// TIA Portal project "ContadoresHMI2" (V16)

(* hardware
DEVICE "S71500/ET200MP station_1"  S7-1500 station
   slot 0: "Rail_0"  Rack  6ES7 590-1***0-0AA0
   slot 1: "PLC_1"  CPU 1516-3 PN/DP  6ES7 516-3AN00-0AB0  V1.8
      slot 3: "CPU display_1"  6ES7591-1BA00-0AA0
      slot 32768: "PROFINET interface_1"  X1
         slot 32769: "Port_1"  X1 P1
         slot 32770: "Port_2"  X1 P2
      slot 33024: "PROFINET interface_2"  X2
         slot 33025: "Port_1"  X2 P1
      slot 33280: "DP interface_1"  X3
DEVICE "HMI_1"  TP700 Comfort
   slot 0: "HMI_1"  TP700 Comfort  6AV2 124-0GC01-0AX0  16.0.0.0
   slot 1: "HMI_RT_1"  TP700 Comfort  6AV2 124-0GC01-0AX0  16.0.0.0
   slot 5: "HMI_1.IE_CP_1"  PROFINET Interface  16.0.0.0
      slot 1: "PROFINET Interface_1"  PROFINET Interface
         slot 1: "Port_1"  Port
         slot 2: "Port_2"  Port
   slot 7: "HMI_1.MPI/DP_CP_1"  MPI/DP Interface  16.0.0.0
*)

// ===== PLC "PLC_1"  CPU 1516-3 PN/DP =====

VAR_GLOBAL   // PLC tag table "Default tag table"
   "ReiniciarJuego" AT %M6.0 : Bool;
   "CodigoS0J1" AT %M6.1 : Bool;
   "CodigoS1J1" AT %M6.2 : Bool;
   "CodigoS2J1" AT %M6.3 : Bool;
   "CodigoS3J1" AT %M6.4 : Bool;
   "CodigoO0J1" AT %M6.5 : Bool;
   "CodigoO1J1" AT %M6.6 : Bool;
   "CodigoO2J1" AT %M6.7 : Bool;
   "CodigoO3J1" AT %M7.0 : Bool;
   "CodigoS0J2" AT %M7.1 : Bool;
   "CodigoS1J2" AT %M7.2 : Bool;
   "CodigoS2J2" AT %M7.3 : Bool;
   "CodigoS3J2" AT %M7.4 : Bool;
   "CodigoO0J2" AT %M7.5 : Bool;
   "CodigoO1J2" AT %M7.6 : Bool;
   "CodigoO2J2" AT %M7.7 : Bool;
   "CodigoO3J2" AT %M8.0 : Bool;
   "Intento0J1" AT %M8.1 : Bool;
   "Intento1J1" AT %M8.2 : Bool;
   "Intento2J1" AT %M8.3 : Bool;
   "Intento3J1" AT %M8.4 : Bool;
   "Intento0J2" AT %M8.5 : Bool;
   "Intento1J2" AT %M8.6 : Bool;
   "Intento2J2" AT %M8.7 : Bool;
   "Intento3J2" AT %M9.0 : Bool;
   "IntentoCompletoJ1" AT %MW2 : UInt;
   "IntentoCompletoJ2" AT %MW4 : UInt;
   "Timer" AT %M9.3 : Bool;
   "Repetido" AT %M9.4 : Bool;
   "Panel1CafeJ1" AT %M9.5 : Bool;
   "Panel1RosaJ1" AT %M9.6 : Bool;
   "Panel1MoradoJ1" AT %M9.7 : Bool;
   "Panel1RojoJ1" AT %M10.0 : Bool;
   "Panel1AzulJ1" AT %M10.1 : Bool;
   "Panel1VerdeJ1" AT %M10.2 : Bool;
   "Panel1AmarilloJ1" AT %M10.3 : Bool;
   "Panel2CafeJ1" AT %M10.4 : Bool;
   "Panel2RosaJ1" AT %M10.5 : Bool;
   "Panel2MoradoJ1" AT %M10.6 : Bool;
   "Panel2RojoJ1" AT %M10.7 : Bool;
   "Panel2AzulJ1" AT %M11.0 : Bool;
   "Panel2VerdeJ1" AT %M11.1 : Bool;
   "Panel2AmarilloJ1" AT %M11.2 : Bool;
   "Panel1CafeJ2" AT %M11.3 : Bool;
   "Panel1RosaJ2" AT %M11.4 : Bool;
   "Panel1MoradoJ2" AT %M11.5 : Bool;
   "Panel1RojoJ2" AT %M11.6 : Bool;
   "Panel1AzulJ2" AT %M11.7 : Bool;
   "Panel1VerdeJ2" AT %M12.0 : Bool;
   "Panel1AmarilloJ2" AT %M12.1 : Bool;
   "Panel2CafeJ2" AT %M12.2 : Bool;
   "Panel2RosaJ2" AT %M12.3 : Bool;
   "Panel2MoradoJ2" AT %M12.4 : Bool;
   "Panel2RojoJ2" AT %M12.5 : Bool;
   "Panel2AzulJ2" AT %M12.6 : Bool;
   "Panel2VerdeJ2" AT %M12.7 : Bool;
   "Panel2AmarilloJ2" AT %M13.0 : Bool;
   "Panel1J1Activado" AT %M13.1 : Bool;
   "Panel2J1Activado" AT %M13.2 : Bool;
   "Panel1J2Activado" AT %M13.3 : Bool;
   "Panel2J2Activado" AT %M13.4 : Bool;
   "ReinicioCorrecto" AT %M13.5 : Bool;
   "Bounce1" AT %M13.6 : Bool;
   "Bounce2" AT %M13.7 : Bool;
   "Bounce3" AT %M14.0 : Bool;
   "Bounce5" AT %M14.1 : Bool;
   "Bounce6" AT %M14.2 : Bool;
   "Bounce7" AT %M14.3 : Bool;
   "Bounce8" AT %M14.4 : Bool;
   "Bounce10" AT %M14.5 : Bool;
   "MensajeCorrecto" AT %M14.6 : Bool;
   "Bounce4" AT %M14.7 : Bool;
   "Bounce9" AT %M15.0 : Bool;
   "ReiniciarContadorJ1" AT %M15.1 : Bool;
   "ReiniciarContadorJ2" AT %M15.2 : Bool;
   "ChecarIntento1J1" AT %M15.3 : Bool;
   "ChecarIntento2J1" AT %M15.4 : Bool;
   "ChecarIntento3J1" AT %M15.5 : Bool;
   "ChecarIntento4J1" AT %M15.6 : Bool;
   "ChecarIntento1J2" AT %M15.7 : Bool;
   "ChecarIntento2J2" AT %M16.0 : Bool;
   "ChecarIntento3J2" AT %M16.1 : Bool;
   "ChecarIntento4J2" AT %M16.2 : Bool;
   "ContadorCorr" AT %MW17 : UInt;
   "ContadorSimi" AT %MW20 : UInt;
   "ContadorError" AT %MW22 : UInt;
   "ContadorCorrTemp" AT %MW24 : UInt;
   "ContadorSimiTemp" AT %MW26 : UInt;
   "ReiniciarChecarCorr" AT %M28.0 : Bool;
   "ReiniciarChecarSimi" AT %M28.1 : Bool;
   "ReiniciarChecarError" AT %M28.2 : Bool;
   "ChecarIntentoCorrecto" AT %M28.3 : Bool;
   "ChecarIntento1SJ1" AT %M28.4 : Bool;
   "ChecarIntento2SJ1" AT %M28.5 : Bool;
   "ChecarIntento3SJ1" AT %M28.6 : Bool;
   "ChecarIntento4SJ1" AT %M28.7 : Bool;
   "ChecarIntento1SJ2" AT %M29.0 : Bool;
   "ChecarIntento2SJ2" AT %M29.1 : Bool;
   "ChecarIntento3SJ2" AT %M29.2 : Bool;
   "ChecarIntento4SJ2" AT %M29.3 : Bool;
   "CorrectasSimilares" AT %M29.4 : Bool;
   "IntentoCompletoCORR" AT %MW31 : UInt;
   "ReiniciarCorrSimiDisp" AT %M34.0 : Bool;
   "CondicionGanasteJ1" AT %M34.1 : Bool;
   "CondicionPerdisteJ1" AT %M34.2 : Bool;
   "CondicionGanasteJ2" AT %M34.3 : Bool;
   "CondicionPerdisteJ2" AT %M34.4 : Bool;
END_VAR

DATA_BLOCK "Var"   // DB3
{ S7_Optimized_Access := 'TRUE' }
VERSION : 0.1
   VAR
      V1 : Array[0..10, 0..10] of Int;
      CodigoSJ1 : Array[0..3] of Int;
      CodigoOJ1 : Array[0..3] of Int;
      CodigoSJ2 : Array[0..3] of Int;
      CodigoOJ2 : Array[0..3] of Int;
      VectorPrincipalJ1 : Array[0..7, 0..3] of Int;
      VectorSecundarioJ1 : Array[0..7, 0..3] of Int;
      VectorPrincipalJ2 : Array[0..7, 0..3] of Int;
      VectorSecundarioJ2 : Array[0..7, 0..3] of Int;
      VectorMensajes : Array[0..10] of Int;
      VectorMensajesReset : Array[0..10] of Int;
      VectorMensajesJ2 : Array[0..10] of Int;
      VectorMensajesResetJ2 : Array[0..10] of Int;
      VectorCorrectas : Array[0..7, 0..3] of Int;
      VectorCorrectasReset : Array[0..7, 0..3] of Int;
      CodigoSimilaresJ1 : Array[0..3] of Int;
      CodigoSimilaresJ1Temp : Array[0..3] of Int;
   END_VAR
BEGIN
END_DATA_BLOCK

// folder: System blocks/Program resources

DATA_BLOCK "ContadorCorrectas"   // DB1
{ S7_Optimized_Access := 'TRUE' }
AUTHOR : Simatic
FAMILY : IEC
NAME : UCNTR
VERSION : 1.2
// stored: InstanceOfName IEC_UCOUNTER
"IEC_UCOUNTER"
BEGIN
END_DATA_BLOCK

DATA_BLOCK "IEC_Counter_0_DB_1"   // DB2
{ S7_Optimized_Access := 'TRUE' }
AUTHOR : Simatic
FAMILY : IEC
NAME : UCNTR
VERSION : 1.2
// stored: InstanceOfName IEC_UCOUNTER
"IEC_UCOUNTER"
BEGIN
END_DATA_BLOCK

DATA_BLOCK "IEC_Timer_1_DB"   // DB4
{ S7_Optimized_Access := 'TRUE' }
AUTHOR : Simatic
FAMILY : IEC
NAME : IEC_TMR
VERSION : 1.0
// stored: InstanceOfName IEC_TIMER
"IEC_TIMER"
BEGIN
END_DATA_BLOCK

DATA_BLOCK "IEC_Timer_0_DB_1"   // DB5
{ S7_Optimized_Access := 'TRUE' }
AUTHOR : Simatic
FAMILY : IEC
NAME : IEC_TMR
VERSION : 1.0
// stored: InstanceOfName IEC_TIMER
"IEC_TIMER"
BEGIN
END_DATA_BLOCK

DATA_BLOCK "IEC_Timer_2_DB"   // DB6
{ S7_Optimized_Access := 'TRUE' }
AUTHOR : Simatic
FAMILY : IEC
NAME : IEC_TMR
VERSION : 1.0
// stored: InstanceOfName IEC_TIMER
"IEC_TIMER"
BEGIN
END_DATA_BLOCK

DATA_BLOCK "IEC_Timer_3_DB"   // DB7
{ S7_Optimized_Access := 'TRUE' }
AUTHOR : Simatic
FAMILY : IEC
NAME : IEC_TMR
VERSION : 1.0
// stored: InstanceOfName IEC_TIMER
"IEC_TIMER"
BEGIN
END_DATA_BLOCK

DATA_BLOCK "IEC_Timer_4_DB"   // DB8
{ S7_Optimized_Access := 'TRUE' }
AUTHOR : Simatic
FAMILY : IEC
NAME : IEC_TMR
VERSION : 1.0
// stored: InstanceOfName IEC_TIMER
"IEC_TIMER"
BEGIN
END_DATA_BLOCK

DATA_BLOCK "IEC_Timer_5_DB"   // DB9
{ S7_Optimized_Access := 'TRUE' }
AUTHOR : Simatic
FAMILY : IEC
NAME : IEC_TMR
VERSION : 1.0
// stored: InstanceOfName IEC_TIMER
"IEC_TIMER"
BEGIN
END_DATA_BLOCK

DATA_BLOCK "ContadorSimilares"   // DB10
{ S7_Optimized_Access := 'TRUE' }
AUTHOR : Simatic
FAMILY : IEC
NAME : UCNTR
VERSION : 1.2
// stored: InstanceOfName IEC_UCOUNTER
"IEC_UCOUNTER"
BEGIN
END_DATA_BLOCK

// folder: (top level)

ORGANIZATION_BLOCK "Main"   // OB1, LAD, ProgramCycle
TITLE = "Main Program Sweep (Cycle)"
{ S7_Optimized_Access := 'TRUE' }
VERSION : 0.1
   VAR_INPUT
      Initial_Call : Bool;   // Initial call of this OB
      Remanence : Bool;   // =True, if remanent data are available
   END_VAR
   VAR_TEMP   // added for the SCL form of the ladder/FBD networks
      _w1 : Bool;
      _w2 : Bool;
      _w3 : Bool;
      _w4 : Bool;
      _w5 : Bool;
      _w6 : Bool;
      _w7 : Bool;
      _w8 : Bool;
      _w9 : Bool;
      _w10 : Bool;
      _w11 : Bool;
      _w12 : Bool;
      _w13 : Bool;
      _w14 : Bool;
      _w15 : Bool;
      _w16 : Bool;
      _w17 : Bool;
      _w18 : Bool;
      _w19 : Bool;
      _w20 : Bool;
      _w21 : Bool;
      _w22 : Bool;
      _w23 : Bool;
      _w24 : Bool;
      _w25 : Bool;
      _w26 : Bool;
      _w27 : Bool;
      _w28 : Bool;
      _w29 : Bool;
      _w30 : Bool;
      _w31 : Bool;
      _w32 : Bool;
      _w33 : Bool;
      _w34 : Bool;
      _w35 : Bool;
      _w36 : Bool;
      _w37 : Bool;
      _w38 : Bool;
      _w39 : Bool;
      _w40 : Bool;
      _w41 : Bool;
      _w42 : Bool;
      _w43 : Bool;
      _w44 : Bool;
      _w45 : Bool;
      _w46 : Bool;
      _w47 : Bool;
      _w48 : Bool;
      _w49 : Bool;
      _w50 : Bool;
      _w51 : Bool;
      _w52 : Bool;
      _w53 : Bool;
      _w54 : Bool;
      _w55 : Bool;
      _w56 : Bool;
      _w57 : Bool;
      _w58 : Bool;
      _w59 : Bool;
      _w60 : Bool;
      _w61 : Bool;
      _w62 : Bool;
      _w63 : Bool;
      _w64 : Bool;
      _w65 : Bool;
      _w66 : Bool;
      _w67 : Bool;
      _w68 : Bool;
      _w69 : Bool;
      _w70 : Bool;
      _w71 : Bool;
      _w72 : Bool;
      _w73 : Bool;
      _w74 : Bool;
      _w75 : Bool;
      _w76 : Bool;
      _w77 : Bool;
      _w78 : Bool;
      _w79 : Bool;
      _w80 : Bool;
      _w81 : Bool;
      _w82 : Bool;
      _w83 : Bool;
      _w84 : Bool;
      _w85 : Bool;
      _w86 : Bool;
      _w87 : Bool;
      _w88 : Bool;
   END_VAR
BEGIN

REGION Network 1: Reiniciar Juego
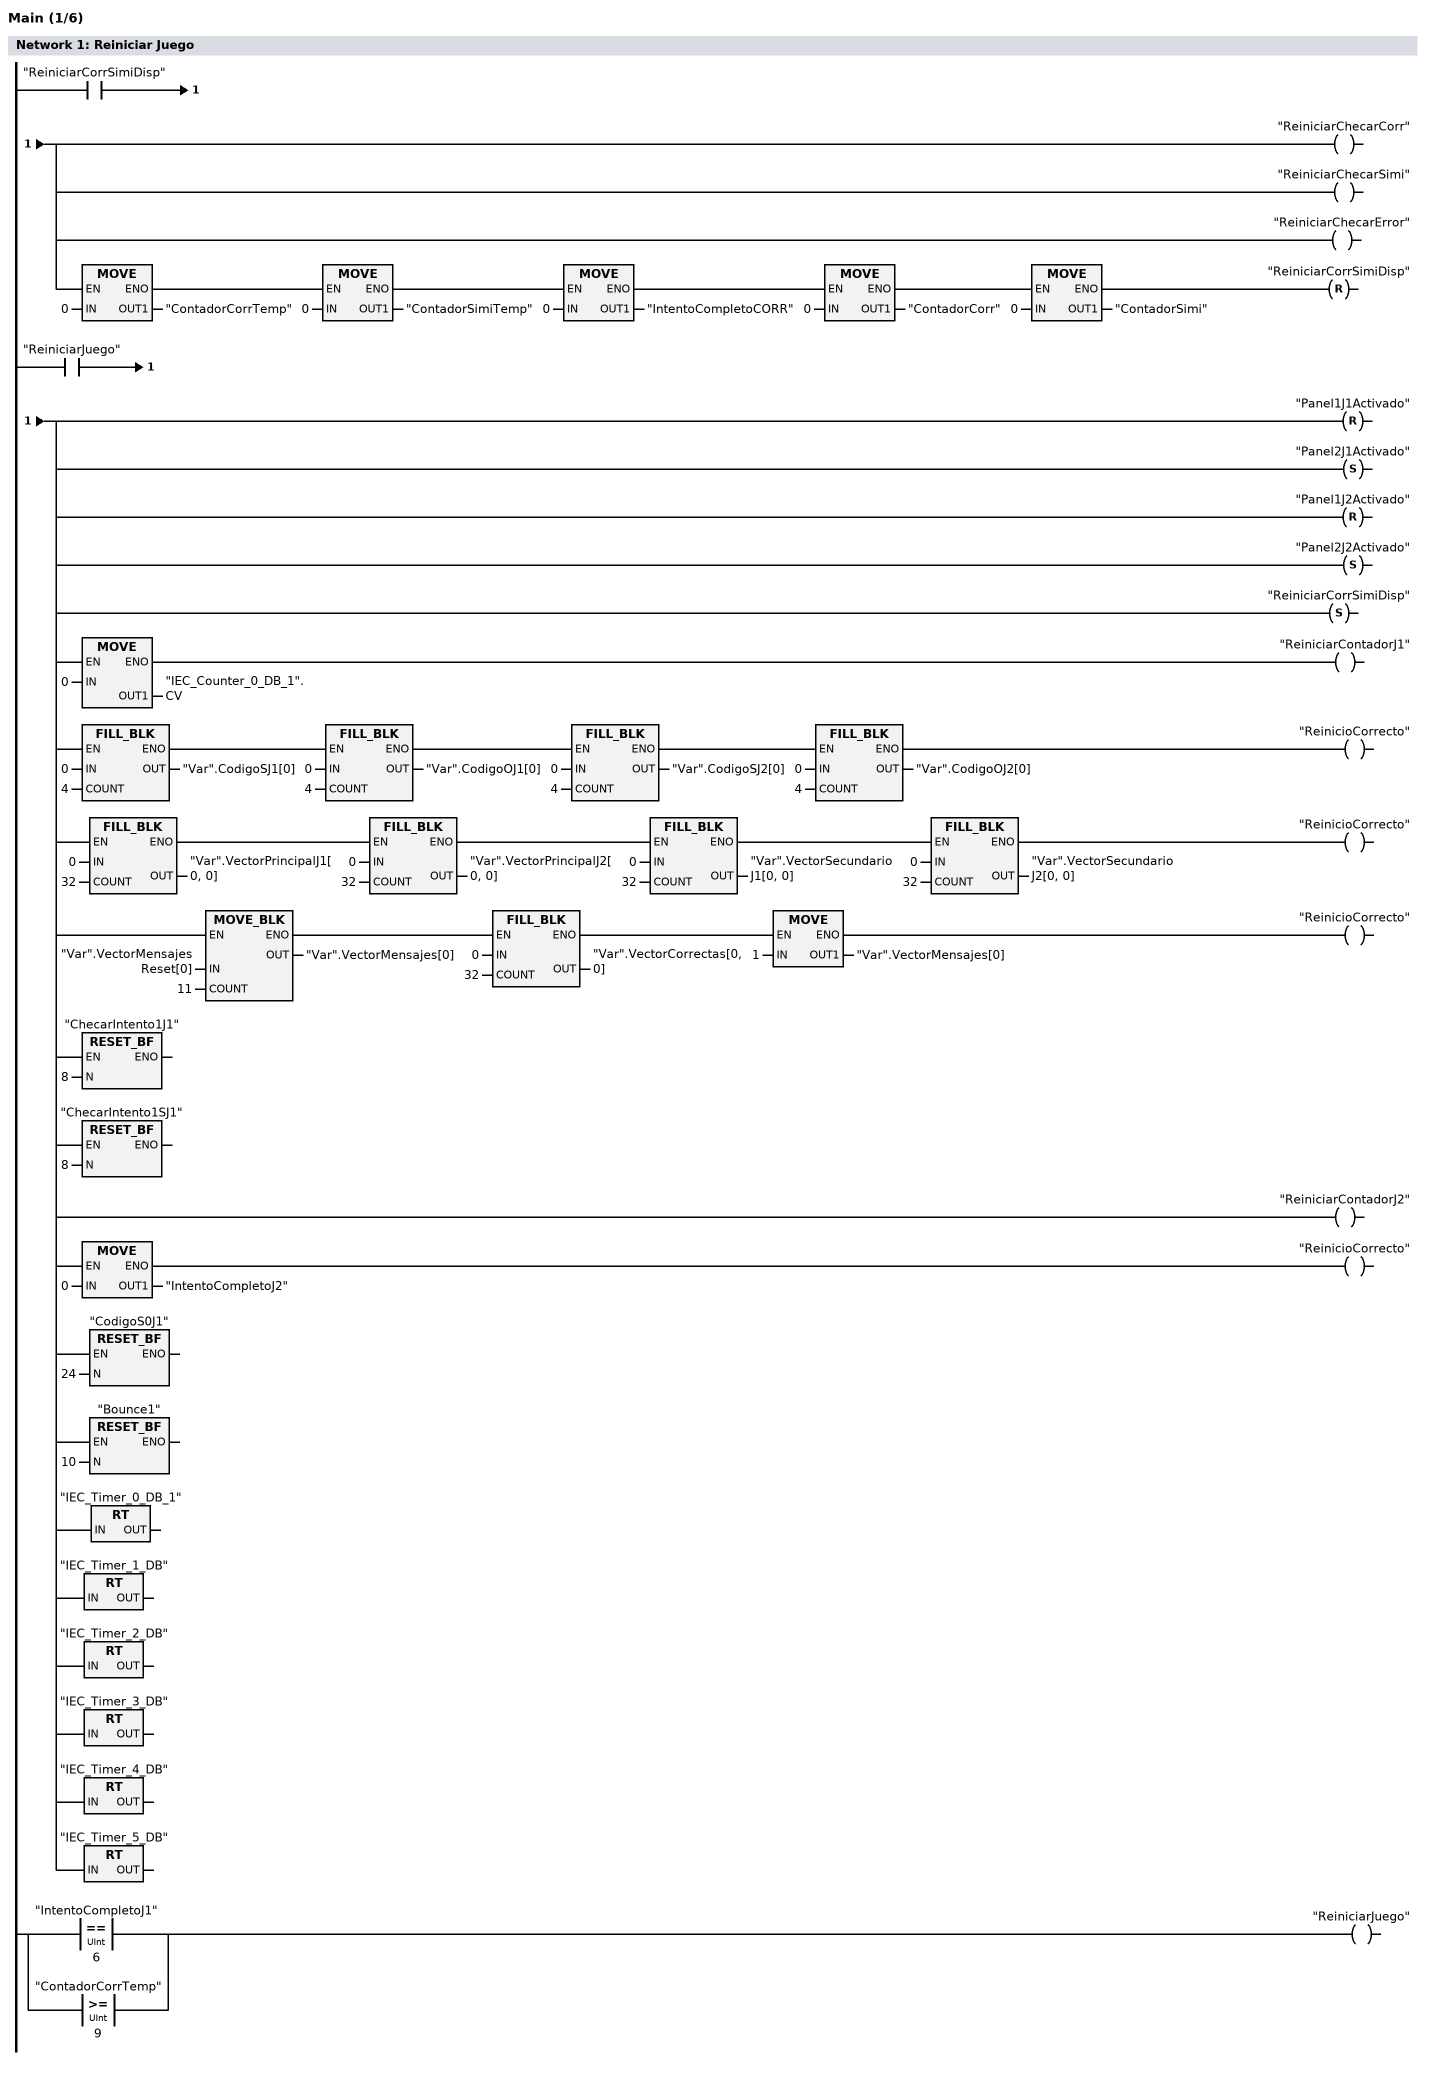
   // no SCL statement known for RBitfield: written as a call
   "ReiniciarChecarCorr" := "ReiniciarCorrSimiDisp";
   "ReiniciarChecarSimi" := "ReiniciarCorrSimiDisp";
   "ReiniciarChecarError" := "ReiniciarCorrSimiDisp";
   IF "ReiniciarCorrSimiDisp" THEN
       "ContadorCorrTemp" := 0;
       "ContadorSimiTemp" := 0;
       "IntentoCompletoCORR" := 0;
       "ContadorCorr" := 0;
       "ContadorSimi" := 0;
       "ReiniciarCorrSimiDisp" := FALSE;
   END_IF;
   IF "ReiniciarJuego" THEN
       "Panel1J1Activado" := FALSE;
       "Panel2J1Activado" := TRUE;
       "Panel1J2Activado" := FALSE;
       "Panel2J2Activado" := TRUE;
       "ReiniciarCorrSimiDisp" := TRUE;
       "IEC_Counter_0_DB_1".CV := 0;
   END_IF;
   "ReiniciarContadorJ1" := "ReiniciarJuego";
   #_w1 := "ReiniciarJuego";
   #_w2 := "ReiniciarJuego";
   IF #_w2 THEN
       FILL_BLK(IN := 0, COUNT := 4, OUT => "Var".CodigoSJ1[0]);
       FILL_BLK(IN := 0, COUNT := 4, OUT => "Var".CodigoOJ1[0]);
       FILL_BLK(IN := 0, COUNT := 4, OUT => "Var".CodigoSJ2[0]);
       FILL_BLK(IN := 0, COUNT := 4, OUT => "Var".CodigoOJ2[0]);
   END_IF;
   "ReinicioCorrecto" := #_w2;
   IF #_w1 THEN
       FILL_BLK(IN := 0, COUNT := 32, OUT => "Var".VectorPrincipalJ1[0, 0]);
       FILL_BLK(IN := 0, COUNT := 32, OUT => "Var".VectorPrincipalJ2[0, 0]);
       FILL_BLK(IN := 0, COUNT := 32, OUT => "Var".VectorSecundarioJ1[0, 0]);
       FILL_BLK(IN := 0, COUNT := 32, OUT => "Var".VectorSecundarioJ2[0, 0]);
   END_IF;
   "ReinicioCorrecto" := #_w1;
   IF #_w1 THEN
       MOVE_BLK(IN := "Var".VectorMensajesReset[0], COUNT := 11, OUT => "Var".VectorMensajes[0]);
       FILL_BLK(IN := 0, COUNT := 32, OUT => "Var".VectorCorrectas[0, 0]);
       "Var".VectorMensajes[0] := 1;
   END_IF;
   "ReinicioCorrecto" := #_w1;
   IF #_w1 THEN
       RESET_BF(operand := "ChecarIntento1J1", n := 8);
       RESET_BF(operand := "ChecarIntento1SJ1", n := 8);
   END_IF;
   "ReiniciarContadorJ2" := #_w1;
   IF #_w1 THEN "IntentoCompletoJ2" := 0; END_IF;
   "ReinicioCorrecto" := #_w1;
   IF #_w1 THEN
       RESET_BF(operand := "CodigoS0J1", n := 24);
       RESET_BF(operand := "Bounce1", n := 10);
       RESET_TIMER("IEC_Timer_0_DB_1");
       RESET_TIMER("IEC_Timer_1_DB");
       RESET_TIMER("IEC_Timer_2_DB");
       RESET_TIMER("IEC_Timer_3_DB");
       RESET_TIMER("IEC_Timer_4_DB");
       RESET_TIMER("IEC_Timer_5_DB");
   END_IF;
   "ReiniciarJuego" := ("IntentoCompletoJ1" = 6) OR ("ContadorCorrTemp" >= 9);
END_REGION

REGION Network 2: Seleccionar Codigo
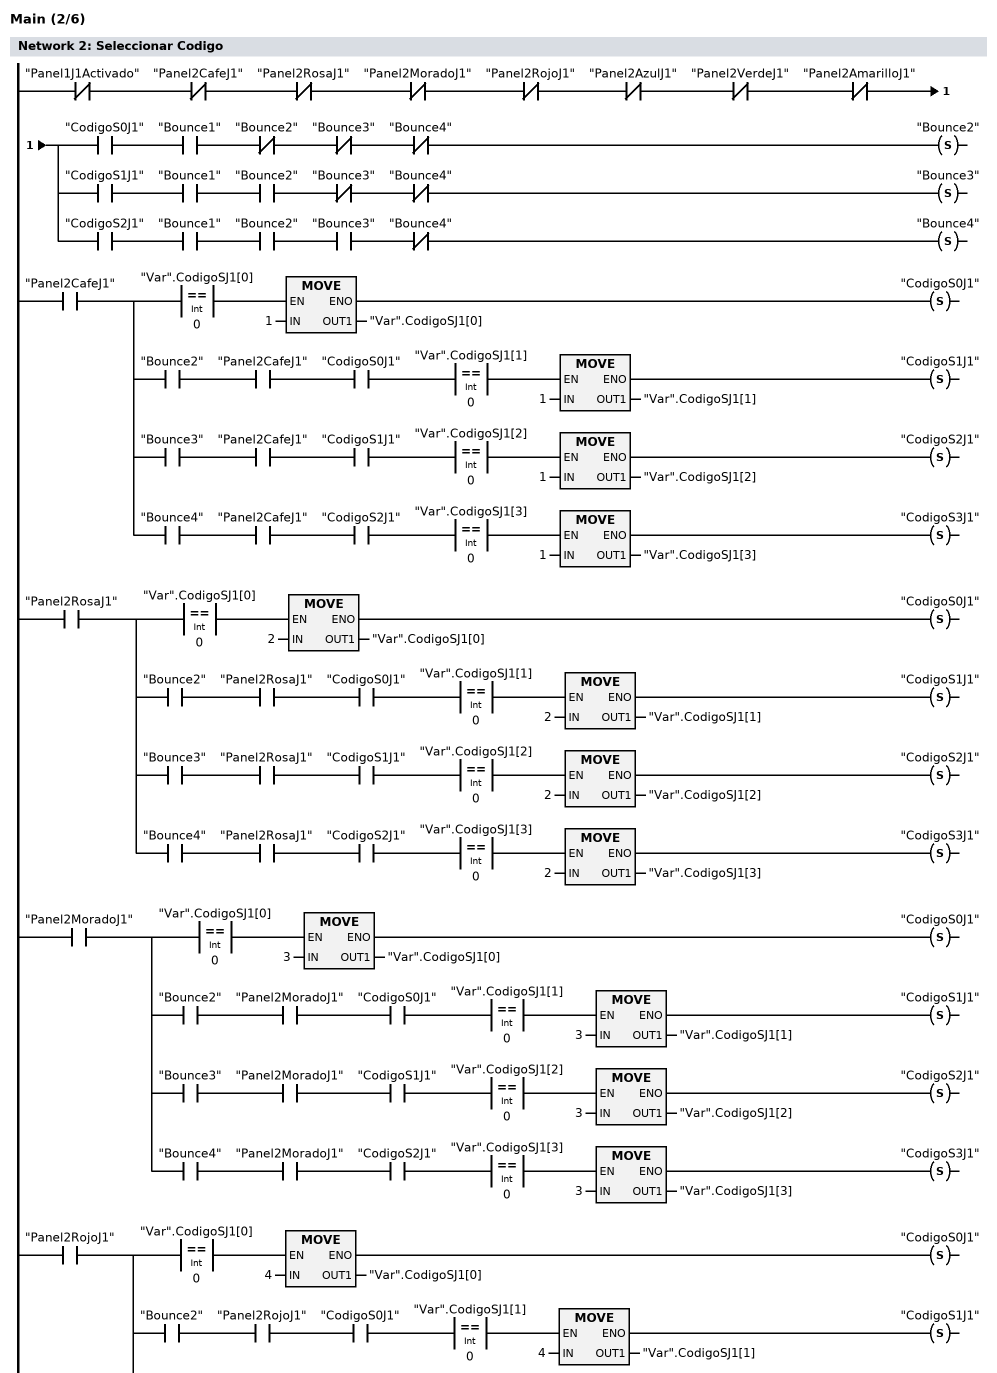
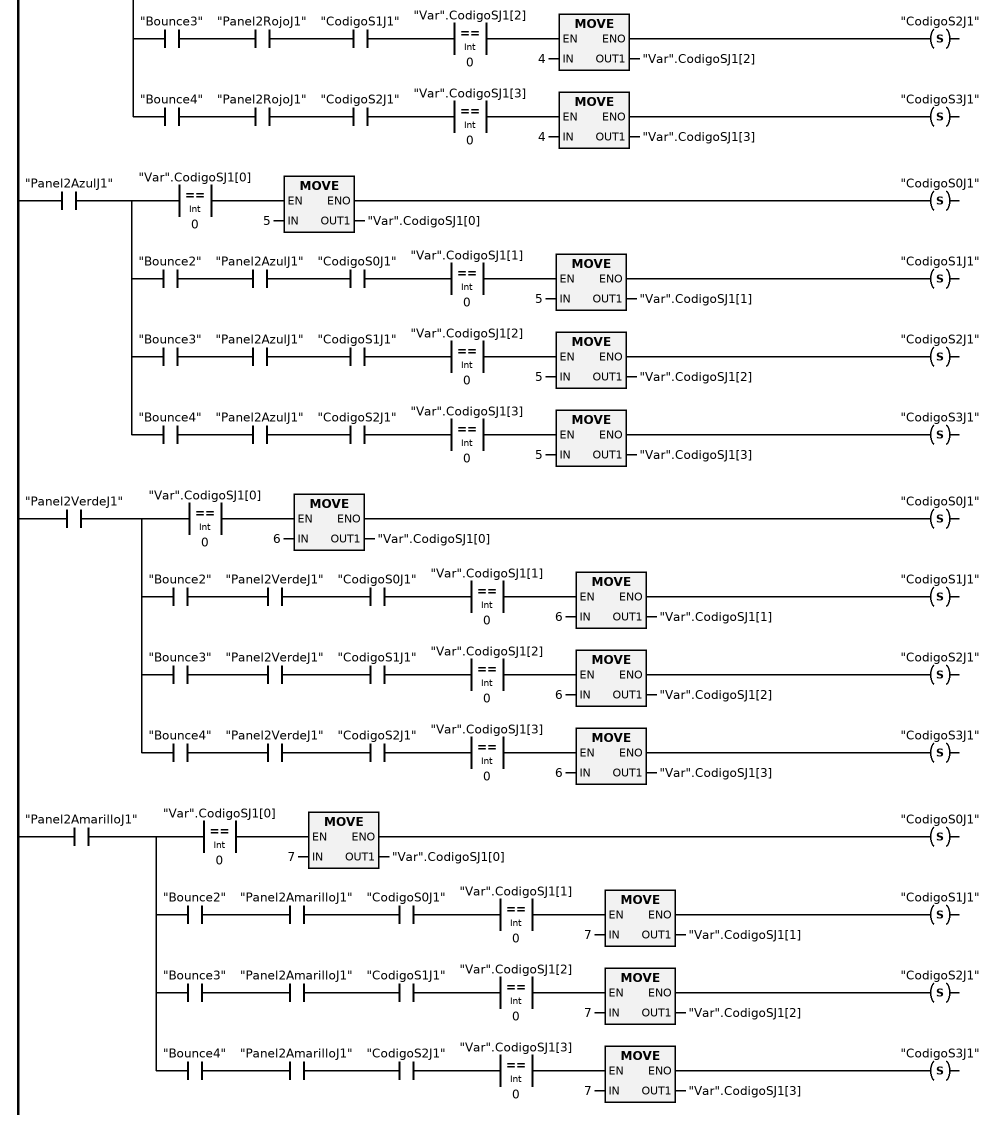
   RUNG wire#powerrail
      I_Contact( "Panel1J1Activado" )
      I_Contact( "Panel2CafeJ1" )
      I_Contact( "Panel2RosaJ1" )
      I_Contact( "Panel2MoradoJ1" )
      I_Contact( "Panel2RojoJ1" )
      I_Contact( "Panel2AzulJ1" )
      I_Contact( "Panel2VerdeJ1" )
      I_Contact( "Panel2AmarilloJ1" )
      wire#w1
      Contact( "CodigoS0J1" )
      Contact( "Bounce1" )
      I_Contact( "Bounce2" )
      I_Contact( "Bounce3" )
      I_Contact( "Bounce4" )
      S_Coil( "Bounce2" )
   END_RUNG
   RUNG wire#w1
      Contact( "CodigoS1J1" )
      Contact( "Bounce1" )
      Contact( "Bounce2" )
      I_Contact( "Bounce3" )
      I_Contact( "Bounce4" )
      S_Coil( "Bounce3" )
   END_RUNG
   RUNG wire#w1
      Contact( "CodigoS2J1" )
      Contact( "Bounce1" )
      Contact( "Bounce2" )
      Contact( "Bounce3" )
      I_Contact( "Bounce4" )
      S_Coil( "Bounce4" )
   END_RUNG
   RUNG wire#powerrail
      Contact( "Panel2CafeJ1" )
      wire#w2
      { S7_Templates := "SrcType := Int" } EQ_Contact(in1 := "Var".CodigoSJ1[0], in2 := 0)
      Move(in := 1, out1 => "Var".CodigoSJ1[0])
      S_Coil( "CodigoS0J1" )
   END_RUNG
   RUNG wire#w2
      Contact( "Bounce2" )
      Contact( "Panel2CafeJ1" )
      Contact( "CodigoS0J1" )
      { S7_Templates := "SrcType := Int" } EQ_Contact(in1 := "Var".CodigoSJ1[1], in2 := 0)
      Move(in := 1, out1 => "Var".CodigoSJ1[1])
      S_Coil( "CodigoS1J1" )
   END_RUNG
   RUNG wire#w2
      Contact( "Bounce3" )
      Contact( "Panel2CafeJ1" )
      Contact( "CodigoS1J1" )
      { S7_Templates := "SrcType := Int" } EQ_Contact(in1 := "Var".CodigoSJ1[2], in2 := 0)
      Move(in := 1, out1 => "Var".CodigoSJ1[2])
      S_Coil( "CodigoS2J1" )
   END_RUNG
   RUNG wire#w2
      Contact( "Bounce4" )
      Contact( "Panel2CafeJ1" )
      Contact( "CodigoS2J1" )
      { S7_Templates := "SrcType := Int" } EQ_Contact(in1 := "Var".CodigoSJ1[3], in2 := 0)
      Move(in := 1, out1 => "Var".CodigoSJ1[3])
      S_Coil( "CodigoS3J1" )
   END_RUNG
   RUNG wire#powerrail
      Contact( "Panel2RosaJ1" )
      wire#w3
      { S7_Templates := "SrcType := Int" } EQ_Contact(in1 := "Var".CodigoSJ1[0], in2 := 0)
      Move(in := 2, out1 => "Var".CodigoSJ1[0])
      S_Coil( "CodigoS0J1" )
   END_RUNG
   RUNG wire#w3
      Contact( "Bounce2" )
      Contact( "Panel2RosaJ1" )
      Contact( "CodigoS0J1" )
      { S7_Templates := "SrcType := Int" } EQ_Contact(in1 := "Var".CodigoSJ1[1], in2 := 0)
      Move(in := 2, out1 => "Var".CodigoSJ1[1])
      S_Coil( "CodigoS1J1" )
   END_RUNG
   RUNG wire#w3
      Contact( "Bounce3" )
      Contact( "Panel2RosaJ1" )
      Contact( "CodigoS1J1" )
      { S7_Templates := "SrcType := Int" } EQ_Contact(in1 := "Var".CodigoSJ1[2], in2 := 0)
      Move(in := 2, out1 => "Var".CodigoSJ1[2])
      S_Coil( "CodigoS2J1" )
   END_RUNG
   RUNG wire#w3
      Contact( "Bounce4" )
      Contact( "Panel2RosaJ1" )
      Contact( "CodigoS2J1" )
      { S7_Templates := "SrcType := Int" } EQ_Contact(in1 := "Var".CodigoSJ1[3], in2 := 0)
      Move(in := 2, out1 => "Var".CodigoSJ1[3])
      S_Coil( "CodigoS3J1" )
   END_RUNG
   RUNG wire#powerrail
      Contact( "Panel2MoradoJ1" )
      wire#w4
      { S7_Templates := "SrcType := Int" } EQ_Contact(in1 := "Var".CodigoSJ1[0], in2 := 0)
      Move(in := 3, out1 => "Var".CodigoSJ1[0])
      S_Coil( "CodigoS0J1" )
   END_RUNG
   RUNG wire#w4
      Contact( "Bounce2" )
      Contact( "Panel2MoradoJ1" )
      Contact( "CodigoS0J1" )
      { S7_Templates := "SrcType := Int" } EQ_Contact(in1 := "Var".CodigoSJ1[1], in2 := 0)
      Move(in := 3, out1 => "Var".CodigoSJ1[1])
      S_Coil( "CodigoS1J1" )
   END_RUNG
   RUNG wire#w4
      Contact( "Bounce3" )
      Contact( "Panel2MoradoJ1" )
      Contact( "CodigoS1J1" )
      { S7_Templates := "SrcType := Int" } EQ_Contact(in1 := "Var".CodigoSJ1[2], in2 := 0)
      Move(in := 3, out1 => "Var".CodigoSJ1[2])
      S_Coil( "CodigoS2J1" )
   END_RUNG
   RUNG wire#w4
      Contact( "Bounce4" )
      Contact( "Panel2MoradoJ1" )
      Contact( "CodigoS2J1" )
      { S7_Templates := "SrcType := Int" } EQ_Contact(in1 := "Var".CodigoSJ1[3], in2 := 0)
      Move(in := 3, out1 => "Var".CodigoSJ1[3])
      S_Coil( "CodigoS3J1" )
   END_RUNG
   RUNG wire#powerrail
      Contact( "Panel2RojoJ1" )
      wire#w5
      { S7_Templates := "SrcType := Int" } EQ_Contact(in1 := "Var".CodigoSJ1[0], in2 := 0)
      Move(in := 4, out1 => "Var".CodigoSJ1[0])
      S_Coil( "CodigoS0J1" )
   END_RUNG
   RUNG wire#w5
      Contact( "Bounce2" )
      Contact( "Panel2RojoJ1" )
      Contact( "CodigoS0J1" )
      { S7_Templates := "SrcType := Int" } EQ_Contact(in1 := "Var".CodigoSJ1[1], in2 := 0)
      Move(in := 4, out1 => "Var".CodigoSJ1[1])
      S_Coil( "CodigoS1J1" )
   END_RUNG
   RUNG wire#w5
      Contact( "Bounce3" )
      Contact( "Panel2RojoJ1" )
      Contact( "CodigoS1J1" )
      { S7_Templates := "SrcType := Int" } EQ_Contact(in1 := "Var".CodigoSJ1[2], in2 := 0)
      Move(in := 4, out1 => "Var".CodigoSJ1[2])
      S_Coil( "CodigoS2J1" )
   END_RUNG
   RUNG wire#w5
      Contact( "Bounce4" )
      Contact( "Panel2RojoJ1" )
      Contact( "CodigoS2J1" )
      { S7_Templates := "SrcType := Int" } EQ_Contact(in1 := "Var".CodigoSJ1[3], in2 := 0)
      Move(in := 4, out1 => "Var".CodigoSJ1[3])
      S_Coil( "CodigoS3J1" )
   END_RUNG
   RUNG wire#powerrail
      Contact( "Panel2AzulJ1" )
      wire#w6
      { S7_Templates := "SrcType := Int" } EQ_Contact(in1 := "Var".CodigoSJ1[0], in2 := 0)
      Move(in := 5, out1 => "Var".CodigoSJ1[0])
      S_Coil( "CodigoS0J1" )
   END_RUNG
   RUNG wire#w6
      Contact( "Bounce2" )
      Contact( "Panel2AzulJ1" )
      Contact( "CodigoS0J1" )
      { S7_Templates := "SrcType := Int" } EQ_Contact(in1 := "Var".CodigoSJ1[1], in2 := 0)
      Move(in := 5, out1 => "Var".CodigoSJ1[1])
      S_Coil( "CodigoS1J1" )
   END_RUNG
   RUNG wire#w6
      Contact( "Bounce3" )
      Contact( "Panel2AzulJ1" )
      Contact( "CodigoS1J1" )
      { S7_Templates := "SrcType := Int" } EQ_Contact(in1 := "Var".CodigoSJ1[2], in2 := 0)
      Move(in := 5, out1 => "Var".CodigoSJ1[2])
      S_Coil( "CodigoS2J1" )
   END_RUNG
   RUNG wire#w6
      Contact( "Bounce4" )
      Contact( "Panel2AzulJ1" )
      Contact( "CodigoS2J1" )
      { S7_Templates := "SrcType := Int" } EQ_Contact(in1 := "Var".CodigoSJ1[3], in2 := 0)
      Move(in := 5, out1 => "Var".CodigoSJ1[3])
      S_Coil( "CodigoS3J1" )
   END_RUNG
   RUNG wire#powerrail
      Contact( "Panel2VerdeJ1" )
      wire#w7
      { S7_Templates := "SrcType := Int" } EQ_Contact(in1 := "Var".CodigoSJ1[0], in2 := 0)
      Move(in := 6, out1 => "Var".CodigoSJ1[0])
      S_Coil( "CodigoS0J1" )
   END_RUNG
   RUNG wire#w7
      Contact( "Bounce2" )
      Contact( "Panel2VerdeJ1" )
      Contact( "CodigoS0J1" )
      { S7_Templates := "SrcType := Int" } EQ_Contact(in1 := "Var".CodigoSJ1[1], in2 := 0)
      Move(in := 6, out1 => "Var".CodigoSJ1[1])
      S_Coil( "CodigoS1J1" )
   END_RUNG
   RUNG wire#w7
      Contact( "Bounce3" )
      Contact( "Panel2VerdeJ1" )
      Contact( "CodigoS1J1" )
      { S7_Templates := "SrcType := Int" } EQ_Contact(in1 := "Var".CodigoSJ1[2], in2 := 0)
      Move(in := 6, out1 => "Var".CodigoSJ1[2])
      S_Coil( "CodigoS2J1" )
   END_RUNG
   RUNG wire#w7
      Contact( "Bounce4" )
      Contact( "Panel2VerdeJ1" )
      Contact( "CodigoS2J1" )
      { S7_Templates := "SrcType := Int" } EQ_Contact(in1 := "Var".CodigoSJ1[3], in2 := 0)
      Move(in := 6, out1 => "Var".CodigoSJ1[3])
      S_Coil( "CodigoS3J1" )
   END_RUNG
   RUNG wire#powerrail
      Contact( "Panel2AmarilloJ1" )
      wire#w8
      { S7_Templates := "SrcType := Int" } EQ_Contact(in1 := "Var".CodigoSJ1[0], in2 := 0)
      Move(in := 7, out1 => "Var".CodigoSJ1[0])
      S_Coil( "CodigoS0J1" )
   END_RUNG
   RUNG wire#w8
      Contact( "Bounce2" )
      Contact( "Panel2AmarilloJ1" )
      Contact( "CodigoS0J1" )
      { S7_Templates := "SrcType := Int" } EQ_Contact(in1 := "Var".CodigoSJ1[1], in2 := 0)
      Move(in := 7, out1 => "Var".CodigoSJ1[1])
      S_Coil( "CodigoS1J1" )
   END_RUNG
   RUNG wire#w8
      Contact( "Bounce3" )
      Contact( "Panel2AmarilloJ1" )
      Contact( "CodigoS1J1" )
      { S7_Templates := "SrcType := Int" } EQ_Contact(in1 := "Var".CodigoSJ1[2], in2 := 0)
      Move(in := 7, out1 => "Var".CodigoSJ1[2])
      S_Coil( "CodigoS2J1" )
   END_RUNG
   RUNG wire#w8
      Contact( "Bounce4" )
      Contact( "Panel2AmarilloJ1" )
      Contact( "CodigoS2J1" )
      { S7_Templates := "SrcType := Int" } EQ_Contact(in1 := "Var".CodigoSJ1[3], in2 := 0)
      Move(in := 7, out1 => "Var".CodigoSJ1[3])
      S_Coil( "CodigoS3J1" )
   END_RUNG
   // the same network as SCL:
   #_w1 := NOT "Panel1J1Activado" AND NOT "Panel2CafeJ1" AND NOT "Panel2RosaJ1" AND NOT "Panel2MoradoJ1" AND NOT "Panel2RojoJ1" AND NOT "Panel2AzulJ1" AND NOT "Panel2VerdeJ1" AND NOT "Panel2AmarilloJ1";
   IF #_w1 AND "CodigoS0J1" AND "Bounce1" AND NOT "Bounce2" AND NOT "Bounce3" AND NOT "Bounce4" THEN
       "Bounce2" := TRUE;
   END_IF;
   IF #_w1 AND "CodigoS1J1" AND "Bounce1" AND "Bounce2" AND NOT "Bounce3" AND NOT "Bounce4" THEN
       "Bounce3" := TRUE;
   END_IF;
   IF #_w1 AND "CodigoS2J1" AND "Bounce1" AND "Bounce2" AND "Bounce3" AND NOT "Bounce4" THEN
       "Bounce4" := TRUE;
   END_IF;
   #_w2 := "Panel2CafeJ1" AND ("Var".CodigoSJ1[0] = 0);
   IF #_w2 THEN
       "Var".CodigoSJ1[0] := 1;
       "CodigoS0J1" := TRUE;
   END_IF;
   #_w3 := "Panel2CafeJ1" AND "Bounce2" AND "Panel2CafeJ1" AND "CodigoS0J1" AND ("Var".CodigoSJ1[1] = 0);
   IF #_w3 THEN
       "Var".CodigoSJ1[1] := 1;
       "CodigoS1J1" := TRUE;
   END_IF;
   #_w4 := "Panel2CafeJ1" AND "Bounce3" AND "Panel2CafeJ1" AND "CodigoS1J1" AND ("Var".CodigoSJ1[2] = 0);
   IF #_w4 THEN
       "Var".CodigoSJ1[2] := 1;
       "CodigoS2J1" := TRUE;
   END_IF;
   #_w5 := "Panel2CafeJ1" AND "Bounce4" AND "Panel2CafeJ1" AND "CodigoS2J1" AND ("Var".CodigoSJ1[3] = 0);
   IF #_w5 THEN
       "Var".CodigoSJ1[3] := 1;
       "CodigoS3J1" := TRUE;
   END_IF;
   #_w6 := "Panel2RosaJ1" AND ("Var".CodigoSJ1[0] = 0);
   IF #_w6 THEN
       "Var".CodigoSJ1[0] := 2;
       "CodigoS0J1" := TRUE;
   END_IF;
   #_w7 := "Panel2RosaJ1" AND "Bounce2" AND "Panel2RosaJ1" AND "CodigoS0J1" AND ("Var".CodigoSJ1[1] = 0);
   IF #_w7 THEN
       "Var".CodigoSJ1[1] := 2;
       "CodigoS1J1" := TRUE;
   END_IF;
   #_w8 := "Panel2RosaJ1" AND "Bounce3" AND "Panel2RosaJ1" AND "CodigoS1J1" AND ("Var".CodigoSJ1[2] = 0);
   IF #_w8 THEN
       "Var".CodigoSJ1[2] := 2;
       "CodigoS2J1" := TRUE;
   END_IF;
   #_w9 := "Panel2RosaJ1" AND "Bounce4" AND "Panel2RosaJ1" AND "CodigoS2J1" AND ("Var".CodigoSJ1[3] = 0);
   IF #_w9 THEN
       "Var".CodigoSJ1[3] := 2;
       "CodigoS3J1" := TRUE;
   END_IF;
   #_w10 := "Panel2MoradoJ1" AND ("Var".CodigoSJ1[0] = 0);
   IF #_w10 THEN
       "Var".CodigoSJ1[0] := 3;
       "CodigoS0J1" := TRUE;
   END_IF;
   #_w11 := "Panel2MoradoJ1" AND "Bounce2" AND "Panel2MoradoJ1" AND "CodigoS0J1" AND ("Var".CodigoSJ1[1] = 0);
   IF #_w11 THEN
       "Var".CodigoSJ1[1] := 3;
       "CodigoS1J1" := TRUE;
   END_IF;
   #_w12 := "Panel2MoradoJ1" AND "Bounce3" AND "Panel2MoradoJ1" AND "CodigoS1J1" AND ("Var".CodigoSJ1[2] = 0);
   IF #_w12 THEN
       "Var".CodigoSJ1[2] := 3;
       "CodigoS2J1" := TRUE;
   END_IF;
   #_w13 := "Panel2MoradoJ1" AND "Bounce4" AND "Panel2MoradoJ1" AND "CodigoS2J1" AND ("Var".CodigoSJ1[3] = 0);
   IF #_w13 THEN
       "Var".CodigoSJ1[3] := 3;
       "CodigoS3J1" := TRUE;
   END_IF;
   #_w14 := "Panel2RojoJ1" AND ("Var".CodigoSJ1[0] = 0);
   IF #_w14 THEN
       "Var".CodigoSJ1[0] := 4;
       "CodigoS0J1" := TRUE;
   END_IF;
   #_w15 := "Panel2RojoJ1" AND "Bounce2" AND "Panel2RojoJ1" AND "CodigoS0J1" AND ("Var".CodigoSJ1[1] = 0);
   IF #_w15 THEN
       "Var".CodigoSJ1[1] := 4;
       "CodigoS1J1" := TRUE;
   END_IF;
   #_w16 := "Panel2RojoJ1" AND "Bounce3" AND "Panel2RojoJ1" AND "CodigoS1J1" AND ("Var".CodigoSJ1[2] = 0);
   IF #_w16 THEN
       "Var".CodigoSJ1[2] := 4;
       "CodigoS2J1" := TRUE;
   END_IF;
   #_w17 := "Panel2RojoJ1" AND "Bounce4" AND "Panel2RojoJ1" AND "CodigoS2J1" AND ("Var".CodigoSJ1[3] = 0);
   IF #_w17 THEN
       "Var".CodigoSJ1[3] := 4;
       "CodigoS3J1" := TRUE;
   END_IF;
   #_w18 := "Panel2AzulJ1" AND ("Var".CodigoSJ1[0] = 0);
   IF #_w18 THEN
       "Var".CodigoSJ1[0] := 5;
       "CodigoS0J1" := TRUE;
   END_IF;
   #_w19 := "Panel2AzulJ1" AND "Bounce2" AND "Panel2AzulJ1" AND "CodigoS0J1" AND ("Var".CodigoSJ1[1] = 0);
   IF #_w19 THEN
       "Var".CodigoSJ1[1] := 5;
       "CodigoS1J1" := TRUE;
   END_IF;
   #_w20 := "Panel2AzulJ1" AND "Bounce3" AND "Panel2AzulJ1" AND "CodigoS1J1" AND ("Var".CodigoSJ1[2] = 0);
   IF #_w20 THEN
       "Var".CodigoSJ1[2] := 5;
       "CodigoS2J1" := TRUE;
   END_IF;
   #_w21 := "Panel2AzulJ1" AND "Bounce4" AND "Panel2AzulJ1" AND "CodigoS2J1" AND ("Var".CodigoSJ1[3] = 0);
   IF #_w21 THEN
       "Var".CodigoSJ1[3] := 5;
       "CodigoS3J1" := TRUE;
   END_IF;
   #_w22 := "Panel2VerdeJ1" AND ("Var".CodigoSJ1[0] = 0);
   IF #_w22 THEN
       "Var".CodigoSJ1[0] := 6;
       "CodigoS0J1" := TRUE;
   END_IF;
   #_w23 := "Panel2VerdeJ1" AND "Bounce2" AND "Panel2VerdeJ1" AND "CodigoS0J1" AND ("Var".CodigoSJ1[1] = 0);
   IF #_w23 THEN
       "Var".CodigoSJ1[1] := 6;
       "CodigoS1J1" := TRUE;
   END_IF;
   #_w24 := "Panel2VerdeJ1" AND "Bounce3" AND "Panel2VerdeJ1" AND "CodigoS1J1" AND ("Var".CodigoSJ1[2] = 0);
   IF #_w24 THEN
       "Var".CodigoSJ1[2] := 6;
       "CodigoS2J1" := TRUE;
   END_IF;
   #_w25 := "Panel2VerdeJ1" AND "Bounce4" AND "Panel2VerdeJ1" AND "CodigoS2J1" AND ("Var".CodigoSJ1[3] = 0);
   IF #_w25 THEN
       "Var".CodigoSJ1[3] := 6;
       "CodigoS3J1" := TRUE;
   END_IF;
   #_w26 := "Panel2AmarilloJ1" AND ("Var".CodigoSJ1[0] = 0);
   IF #_w26 THEN
       "Var".CodigoSJ1[0] := 7;
       "CodigoS0J1" := TRUE;
   END_IF;
   #_w27 := "Panel2AmarilloJ1" AND "Bounce2" AND "Panel2AmarilloJ1" AND "CodigoS0J1" AND ("Var".CodigoSJ1[1] = 0);
   IF #_w27 THEN
       "Var".CodigoSJ1[1] := 7;
       "CodigoS1J1" := TRUE;
   END_IF;
   #_w28 := "Panel2AmarilloJ1" AND "Bounce3" AND "Panel2AmarilloJ1" AND "CodigoS1J1" AND ("Var".CodigoSJ1[2] = 0);
   IF #_w28 THEN
       "Var".CodigoSJ1[2] := 7;
       "CodigoS2J1" := TRUE;
   END_IF;
   #_w29 := "Panel2AmarilloJ1" AND "Bounce4" AND "Panel2AmarilloJ1" AND "CodigoS2J1" AND ("Var".CodigoSJ1[3] = 0);
   IF #_w29 THEN
       "Var".CodigoSJ1[3] := 7;
       "CodigoS3J1" := TRUE;
   END_IF;
END_REGION

REGION Network 3: Clave Secreta
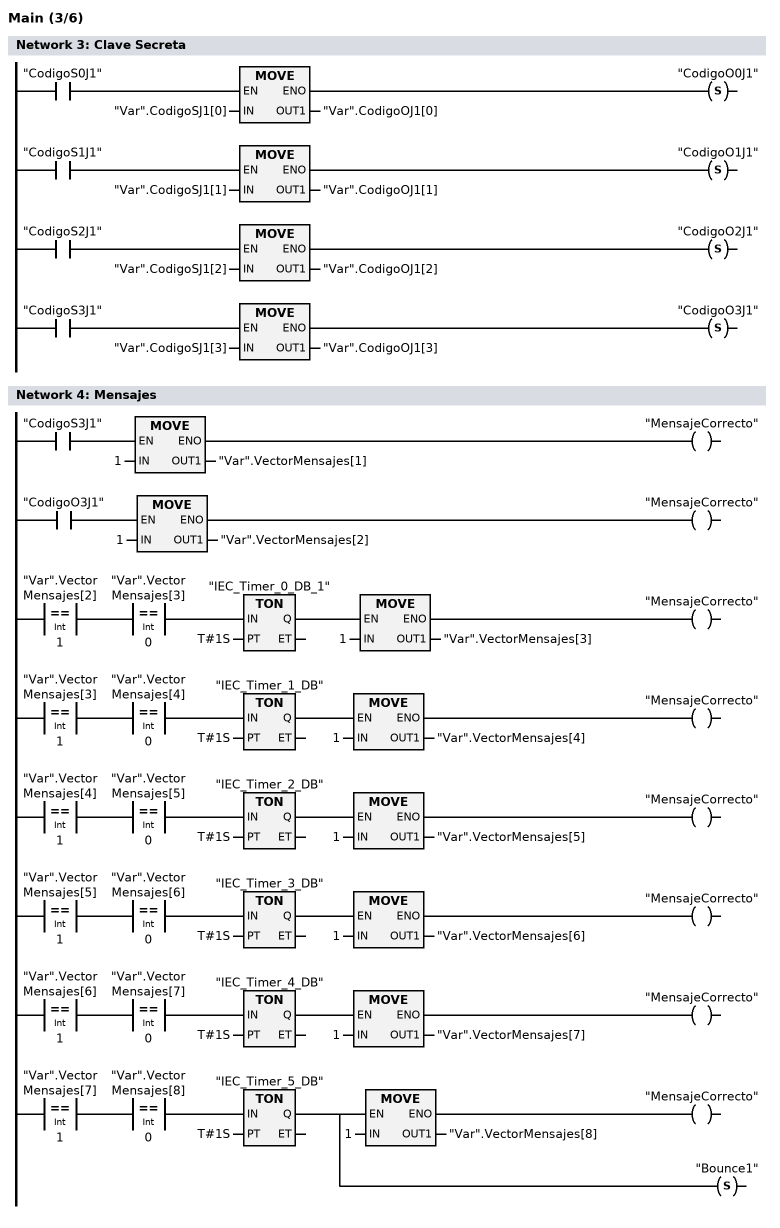
   RUNG wire#powerrail
      Contact( "CodigoS0J1" )
      Move(in := "Var".CodigoSJ1[0], out1 => "Var".CodigoOJ1[0])
      S_Coil( "CodigoO0J1" )
   END_RUNG
   RUNG wire#powerrail
      Contact( "CodigoS1J1" )
      Move(in := "Var".CodigoSJ1[1], out1 => "Var".CodigoOJ1[1])
      S_Coil( "CodigoO1J1" )
   END_RUNG
   RUNG wire#powerrail
      Contact( "CodigoS2J1" )
      Move(in := "Var".CodigoSJ1[2], out1 => "Var".CodigoOJ1[2])
      S_Coil( "CodigoO2J1" )
   END_RUNG
   RUNG wire#powerrail
      Contact( "CodigoS3J1" )
      Move(in := "Var".CodigoSJ1[3], out1 => "Var".CodigoOJ1[3])
      S_Coil( "CodigoO3J1" )
   END_RUNG
   // the same network as SCL:
   IF "CodigoS0J1" THEN
       "Var".CodigoOJ1[0] := "Var".CodigoSJ1[0];
       "CodigoO0J1" := TRUE;
   END_IF;
   IF "CodigoS1J1" THEN
       "Var".CodigoOJ1[1] := "Var".CodigoSJ1[1];
       "CodigoO1J1" := TRUE;
   END_IF;
   IF "CodigoS2J1" THEN
       "Var".CodigoOJ1[2] := "Var".CodigoSJ1[2];
       "CodigoO2J1" := TRUE;
   END_IF;
   IF "CodigoS3J1" THEN
       "Var".CodigoOJ1[3] := "Var".CodigoSJ1[3];
       "CodigoO3J1" := TRUE;
   END_IF;
END_REGION

REGION Network 4: Mensajes
   IF "CodigoS3J1" THEN "Var".VectorMensajes[1] := 1; END_IF;
   "MensajeCorrecto" := "CodigoS3J1";
   IF "CodigoO3J1" THEN "Var".VectorMensajes[2] := 1; END_IF;
   "MensajeCorrecto" := "CodigoO3J1";
   "IEC_Timer_0_DB_1".TON(IN := ("Var".VectorMensajes[2] = 1) AND ("Var".VectorMensajes[3] = 0), PT := T#1S);
   IF "IEC_Timer_0_DB_1".Q THEN "Var".VectorMensajes[3] := 1; END_IF;
   "MensajeCorrecto" := "IEC_Timer_0_DB_1".Q;
   "IEC_Timer_1_DB".TON(IN := ("Var".VectorMensajes[3] = 1) AND ("Var".VectorMensajes[4] = 0), PT := T#1S);
   IF "IEC_Timer_1_DB".Q THEN "Var".VectorMensajes[4] := 1; END_IF;
   "MensajeCorrecto" := "IEC_Timer_1_DB".Q;
   "IEC_Timer_2_DB".TON(IN := ("Var".VectorMensajes[4] = 1) AND ("Var".VectorMensajes[5] = 0), PT := T#1S);
   IF "IEC_Timer_2_DB".Q THEN "Var".VectorMensajes[5] := 1; END_IF;
   "MensajeCorrecto" := "IEC_Timer_2_DB".Q;
   "IEC_Timer_3_DB".TON(IN := ("Var".VectorMensajes[5] = 1) AND ("Var".VectorMensajes[6] = 0), PT := T#1S);
   IF "IEC_Timer_3_DB".Q THEN "Var".VectorMensajes[6] := 1; END_IF;
   "MensajeCorrecto" := "IEC_Timer_3_DB".Q;
   "IEC_Timer_4_DB".TON(IN := ("Var".VectorMensajes[6] = 1) AND ("Var".VectorMensajes[7] = 0), PT := T#1S);
   IF "IEC_Timer_4_DB".Q THEN "Var".VectorMensajes[7] := 1; END_IF;
   "MensajeCorrecto" := "IEC_Timer_4_DB".Q;
   "IEC_Timer_5_DB".TON(IN := ("Var".VectorMensajes[7] = 1) AND ("Var".VectorMensajes[8] = 0), PT := T#1S);
   IF "IEC_Timer_5_DB".Q THEN "Var".VectorMensajes[8] := 1; END_IF;
   "MensajeCorrecto" := "IEC_Timer_5_DB".Q;
   IF "IEC_Timer_5_DB".Q THEN "Bounce1" := TRUE; END_IF;
END_REGION

REGION Network 5: ActivarOtroPanel
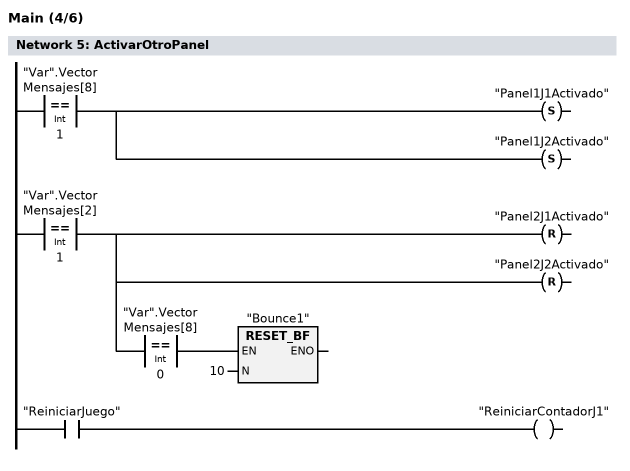
   // no SCL statement known for RBitfield: written as a call
   IF "Var".VectorMensajes[8] = 1 THEN
       "Panel1J1Activado" := TRUE;
       "Panel1J2Activado" := TRUE;
   END_IF;
   #_w1 := "Var".VectorMensajes[2] = 1;
   IF #_w1 THEN
       "Panel2J1Activado" := FALSE;
       "Panel2J2Activado" := FALSE;
   END_IF;
   IF #_w1 AND ("Var".VectorMensajes[8] = 0) THEN RESET_BF(operand := "Bounce1", n := 10); END_IF;
   "ReiniciarContadorJ1" := "ReiniciarJuego";
END_REGION

REGION Network 6: Seleccionar Intentos
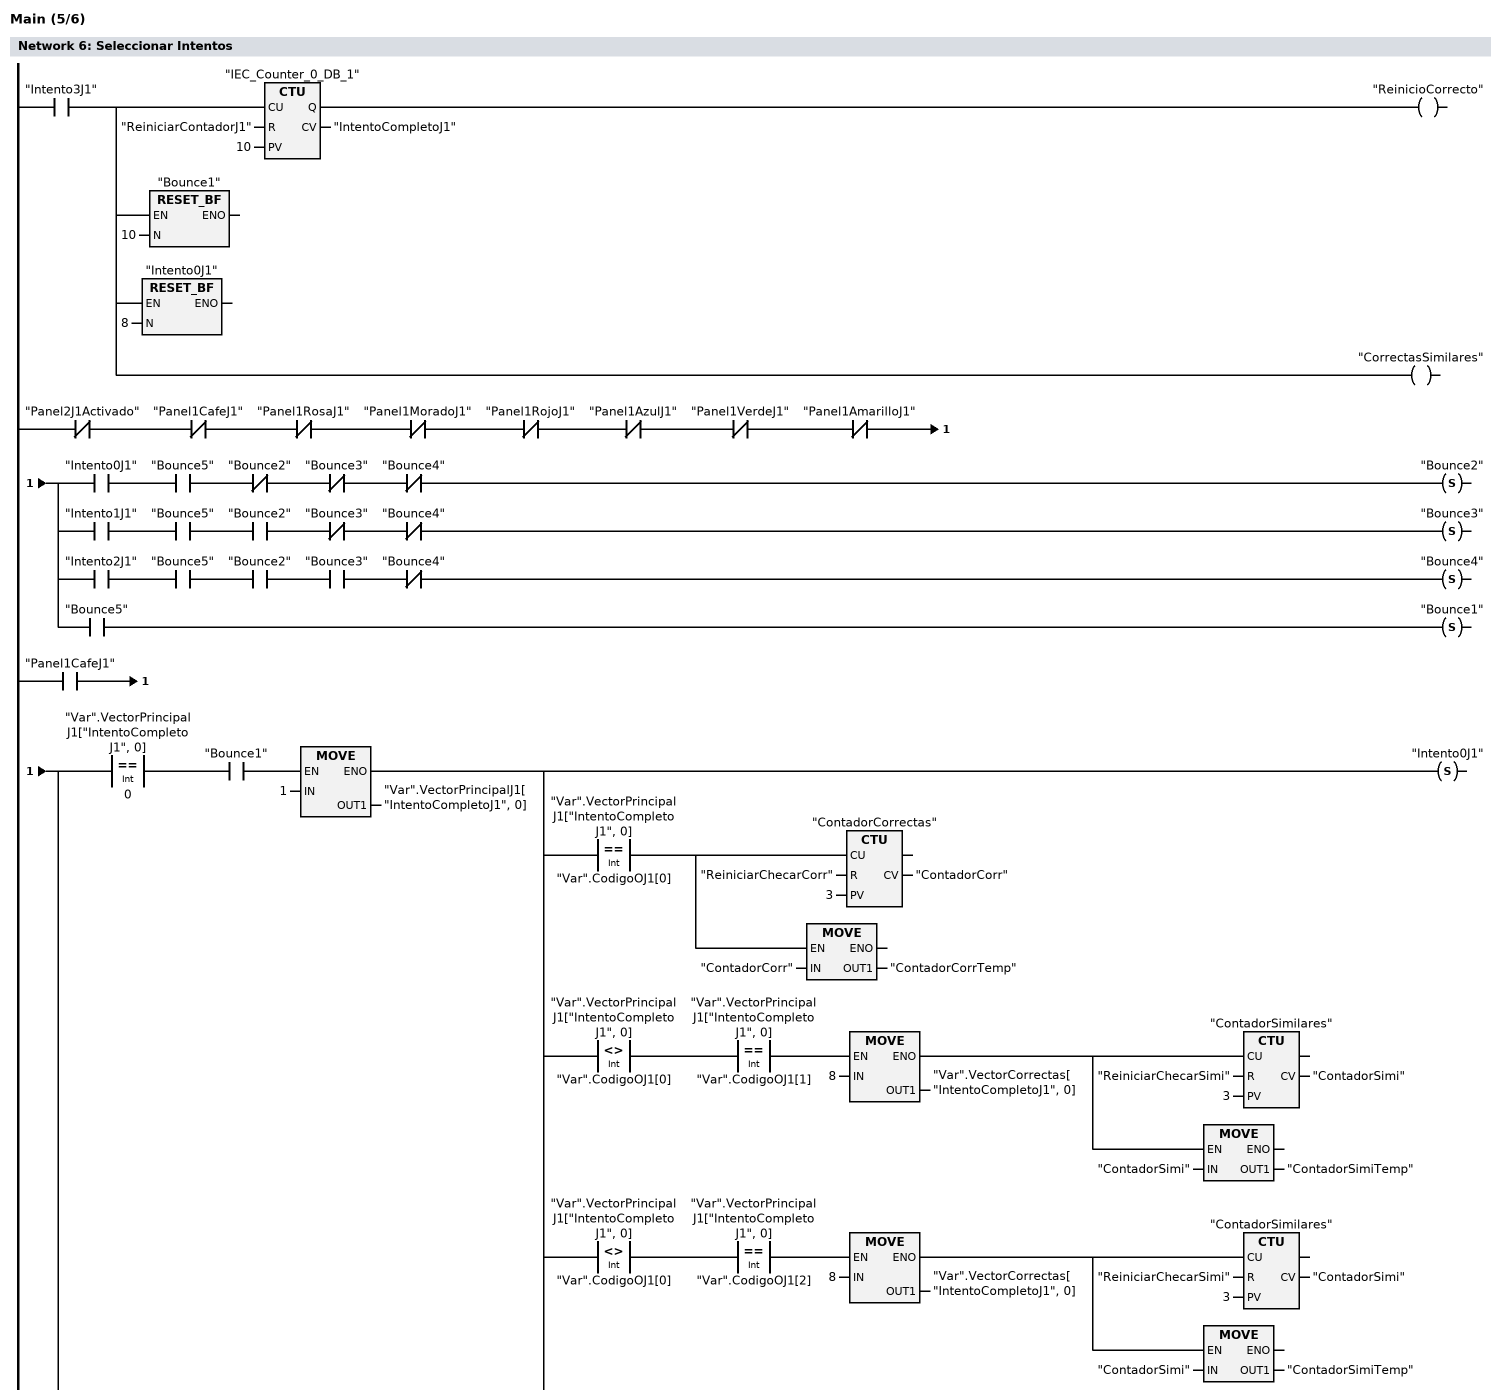
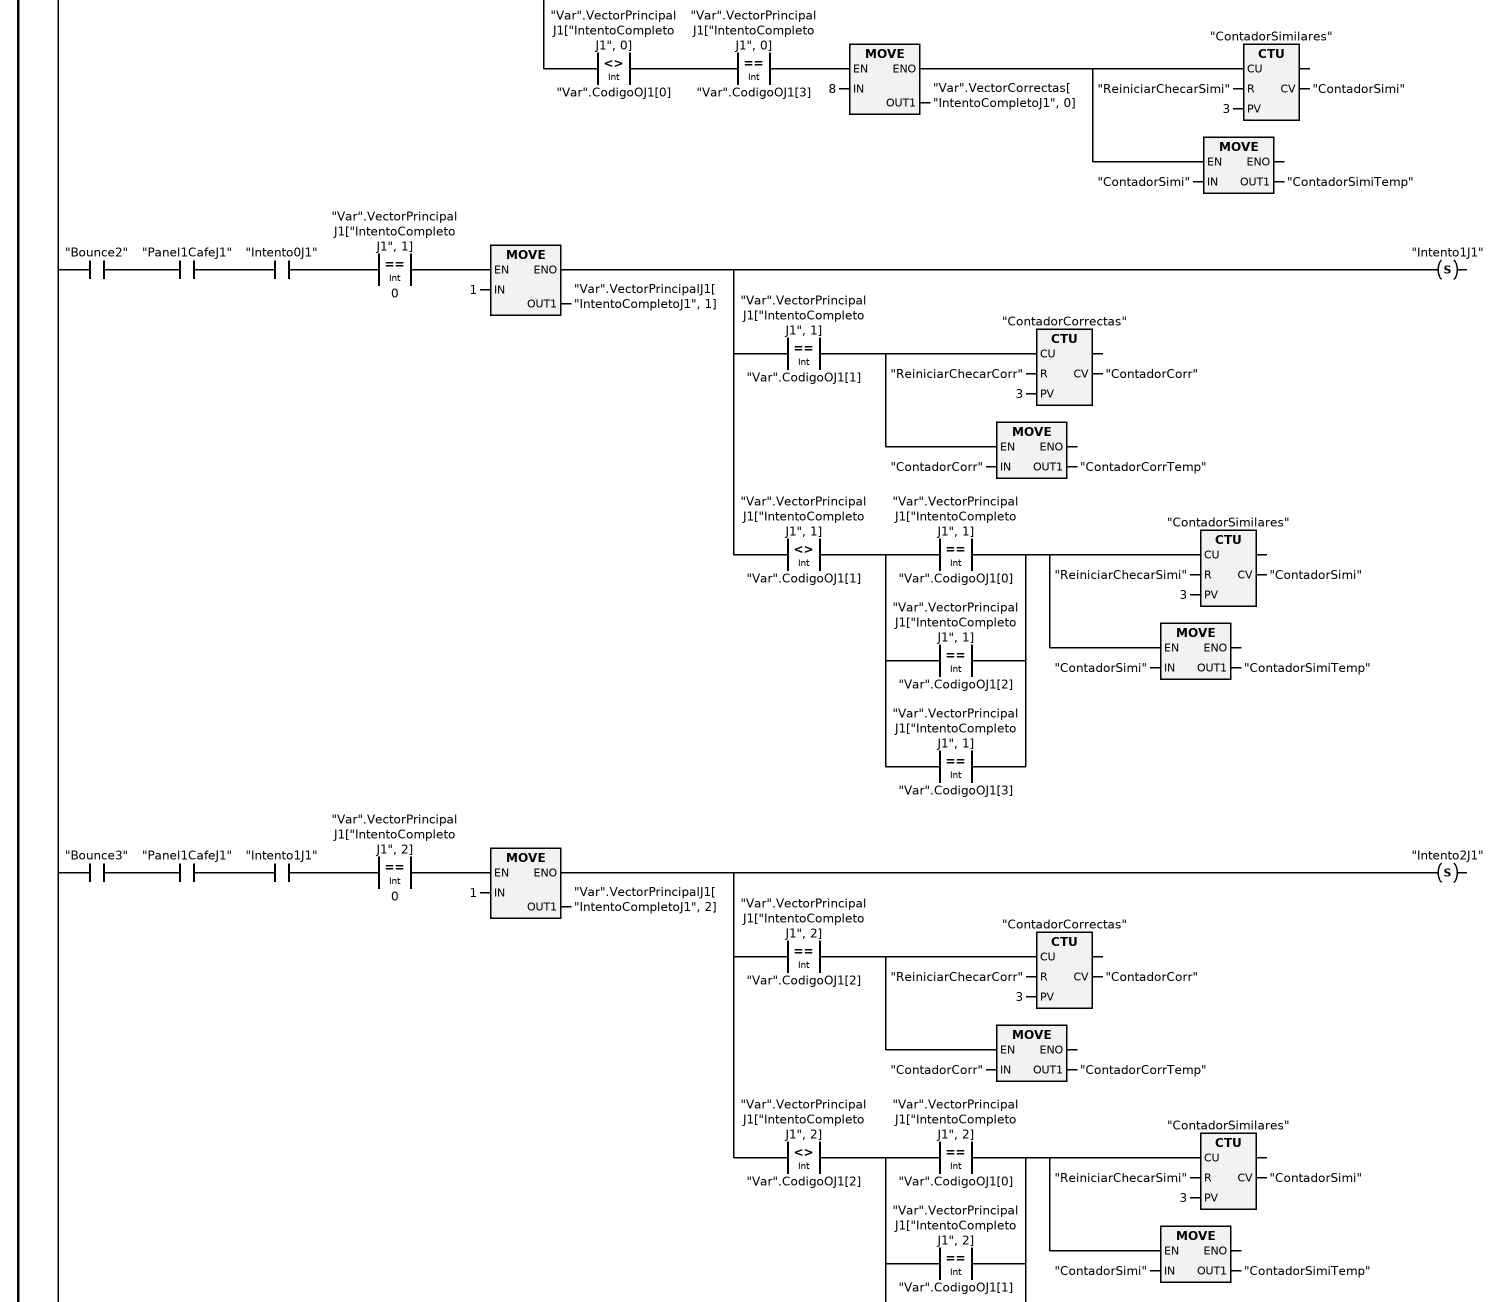
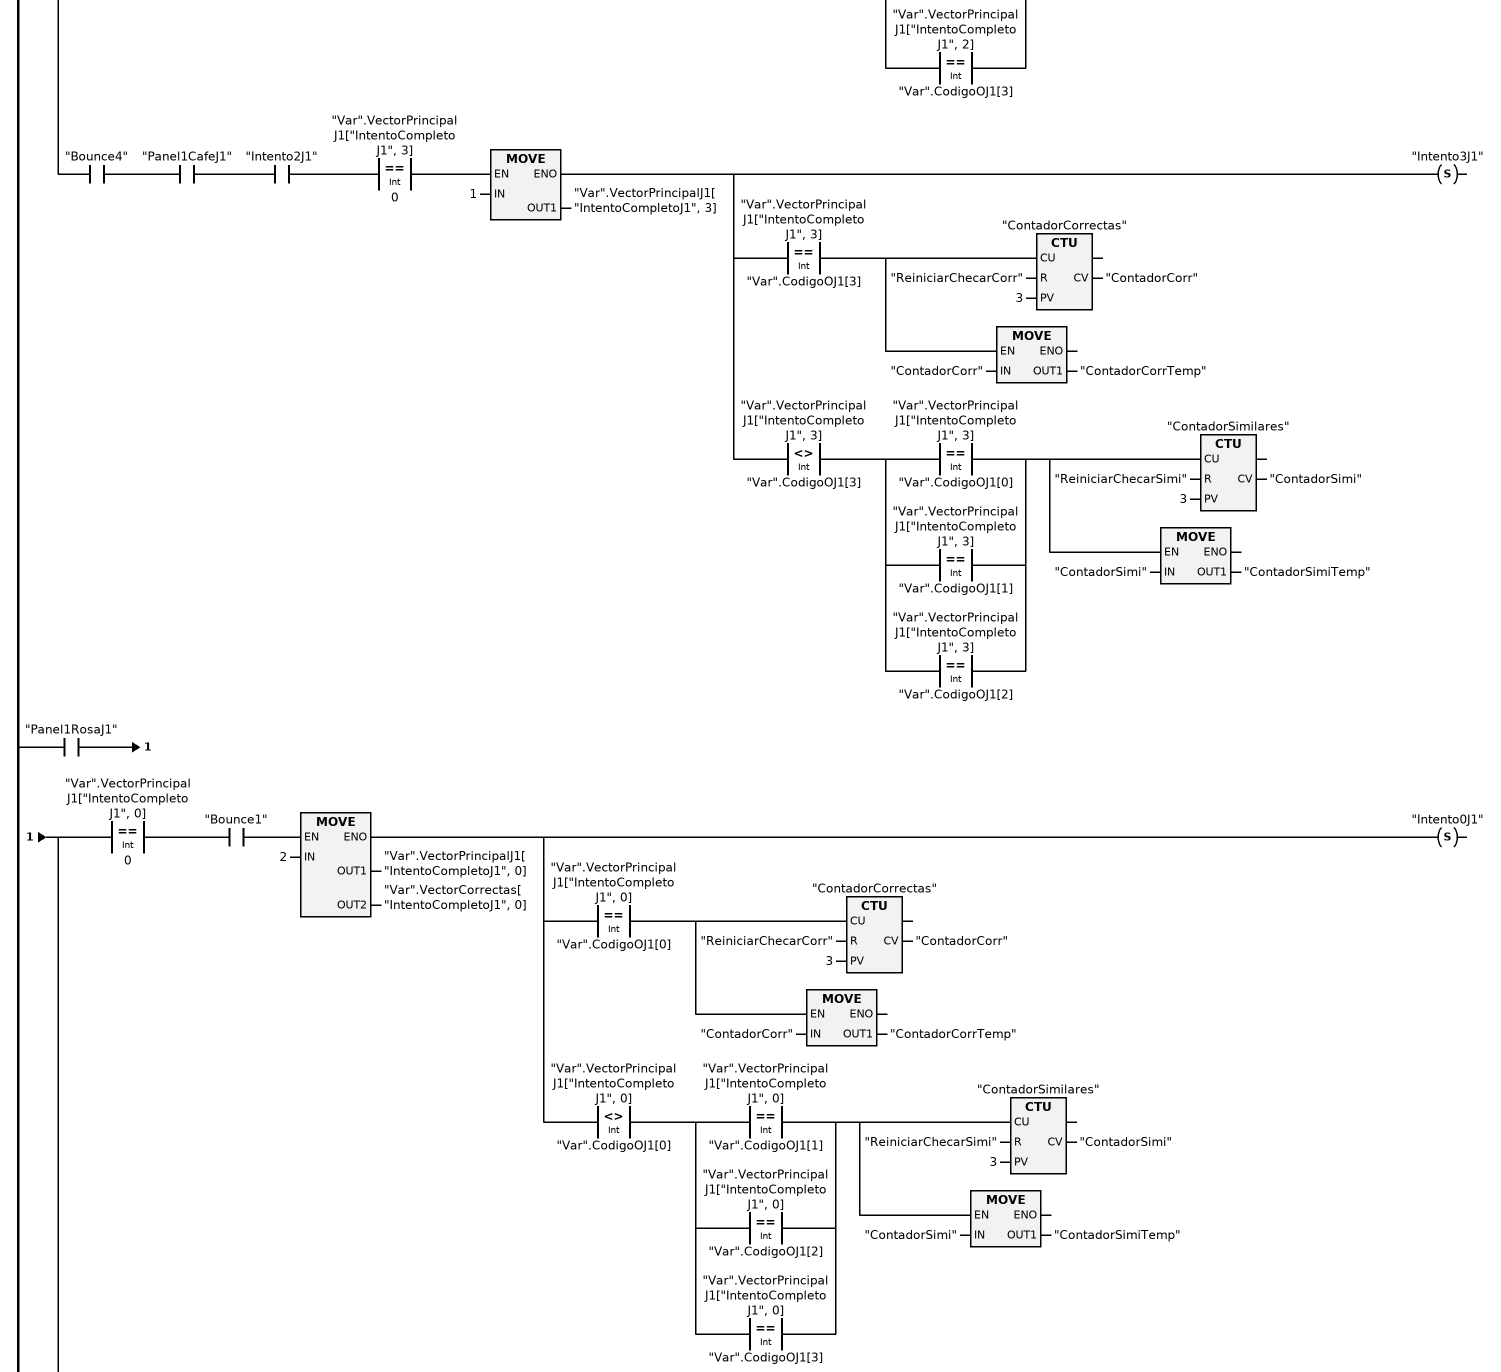
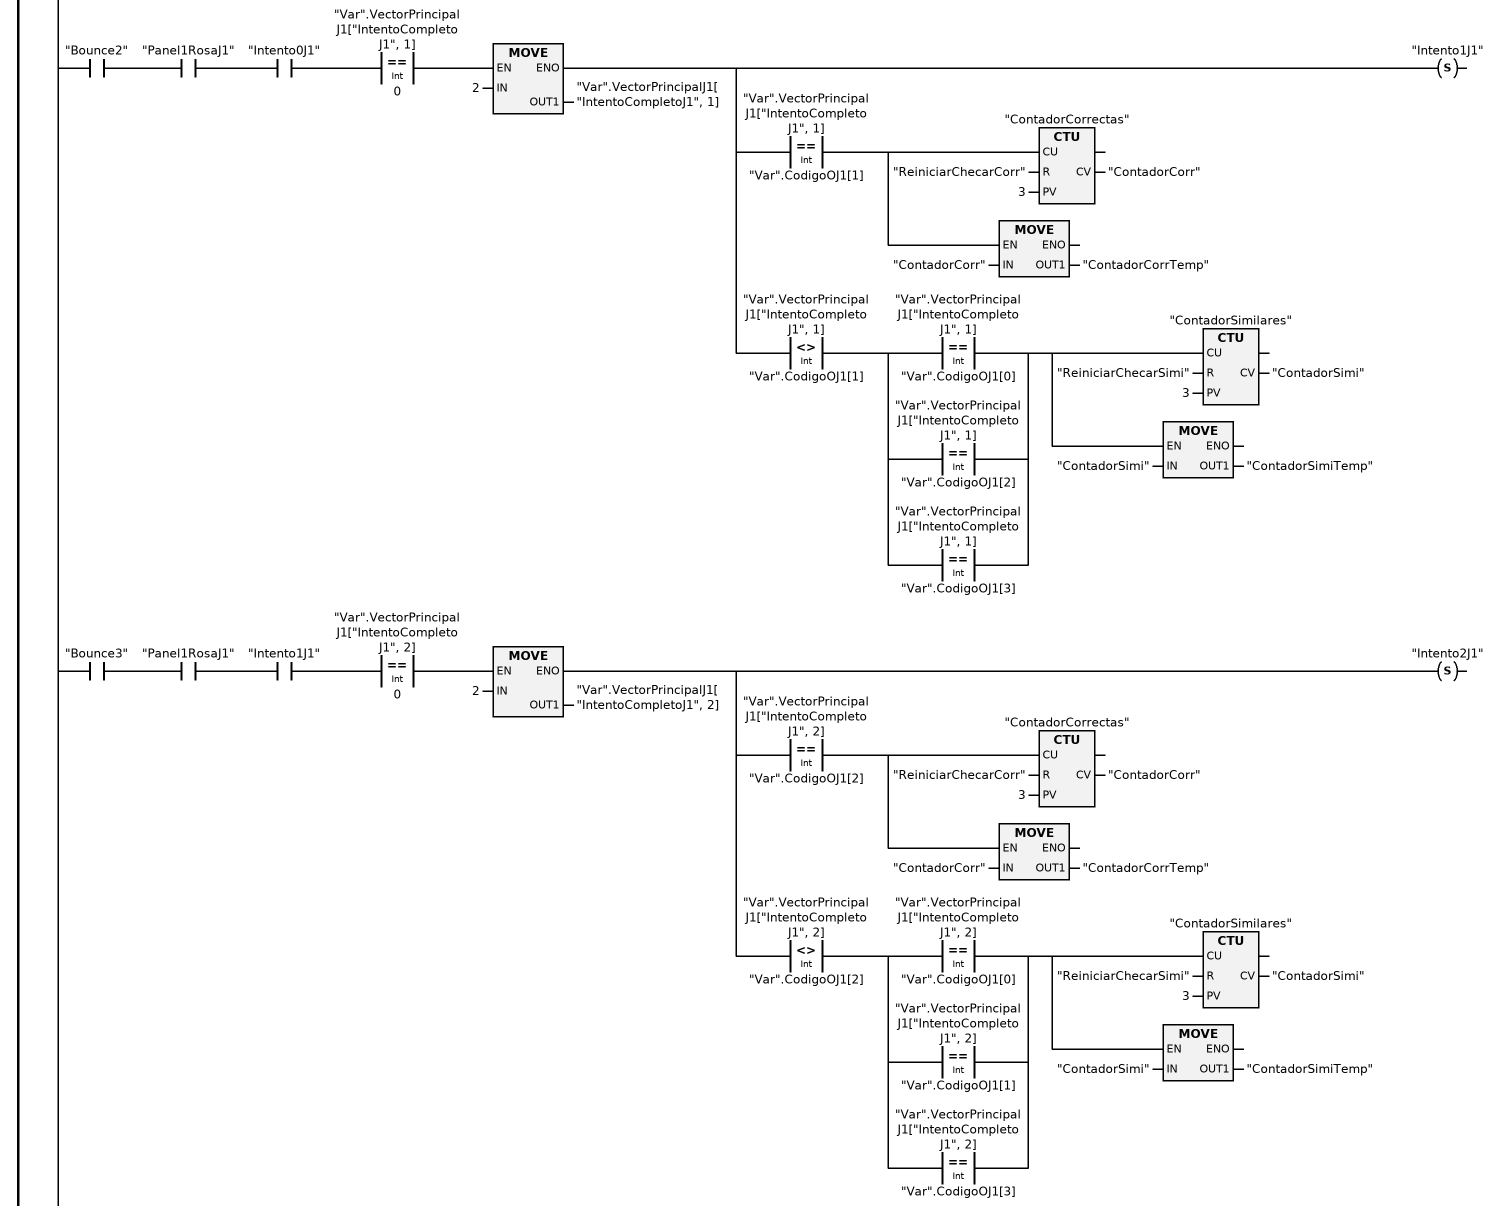
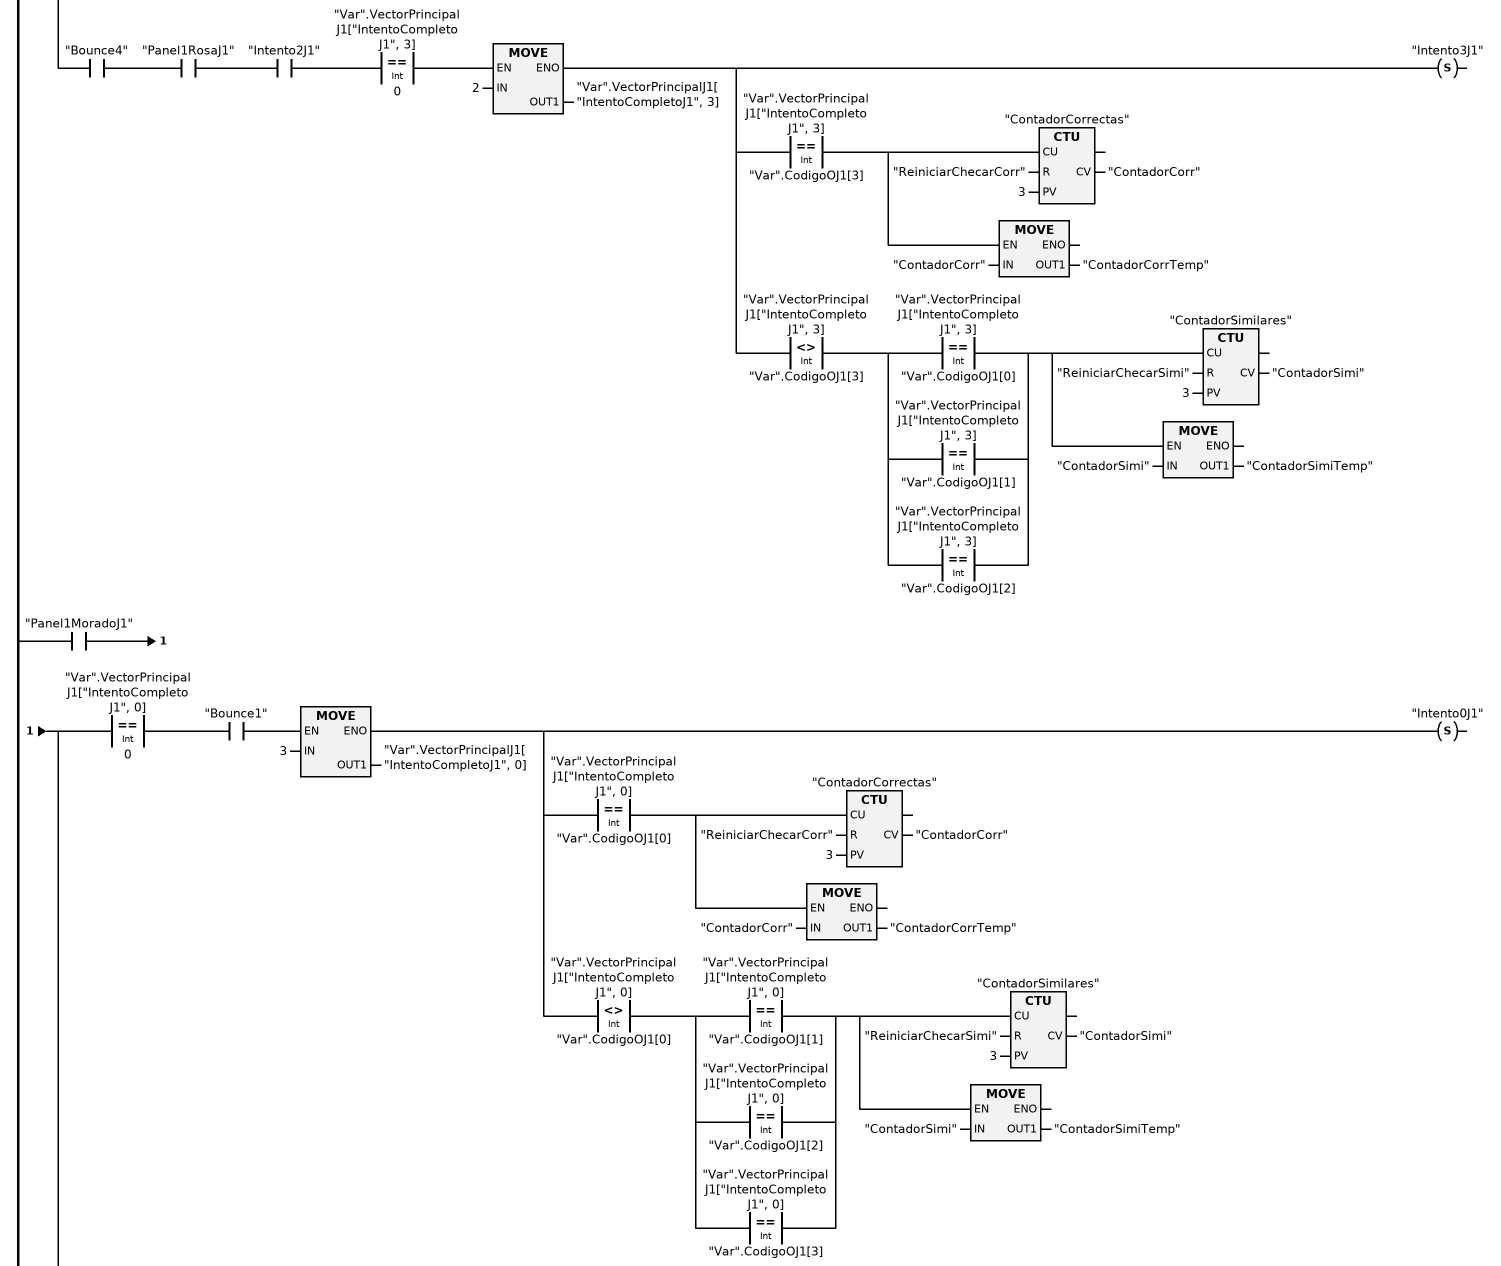
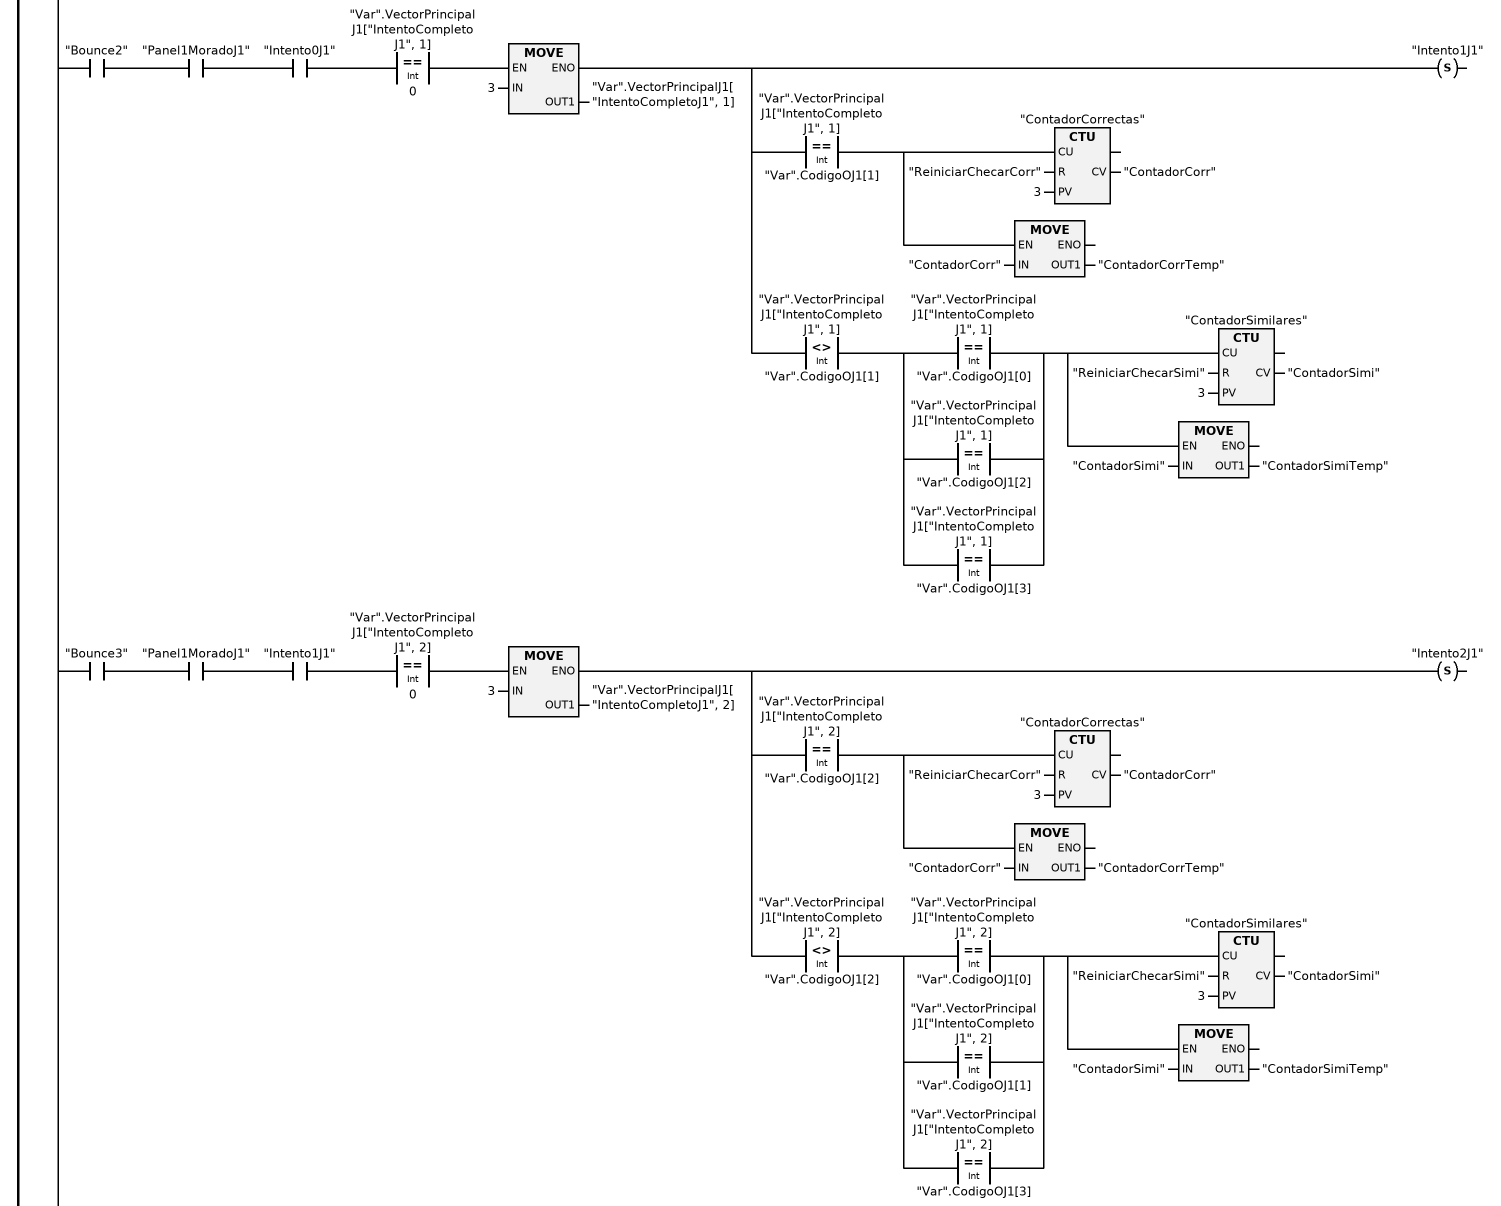
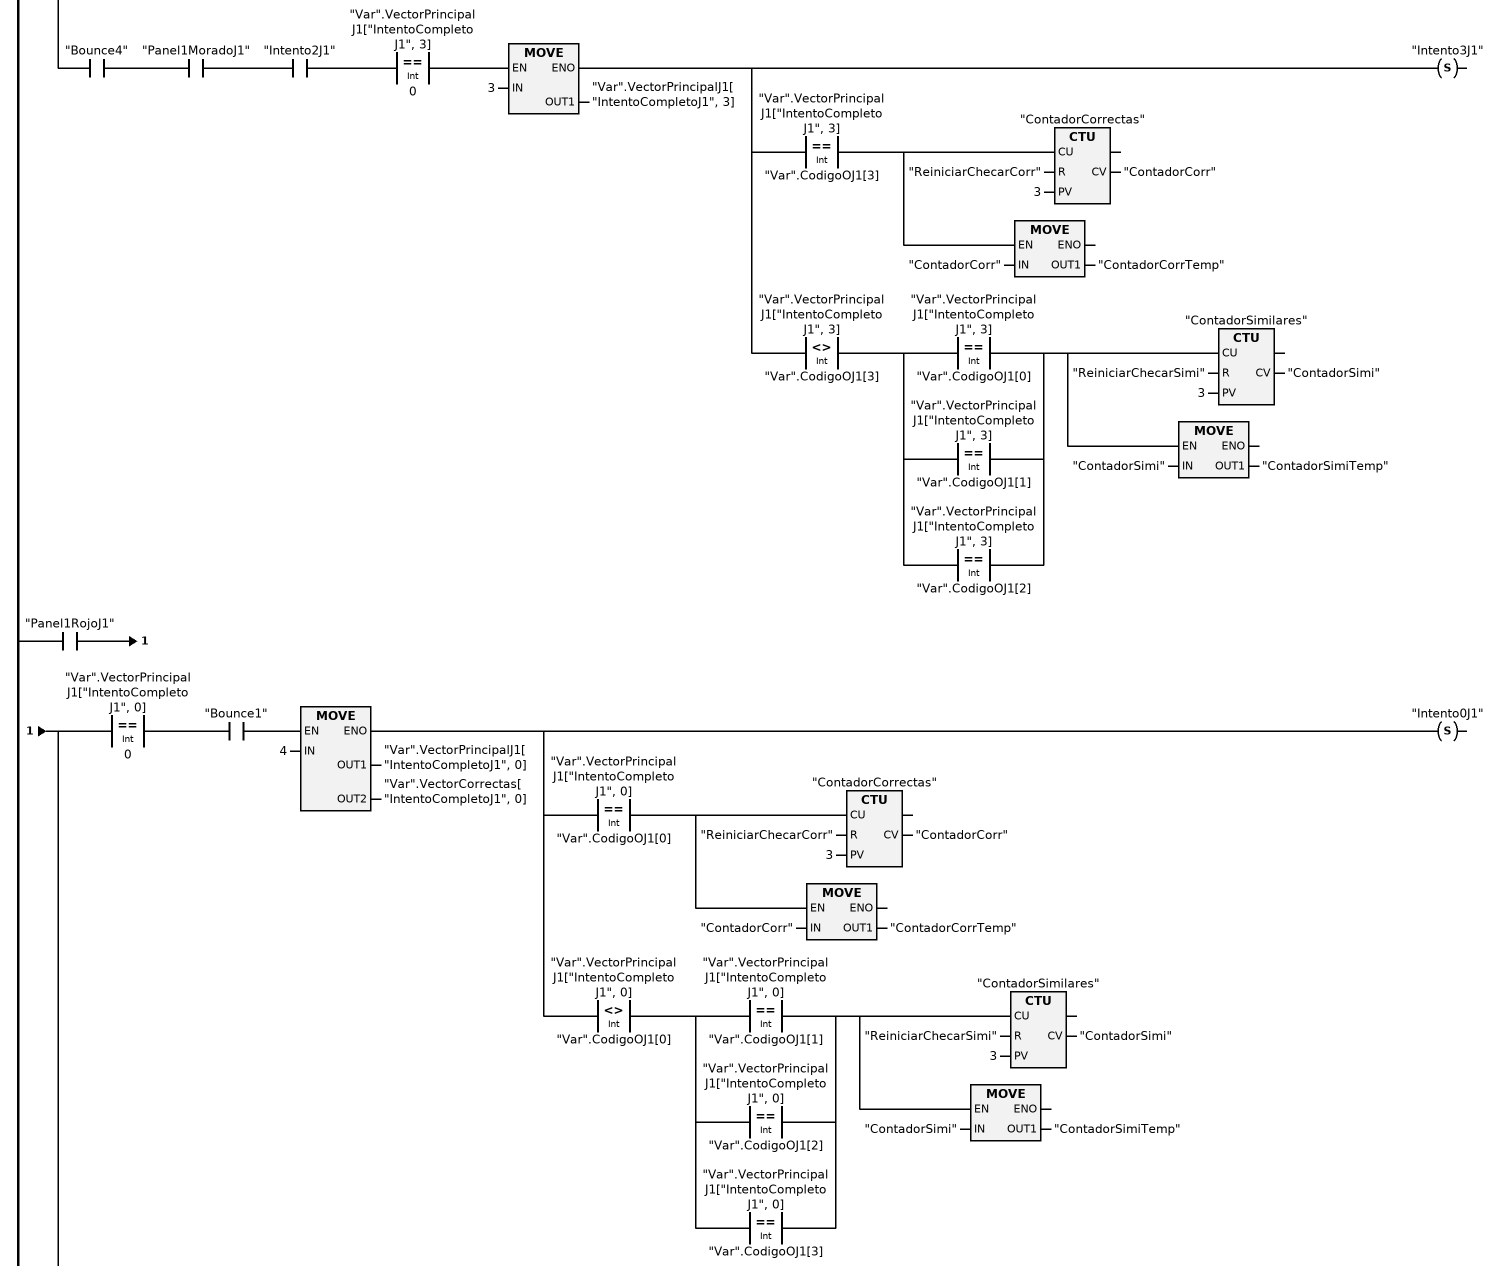
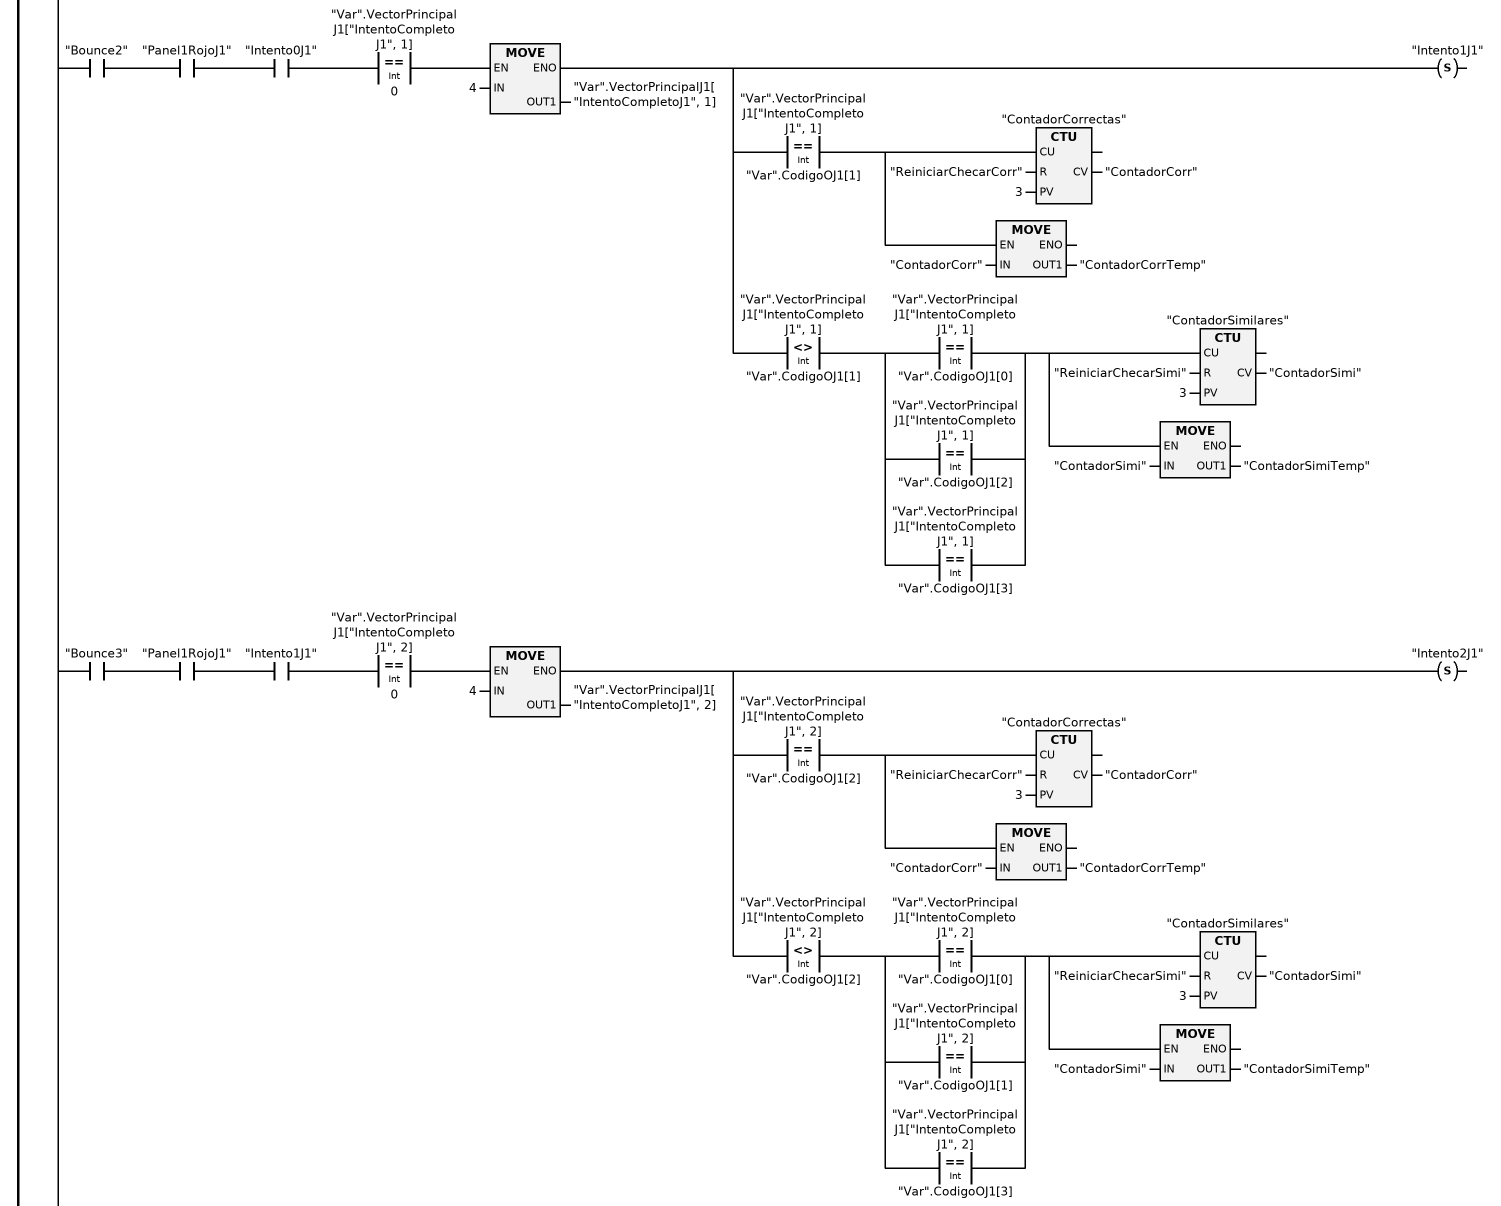
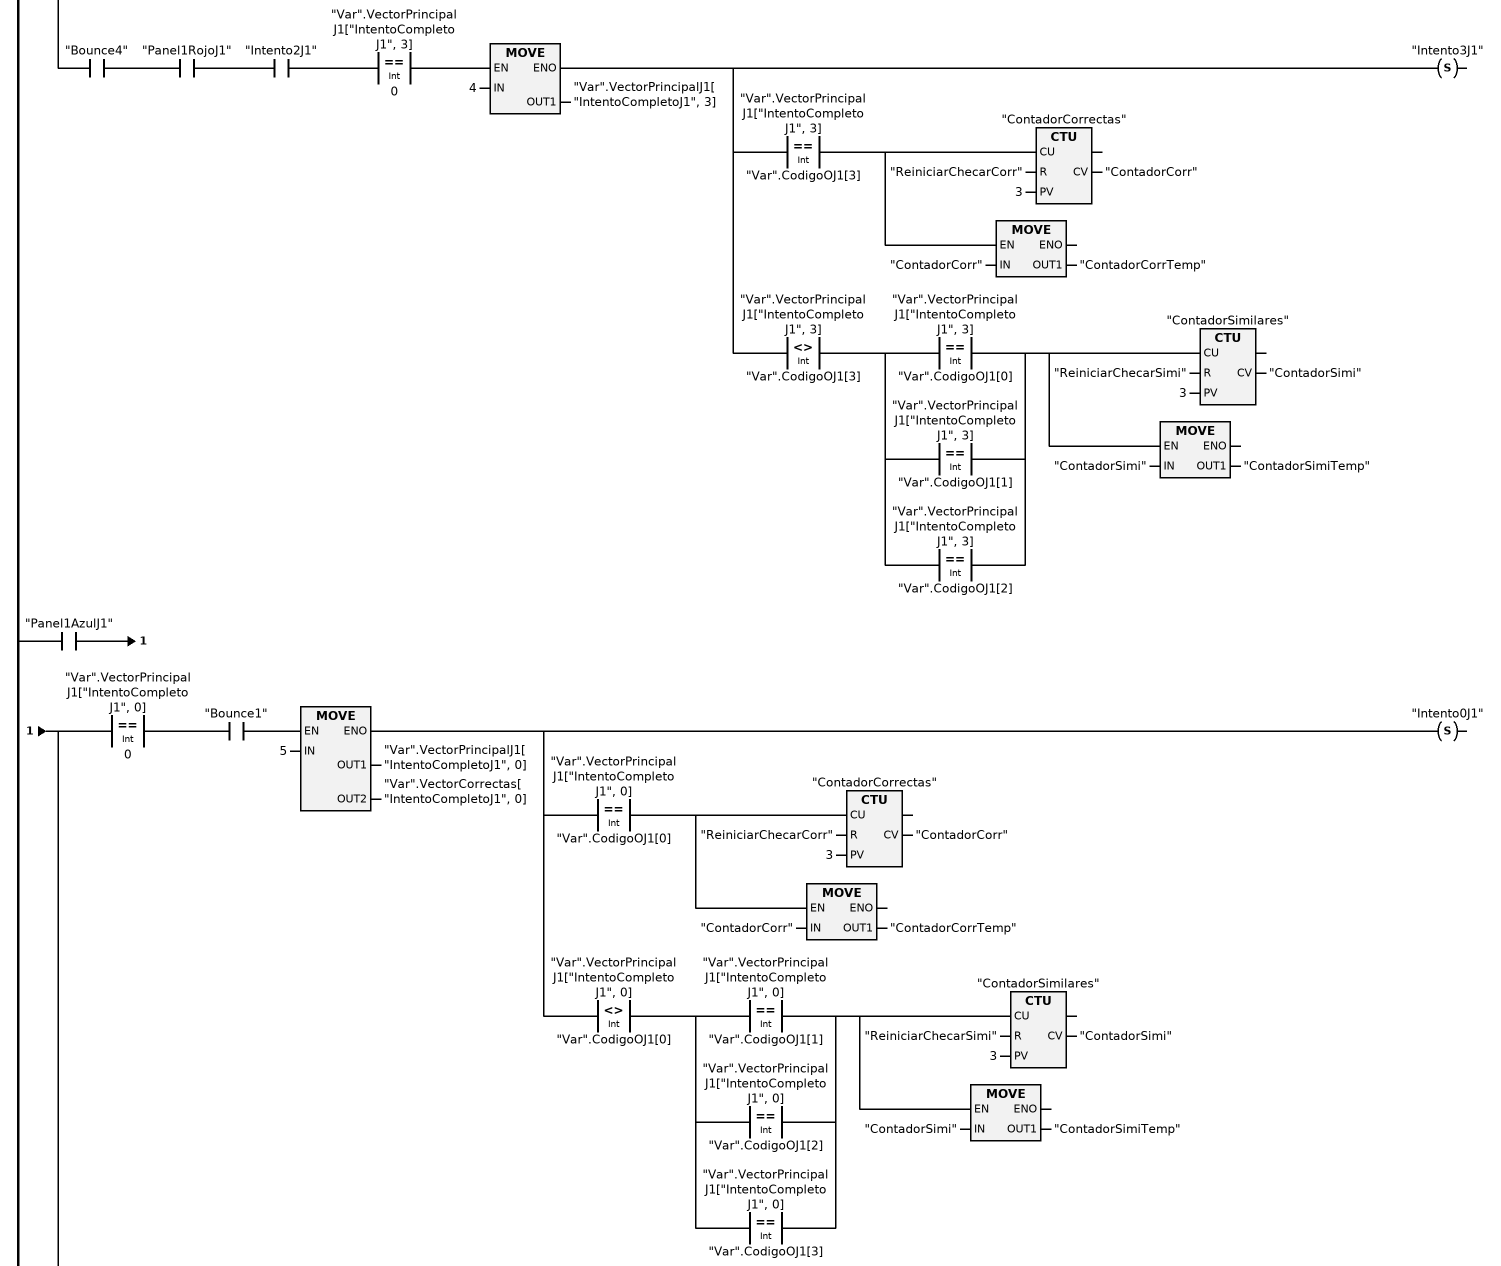
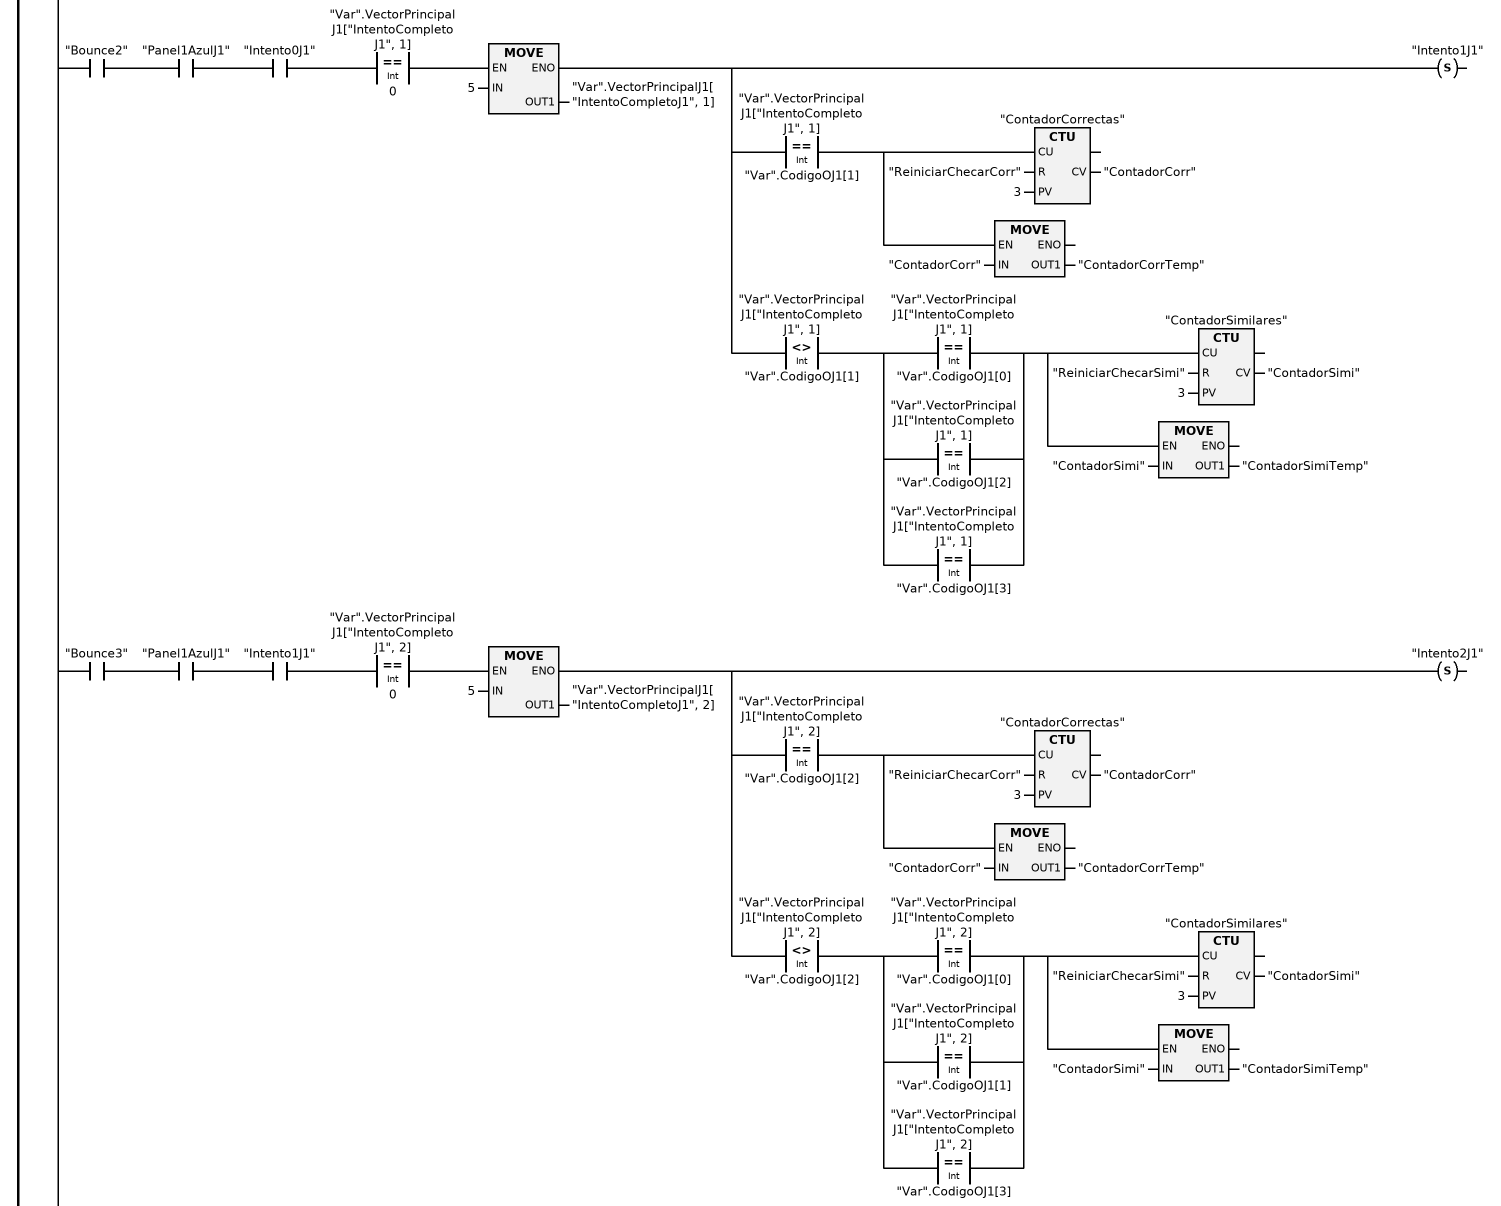
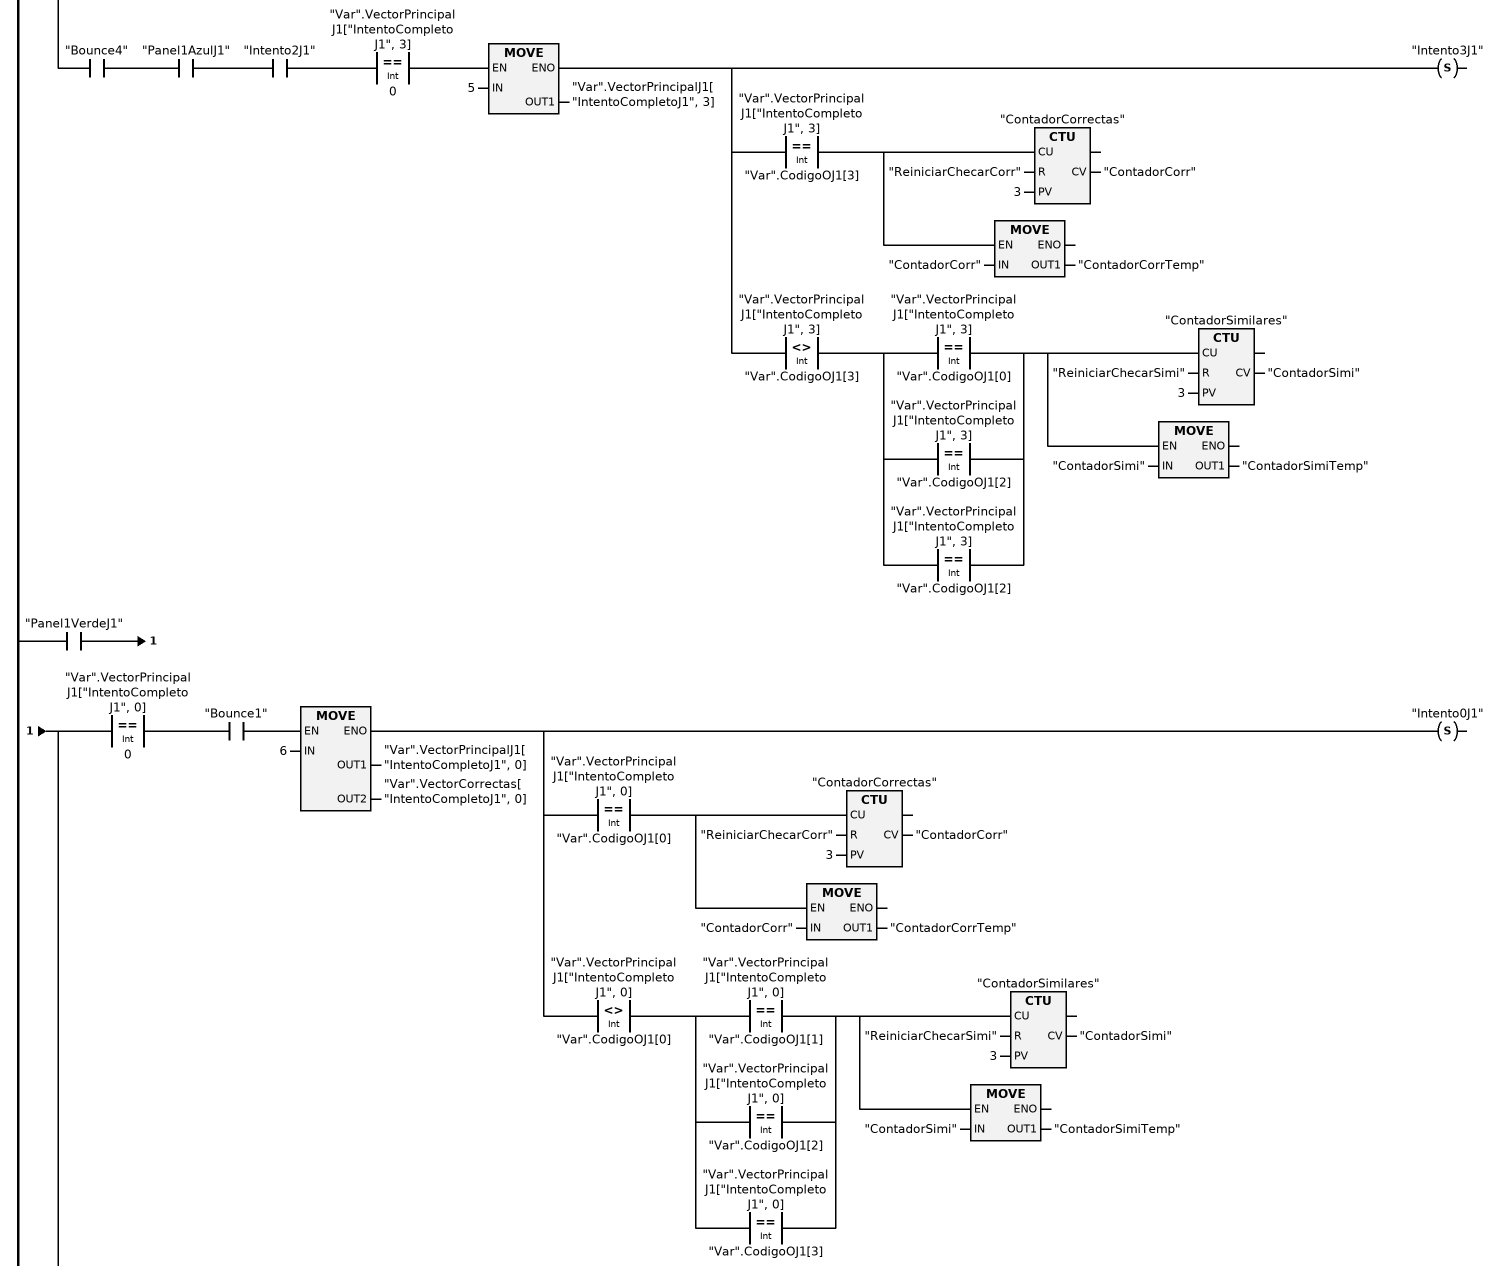
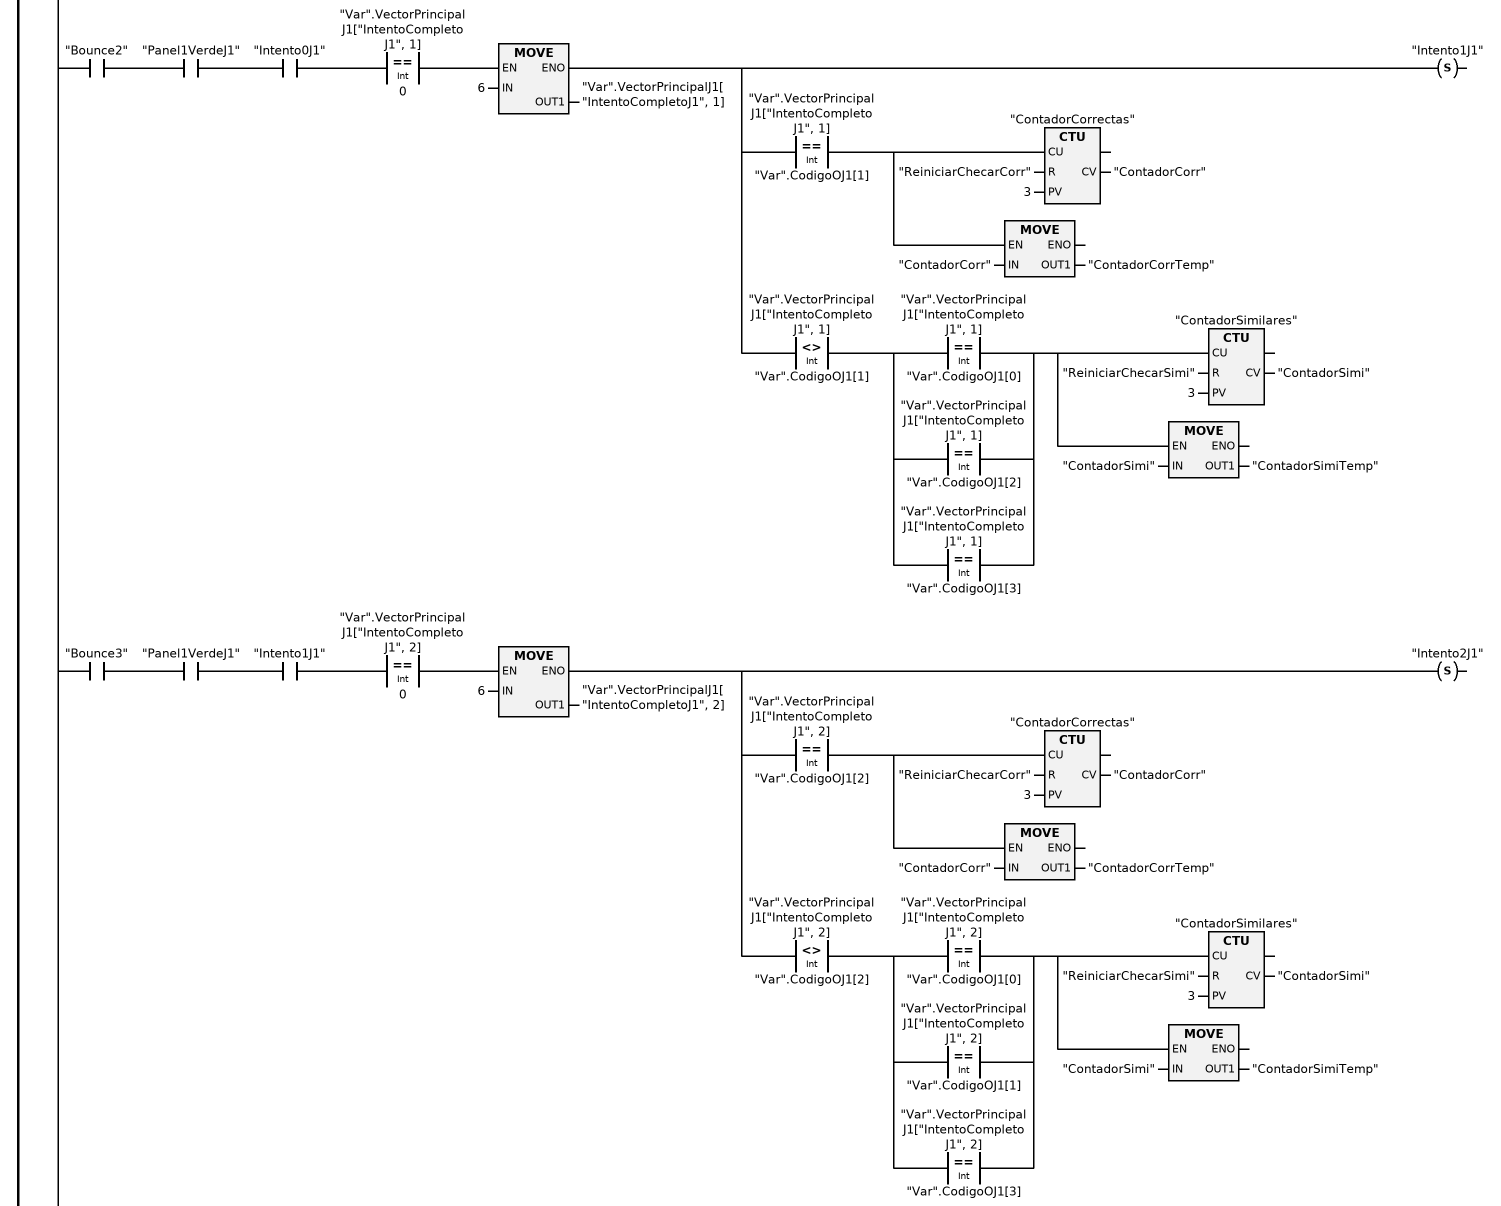
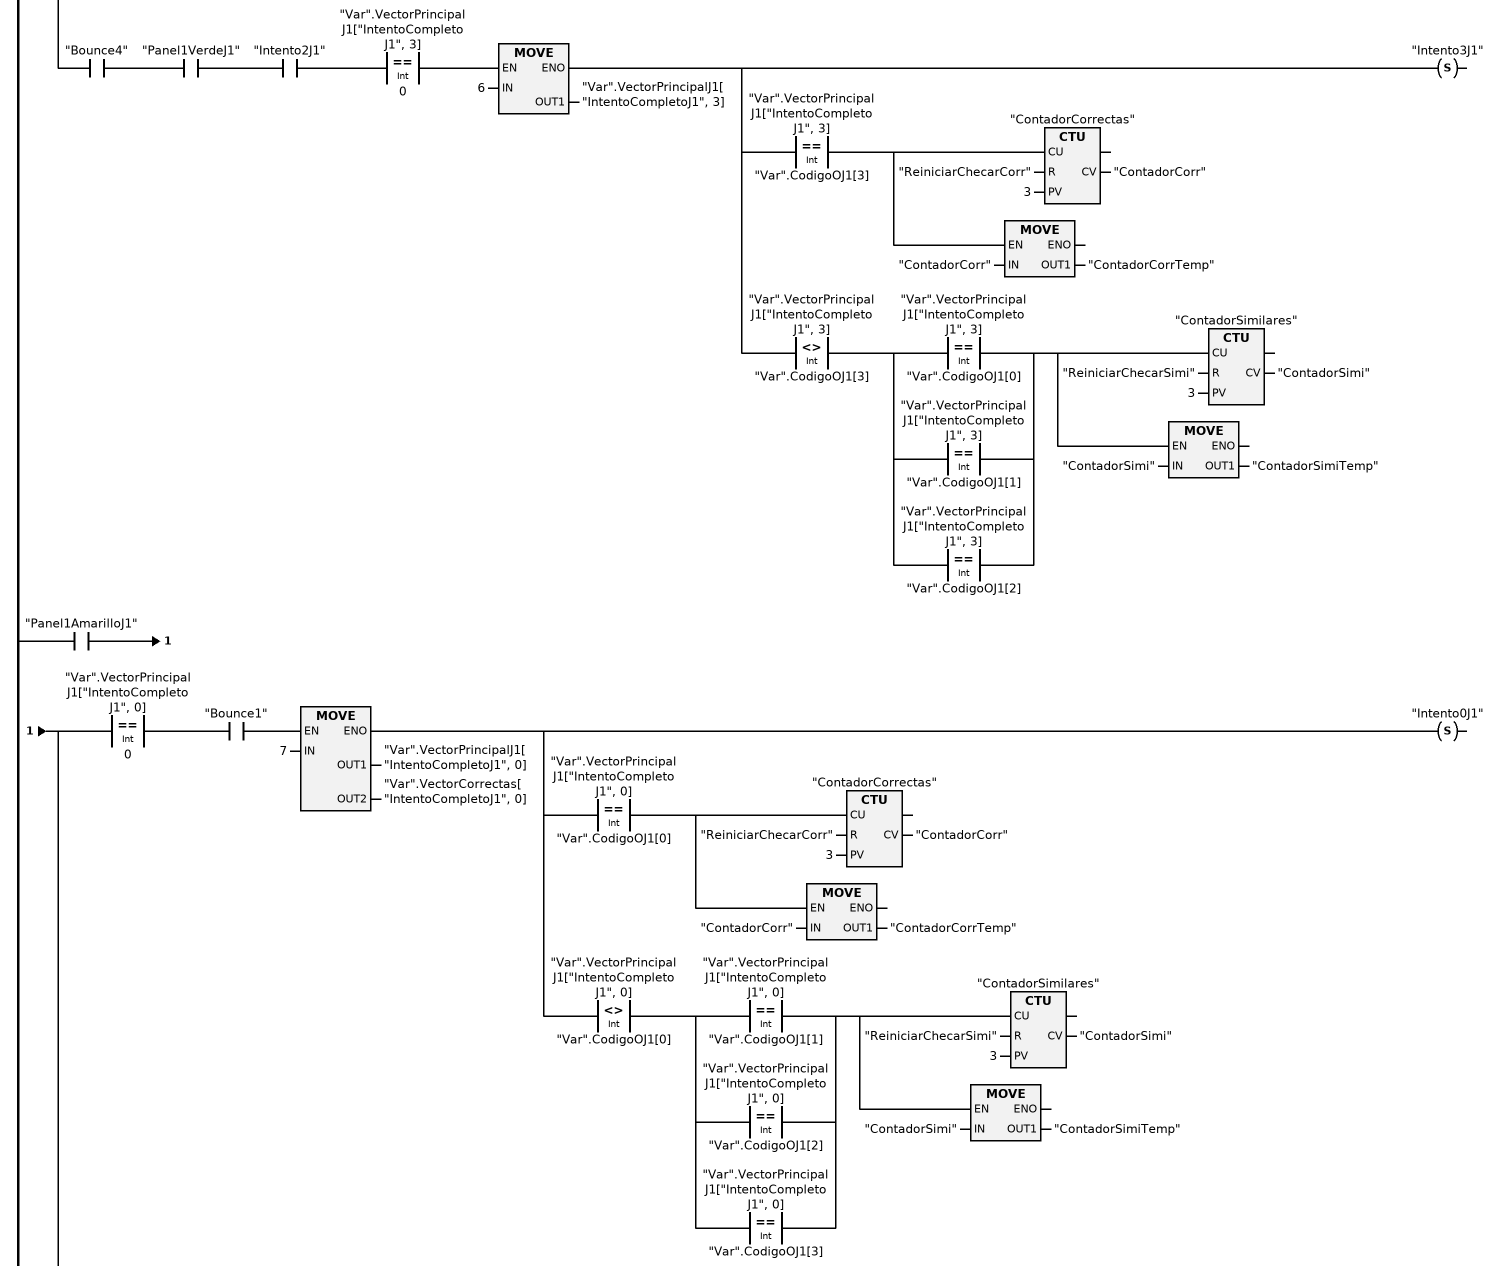
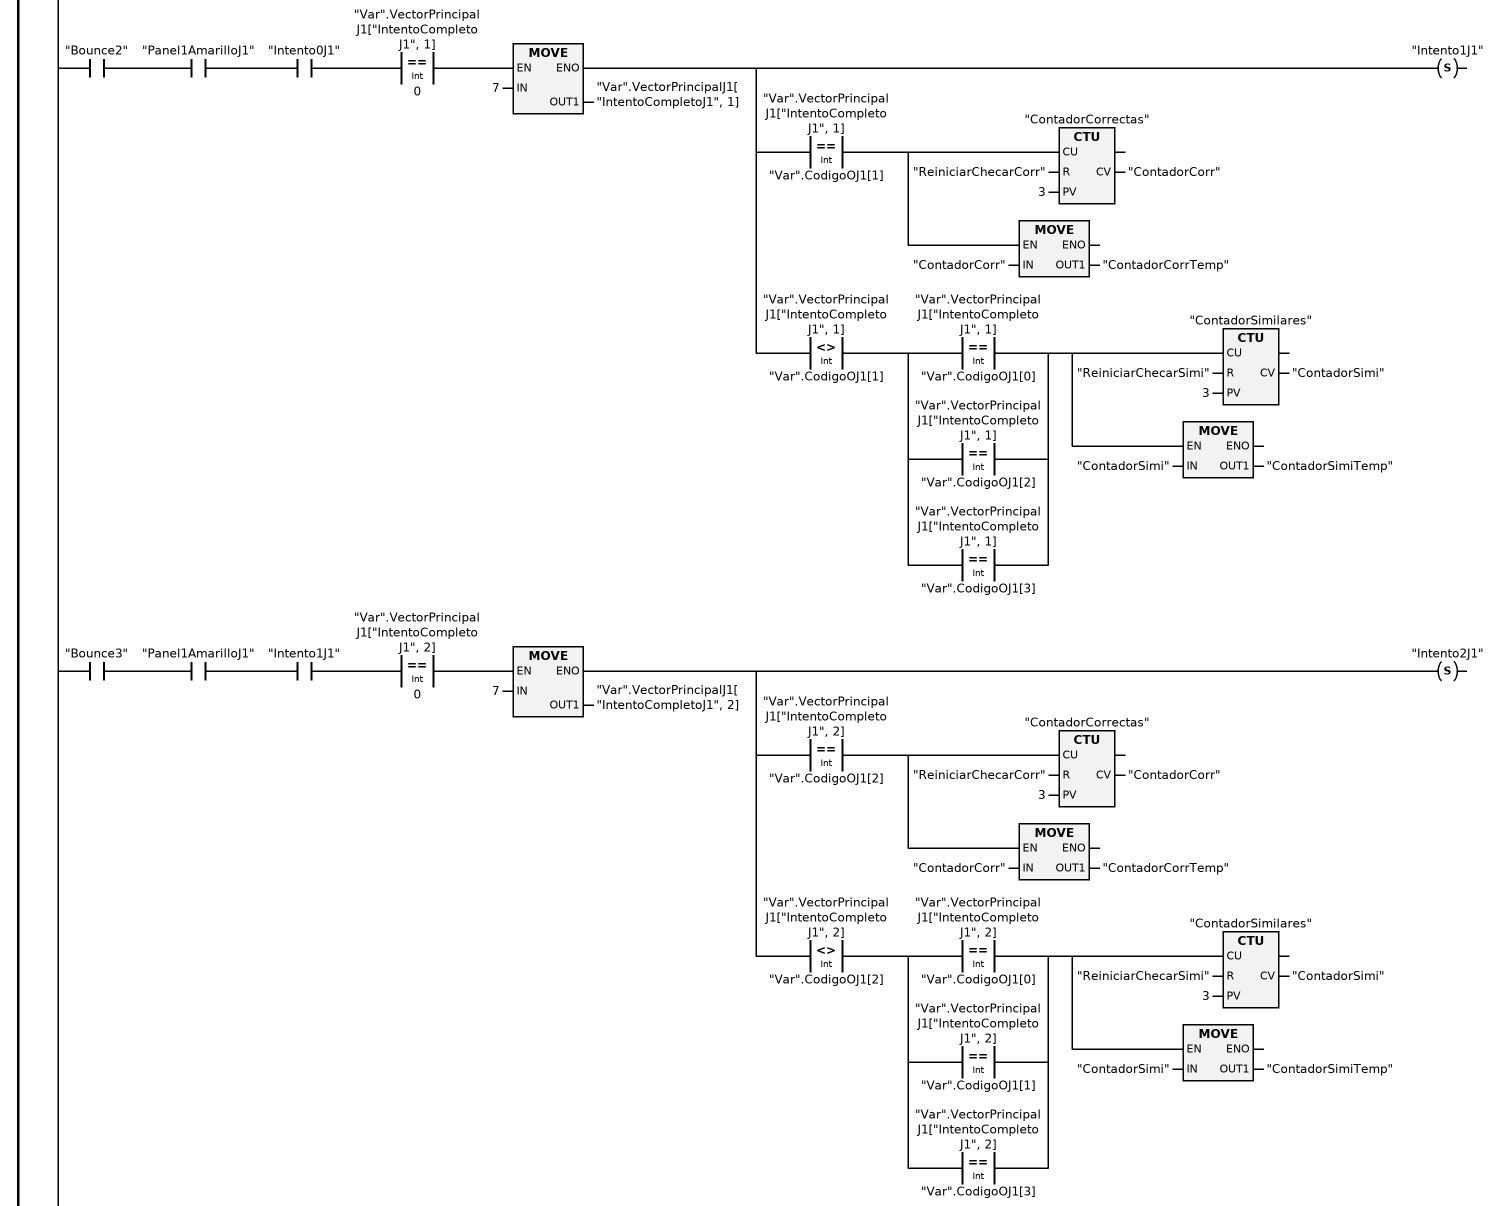
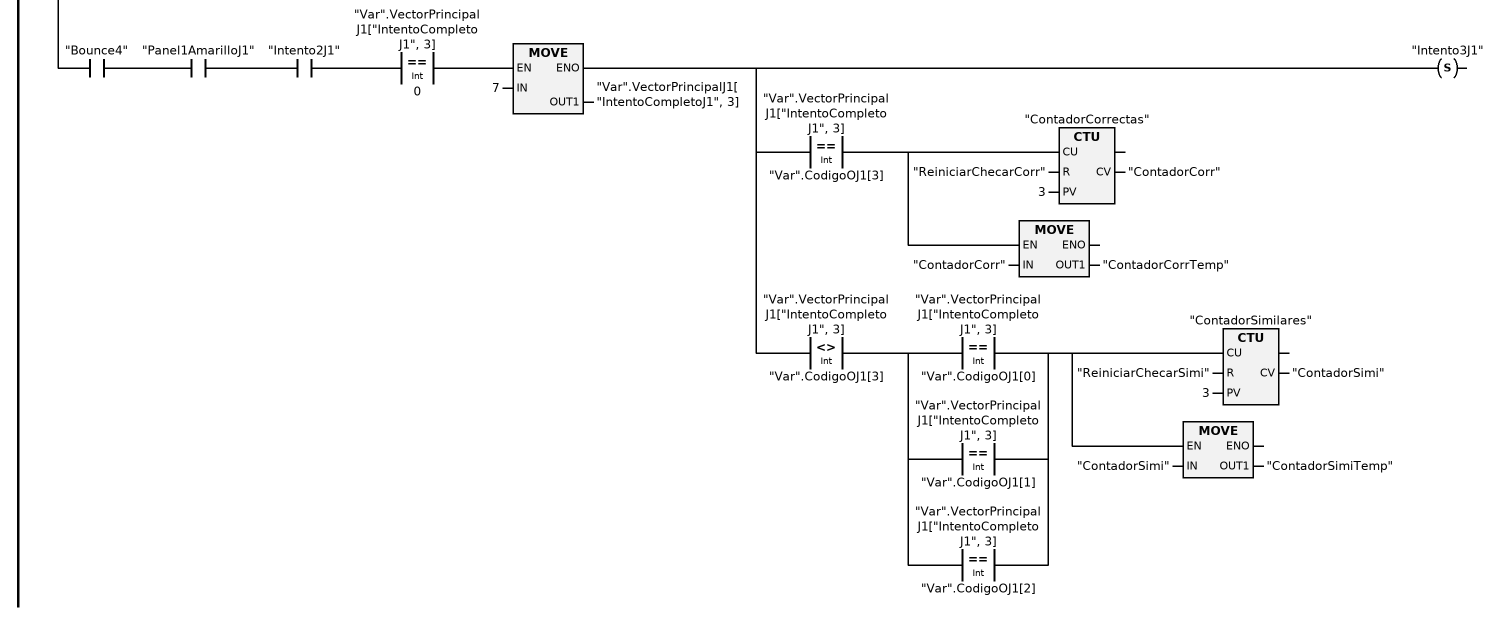
   // no SCL statement known for RBitfield: written as a call
   "IEC_Counter_0_DB_1".CTU(CU := "Intento3J1", R := "ReiniciarContadorJ1", PV := 10, CV => "IntentoCompletoJ1");
   "ReinicioCorrecto" := "IEC_Counter_0_DB_1".Q;
   #_w1 := "Intento3J1";
   IF #_w1 THEN
       RESET_BF(operand := "Bounce1", n := 10);
       RESET_BF(operand := "Intento0J1", n := 8);
   END_IF;
   "CorrectasSimilares" := #_w1;
   #_w2 := NOT "Panel2J1Activado" AND NOT "Panel1CafeJ1" AND NOT "Panel1RosaJ1" AND NOT "Panel1MoradoJ1" AND NOT "Panel1RojoJ1" AND NOT "Panel1AzulJ1" AND NOT "Panel1VerdeJ1" AND NOT "Panel1AmarilloJ1";
   IF #_w2 AND "Intento0J1" AND "Bounce5" AND NOT "Bounce2" AND NOT "Bounce3" AND NOT "Bounce4" THEN
       "Bounce2" := TRUE;
   END_IF;
   IF #_w2 AND "Intento1J1" AND "Bounce5" AND "Bounce2" AND NOT "Bounce3" AND NOT "Bounce4" THEN
       "Bounce3" := TRUE;
   END_IF;
   IF #_w2 AND "Intento2J1" AND "Bounce5" AND "Bounce2" AND "Bounce3" AND NOT "Bounce4" THEN
       "Bounce4" := TRUE;
   END_IF;
   IF #_w2 AND "Bounce5" THEN "Bounce1" := TRUE; END_IF;
   #_w3 := "Panel1CafeJ1" AND ("Var".VectorPrincipalJ1["IntentoCompletoJ1", 0] = 0) AND "Bounce1";
   IF #_w3 THEN
       "Var".VectorPrincipalJ1["IntentoCompletoJ1", 0] := 1;
       "Intento0J1" := TRUE;
   END_IF;
   #_w4 := #_w3 AND ("Var".VectorPrincipalJ1["IntentoCompletoJ1", 0] = "Var".CodigoOJ1[0]);
   "ContadorCorrectas".CTU(CU := #_w4, R := "ReiniciarChecarCorr", PV := 3, CV => "ContadorCorr");
   IF #_w4 THEN "ContadorCorrTemp" := "ContadorCorr"; END_IF;
   #_w5 := #_w3 AND ("Var".VectorPrincipalJ1["IntentoCompletoJ1", 0] <> "Var".CodigoOJ1[0]) AND ("Var".VectorPrincipalJ1["IntentoCompletoJ1", 0] = "Var".CodigoOJ1[1]);
   IF #_w5 THEN "Var".VectorCorrectas["IntentoCompletoJ1", 0] := 8; END_IF;
   "ContadorSimilares".CTU(CU := #_w5, R := "ReiniciarChecarSimi", PV := 3, CV => "ContadorSimi");
   IF #_w5 THEN "ContadorSimiTemp" := "ContadorSimi"; END_IF;
   #_w6 := #_w3 AND ("Var".VectorPrincipalJ1["IntentoCompletoJ1", 0] <> "Var".CodigoOJ1[0]) AND ("Var".VectorPrincipalJ1["IntentoCompletoJ1", 0] = "Var".CodigoOJ1[2]);
   IF #_w6 THEN "Var".VectorCorrectas["IntentoCompletoJ1", 0] := 8; END_IF;
   "ContadorSimilares".CTU(CU := #_w6, R := "ReiniciarChecarSimi", PV := 3, CV => "ContadorSimi");
   IF #_w6 THEN "ContadorSimiTemp" := "ContadorSimi"; END_IF;
   #_w7 := #_w3 AND ("Var".VectorPrincipalJ1["IntentoCompletoJ1", 0] <> "Var".CodigoOJ1[0]) AND ("Var".VectorPrincipalJ1["IntentoCompletoJ1", 0] = "Var".CodigoOJ1[3]);
   IF #_w7 THEN "Var".VectorCorrectas["IntentoCompletoJ1", 0] := 8; END_IF;
   "ContadorSimilares".CTU(CU := #_w7, R := "ReiniciarChecarSimi", PV := 3, CV => "ContadorSimi");
   IF #_w7 THEN "ContadorSimiTemp" := "ContadorSimi"; END_IF;
   #_w8 := "Panel1CafeJ1" AND "Bounce2" AND "Panel1CafeJ1" AND "Intento0J1" AND ("Var".VectorPrincipalJ1["IntentoCompletoJ1", 1] = 0);
   IF #_w8 THEN
       "Var".VectorPrincipalJ1["IntentoCompletoJ1", 1] := 1;
       "Intento1J1" := TRUE;
   END_IF;
   #_w9 := #_w8 AND ("Var".VectorPrincipalJ1["IntentoCompletoJ1", 1] = "Var".CodigoOJ1[1]);
   "ContadorCorrectas".CTU(CU := #_w9, R := "ReiniciarChecarCorr", PV := 3, CV => "ContadorCorr");
   IF #_w9 THEN "ContadorCorrTemp" := "ContadorCorr"; END_IF;
   #_w10 := #_w8 AND ("Var".VectorPrincipalJ1["IntentoCompletoJ1", 1] <> "Var".CodigoOJ1[1]) AND (("Var".VectorPrincipalJ1["IntentoCompletoJ1", 1] = "Var".CodigoOJ1[0]) OR ("Var".VectorPrincipalJ1["IntentoCompletoJ1", 1] = "Var".CodigoOJ1[2]) OR ("Var".VectorPrincipalJ1["IntentoCompletoJ1", 1] = "Var".CodigoOJ1[3]));
   "ContadorSimilares".CTU(CU := #_w10, R := "ReiniciarChecarSimi", PV := 3, CV => "ContadorSimi");
   IF #_w10 THEN "ContadorSimiTemp" := "ContadorSimi"; END_IF;
   #_w11 := "Panel1CafeJ1" AND "Bounce3" AND "Panel1CafeJ1" AND "Intento1J1" AND ("Var".VectorPrincipalJ1["IntentoCompletoJ1", 2] = 0);
   IF #_w11 THEN
       "Var".VectorPrincipalJ1["IntentoCompletoJ1", 2] := 1;
       "Intento2J1" := TRUE;
   END_IF;
   #_w12 := #_w11 AND ("Var".VectorPrincipalJ1["IntentoCompletoJ1", 2] = "Var".CodigoOJ1[2]);
   "ContadorCorrectas".CTU(CU := #_w12, R := "ReiniciarChecarCorr", PV := 3, CV => "ContadorCorr");
   IF #_w12 THEN "ContadorCorrTemp" := "ContadorCorr"; END_IF;
   #_w13 := #_w11 AND ("Var".VectorPrincipalJ1["IntentoCompletoJ1", 2] <> "Var".CodigoOJ1[2]) AND (("Var".VectorPrincipalJ1["IntentoCompletoJ1", 2] = "Var".CodigoOJ1[0]) OR ("Var".VectorPrincipalJ1["IntentoCompletoJ1", 2] = "Var".CodigoOJ1[1]) OR ("Var".VectorPrincipalJ1["IntentoCompletoJ1", 2] = "Var".CodigoOJ1[3]));
   "ContadorSimilares".CTU(CU := #_w13, R := "ReiniciarChecarSimi", PV := 3, CV => "ContadorSimi");
   IF #_w13 THEN "ContadorSimiTemp" := "ContadorSimi"; END_IF;
   #_w14 := "Panel1CafeJ1" AND "Bounce4" AND "Panel1CafeJ1" AND "Intento2J1" AND ("Var".VectorPrincipalJ1["IntentoCompletoJ1", 3] = 0);
   IF #_w14 THEN
       "Var".VectorPrincipalJ1["IntentoCompletoJ1", 3] := 1;
       "Intento3J1" := TRUE;
   END_IF;
   #_w15 := #_w14 AND ("Var".VectorPrincipalJ1["IntentoCompletoJ1", 3] = "Var".CodigoOJ1[3]);
   "ContadorCorrectas".CTU(CU := #_w15, R := "ReiniciarChecarCorr", PV := 3, CV => "ContadorCorr");
   IF #_w15 THEN "ContadorCorrTemp" := "ContadorCorr"; END_IF;
   #_w16 := #_w14 AND ("Var".VectorPrincipalJ1["IntentoCompletoJ1", 3] <> "Var".CodigoOJ1[3]) AND (("Var".VectorPrincipalJ1["IntentoCompletoJ1", 3] = "Var".CodigoOJ1[0]) OR ("Var".VectorPrincipalJ1["IntentoCompletoJ1", 3] = "Var".CodigoOJ1[1]) OR ("Var".VectorPrincipalJ1["IntentoCompletoJ1", 3] = "Var".CodigoOJ1[2]));
   "ContadorSimilares".CTU(CU := #_w16, R := "ReiniciarChecarSimi", PV := 3, CV => "ContadorSimi");
   IF #_w16 THEN "ContadorSimiTemp" := "ContadorSimi"; END_IF;
   #_w17 := "Panel1RosaJ1" AND ("Var".VectorPrincipalJ1["IntentoCompletoJ1", 0] = 0) AND "Bounce1";
   IF #_w17 THEN
       "Var".VectorPrincipalJ1["IntentoCompletoJ1", 0] := 2;
       "Var".VectorCorrectas["IntentoCompletoJ1", 0] := 2;
       "Intento0J1" := TRUE;
   END_IF;
   #_w18 := #_w17 AND ("Var".VectorPrincipalJ1["IntentoCompletoJ1", 0] = "Var".CodigoOJ1[0]);
   "ContadorCorrectas".CTU(CU := #_w18, R := "ReiniciarChecarCorr", PV := 3, CV => "ContadorCorr");
   IF #_w18 THEN "ContadorCorrTemp" := "ContadorCorr"; END_IF;
   #_w19 := #_w17 AND ("Var".VectorPrincipalJ1["IntentoCompletoJ1", 0] <> "Var".CodigoOJ1[0]) AND (("Var".VectorPrincipalJ1["IntentoCompletoJ1", 0] = "Var".CodigoOJ1[1]) OR ("Var".VectorPrincipalJ1["IntentoCompletoJ1", 0] = "Var".CodigoOJ1[2]) OR ("Var".VectorPrincipalJ1["IntentoCompletoJ1", 0] = "Var".CodigoOJ1[3]));
   "ContadorSimilares".CTU(CU := #_w19, R := "ReiniciarChecarSimi", PV := 3, CV => "ContadorSimi");
   IF #_w19 THEN "ContadorSimiTemp" := "ContadorSimi"; END_IF;
   #_w20 := "Panel1RosaJ1" AND "Bounce2" AND "Panel1RosaJ1" AND "Intento0J1" AND ("Var".VectorPrincipalJ1["IntentoCompletoJ1", 1] = 0);
   IF #_w20 THEN
       "Var".VectorPrincipalJ1["IntentoCompletoJ1", 1] := 2;
       "Intento1J1" := TRUE;
   END_IF;
   #_w21 := #_w20 AND ("Var".VectorPrincipalJ1["IntentoCompletoJ1", 1] = "Var".CodigoOJ1[1]);
   "ContadorCorrectas".CTU(CU := #_w21, R := "ReiniciarChecarCorr", PV := 3, CV => "ContadorCorr");
   IF #_w21 THEN "ContadorCorrTemp" := "ContadorCorr"; END_IF;
   #_w22 := #_w20 AND ("Var".VectorPrincipalJ1["IntentoCompletoJ1", 1] <> "Var".CodigoOJ1[1]) AND (("Var".VectorPrincipalJ1["IntentoCompletoJ1", 1] = "Var".CodigoOJ1[0]) OR ("Var".VectorPrincipalJ1["IntentoCompletoJ1", 1] = "Var".CodigoOJ1[2]) OR ("Var".VectorPrincipalJ1["IntentoCompletoJ1", 1] = "Var".CodigoOJ1[3]));
   "ContadorSimilares".CTU(CU := #_w22, R := "ReiniciarChecarSimi", PV := 3, CV => "ContadorSimi");
   IF #_w22 THEN "ContadorSimiTemp" := "ContadorSimi"; END_IF;
   #_w23 := "Panel1RosaJ1" AND "Bounce3" AND "Panel1RosaJ1" AND "Intento1J1" AND ("Var".VectorPrincipalJ1["IntentoCompletoJ1", 2] = 0);
   IF #_w23 THEN
       "Var".VectorPrincipalJ1["IntentoCompletoJ1", 2] := 2;
       "Intento2J1" := TRUE;
   END_IF;
   #_w24 := #_w23 AND ("Var".VectorPrincipalJ1["IntentoCompletoJ1", 2] = "Var".CodigoOJ1[2]);
   "ContadorCorrectas".CTU(CU := #_w24, R := "ReiniciarChecarCorr", PV := 3, CV => "ContadorCorr");
   IF #_w24 THEN "ContadorCorrTemp" := "ContadorCorr"; END_IF;
   #_w25 := #_w23 AND ("Var".VectorPrincipalJ1["IntentoCompletoJ1", 2] <> "Var".CodigoOJ1[2]) AND (("Var".VectorPrincipalJ1["IntentoCompletoJ1", 2] = "Var".CodigoOJ1[0]) OR ("Var".VectorPrincipalJ1["IntentoCompletoJ1", 2] = "Var".CodigoOJ1[1]) OR ("Var".VectorPrincipalJ1["IntentoCompletoJ1", 2] = "Var".CodigoOJ1[3]));
   "ContadorSimilares".CTU(CU := #_w25, R := "ReiniciarChecarSimi", PV := 3, CV => "ContadorSimi");
   IF #_w25 THEN "ContadorSimiTemp" := "ContadorSimi"; END_IF;
   #_w26 := "Panel1RosaJ1" AND "Bounce4" AND "Panel1RosaJ1" AND "Intento2J1" AND ("Var".VectorPrincipalJ1["IntentoCompletoJ1", 3] = 0);
   IF #_w26 THEN
       "Var".VectorPrincipalJ1["IntentoCompletoJ1", 3] := 2;
       "Intento3J1" := TRUE;
   END_IF;
   #_w27 := #_w26 AND ("Var".VectorPrincipalJ1["IntentoCompletoJ1", 3] = "Var".CodigoOJ1[3]);
   "ContadorCorrectas".CTU(CU := #_w27, R := "ReiniciarChecarCorr", PV := 3, CV => "ContadorCorr");
   IF #_w27 THEN "ContadorCorrTemp" := "ContadorCorr"; END_IF;
   #_w28 := #_w26 AND ("Var".VectorPrincipalJ1["IntentoCompletoJ1", 3] <> "Var".CodigoOJ1[3]) AND (("Var".VectorPrincipalJ1["IntentoCompletoJ1", 3] = "Var".CodigoOJ1[0]) OR ("Var".VectorPrincipalJ1["IntentoCompletoJ1", 3] = "Var".CodigoOJ1[1]) OR ("Var".VectorPrincipalJ1["IntentoCompletoJ1", 3] = "Var".CodigoOJ1[2]));
   "ContadorSimilares".CTU(CU := #_w28, R := "ReiniciarChecarSimi", PV := 3, CV => "ContadorSimi");
   IF #_w28 THEN "ContadorSimiTemp" := "ContadorSimi"; END_IF;
   #_w29 := "Panel1MoradoJ1" AND ("Var".VectorPrincipalJ1["IntentoCompletoJ1", 0] = 0) AND "Bounce1";
   IF #_w29 THEN
       "Var".VectorPrincipalJ1["IntentoCompletoJ1", 0] := 3;
       "Intento0J1" := TRUE;
   END_IF;
   #_w30 := #_w29 AND ("Var".VectorPrincipalJ1["IntentoCompletoJ1", 0] = "Var".CodigoOJ1[0]);
   "ContadorCorrectas".CTU(CU := #_w30, R := "ReiniciarChecarCorr", PV := 3, CV => "ContadorCorr");
   IF #_w30 THEN "ContadorCorrTemp" := "ContadorCorr"; END_IF;
   #_w31 := #_w29 AND ("Var".VectorPrincipalJ1["IntentoCompletoJ1", 0] <> "Var".CodigoOJ1[0]) AND (("Var".VectorPrincipalJ1["IntentoCompletoJ1", 0] = "Var".CodigoOJ1[1]) OR ("Var".VectorPrincipalJ1["IntentoCompletoJ1", 0] = "Var".CodigoOJ1[2]) OR ("Var".VectorPrincipalJ1["IntentoCompletoJ1", 0] = "Var".CodigoOJ1[3]));
   "ContadorSimilares".CTU(CU := #_w31, R := "ReiniciarChecarSimi", PV := 3, CV => "ContadorSimi");
   IF #_w31 THEN "ContadorSimiTemp" := "ContadorSimi"; END_IF;
   #_w32 := "Panel1MoradoJ1" AND "Bounce2" AND "Panel1MoradoJ1" AND "Intento0J1" AND ("Var".VectorPrincipalJ1["IntentoCompletoJ1", 1] = 0);
   IF #_w32 THEN
       "Var".VectorPrincipalJ1["IntentoCompletoJ1", 1] := 3;
       "Intento1J1" := TRUE;
   END_IF;
   #_w33 := #_w32 AND ("Var".VectorPrincipalJ1["IntentoCompletoJ1", 1] = "Var".CodigoOJ1[1]);
   "ContadorCorrectas".CTU(CU := #_w33, R := "ReiniciarChecarCorr", PV := 3, CV => "ContadorCorr");
   IF #_w33 THEN "ContadorCorrTemp" := "ContadorCorr"; END_IF;
   #_w34 := #_w32 AND ("Var".VectorPrincipalJ1["IntentoCompletoJ1", 1] <> "Var".CodigoOJ1[1]) AND (("Var".VectorPrincipalJ1["IntentoCompletoJ1", 1] = "Var".CodigoOJ1[0]) OR ("Var".VectorPrincipalJ1["IntentoCompletoJ1", 1] = "Var".CodigoOJ1[2]) OR ("Var".VectorPrincipalJ1["IntentoCompletoJ1", 1] = "Var".CodigoOJ1[3]));
   "ContadorSimilares".CTU(CU := #_w34, R := "ReiniciarChecarSimi", PV := 3, CV => "ContadorSimi");
   IF #_w34 THEN "ContadorSimiTemp" := "ContadorSimi"; END_IF;
   #_w35 := "Panel1MoradoJ1" AND "Bounce3" AND "Panel1MoradoJ1" AND "Intento1J1" AND ("Var".VectorPrincipalJ1["IntentoCompletoJ1", 2] = 0);
   IF #_w35 THEN
       "Var".VectorPrincipalJ1["IntentoCompletoJ1", 2] := 3;
       "Intento2J1" := TRUE;
   END_IF;
   #_w36 := #_w35 AND ("Var".VectorPrincipalJ1["IntentoCompletoJ1", 2] = "Var".CodigoOJ1[2]);
   "ContadorCorrectas".CTU(CU := #_w36, R := "ReiniciarChecarCorr", PV := 3, CV => "ContadorCorr");
   IF #_w36 THEN "ContadorCorrTemp" := "ContadorCorr"; END_IF;
   #_w37 := #_w35 AND ("Var".VectorPrincipalJ1["IntentoCompletoJ1", 2] <> "Var".CodigoOJ1[2]) AND (("Var".VectorPrincipalJ1["IntentoCompletoJ1", 2] = "Var".CodigoOJ1[0]) OR ("Var".VectorPrincipalJ1["IntentoCompletoJ1", 2] = "Var".CodigoOJ1[1]) OR ("Var".VectorPrincipalJ1["IntentoCompletoJ1", 2] = "Var".CodigoOJ1[3]));
   "ContadorSimilares".CTU(CU := #_w37, R := "ReiniciarChecarSimi", PV := 3, CV => "ContadorSimi");
   IF #_w37 THEN "ContadorSimiTemp" := "ContadorSimi"; END_IF;
   #_w38 := "Panel1MoradoJ1" AND "Bounce4" AND "Panel1MoradoJ1" AND "Intento2J1" AND ("Var".VectorPrincipalJ1["IntentoCompletoJ1", 3] = 0);
   IF #_w38 THEN
       "Var".VectorPrincipalJ1["IntentoCompletoJ1", 3] := 3;
       "Intento3J1" := TRUE;
   END_IF;
   #_w39 := #_w38 AND ("Var".VectorPrincipalJ1["IntentoCompletoJ1", 3] = "Var".CodigoOJ1[3]);
   "ContadorCorrectas".CTU(CU := #_w39, R := "ReiniciarChecarCorr", PV := 3, CV => "ContadorCorr");
   IF #_w39 THEN "ContadorCorrTemp" := "ContadorCorr"; END_IF;
   #_w40 := #_w38 AND ("Var".VectorPrincipalJ1["IntentoCompletoJ1", 3] <> "Var".CodigoOJ1[3]) AND (("Var".VectorPrincipalJ1["IntentoCompletoJ1", 3] = "Var".CodigoOJ1[0]) OR ("Var".VectorPrincipalJ1["IntentoCompletoJ1", 3] = "Var".CodigoOJ1[1]) OR ("Var".VectorPrincipalJ1["IntentoCompletoJ1", 3] = "Var".CodigoOJ1[2]));
   "ContadorSimilares".CTU(CU := #_w40, R := "ReiniciarChecarSimi", PV := 3, CV => "ContadorSimi");
   IF #_w40 THEN "ContadorSimiTemp" := "ContadorSimi"; END_IF;
   #_w41 := "Panel1RojoJ1" AND ("Var".VectorPrincipalJ1["IntentoCompletoJ1", 0] = 0) AND "Bounce1";
   IF #_w41 THEN
       "Var".VectorPrincipalJ1["IntentoCompletoJ1", 0] := 4;
       "Var".VectorCorrectas["IntentoCompletoJ1", 0] := 4;
       "Intento0J1" := TRUE;
   END_IF;
   #_w42 := #_w41 AND ("Var".VectorPrincipalJ1["IntentoCompletoJ1", 0] = "Var".CodigoOJ1[0]);
   "ContadorCorrectas".CTU(CU := #_w42, R := "ReiniciarChecarCorr", PV := 3, CV => "ContadorCorr");
   IF #_w42 THEN "ContadorCorrTemp" := "ContadorCorr"; END_IF;
   #_w43 := #_w41 AND ("Var".VectorPrincipalJ1["IntentoCompletoJ1", 0] <> "Var".CodigoOJ1[0]) AND (("Var".VectorPrincipalJ1["IntentoCompletoJ1", 0] = "Var".CodigoOJ1[1]) OR ("Var".VectorPrincipalJ1["IntentoCompletoJ1", 0] = "Var".CodigoOJ1[2]) OR ("Var".VectorPrincipalJ1["IntentoCompletoJ1", 0] = "Var".CodigoOJ1[3]));
   "ContadorSimilares".CTU(CU := #_w43, R := "ReiniciarChecarSimi", PV := 3, CV => "ContadorSimi");
   IF #_w43 THEN "ContadorSimiTemp" := "ContadorSimi"; END_IF;
   #_w44 := "Panel1RojoJ1" AND "Bounce2" AND "Panel1RojoJ1" AND "Intento0J1" AND ("Var".VectorPrincipalJ1["IntentoCompletoJ1", 1] = 0);
   IF #_w44 THEN
       "Var".VectorPrincipalJ1["IntentoCompletoJ1", 1] := 4;
       "Intento1J1" := TRUE;
   END_IF;
   #_w45 := #_w44 AND ("Var".VectorPrincipalJ1["IntentoCompletoJ1", 1] = "Var".CodigoOJ1[1]);
   "ContadorCorrectas".CTU(CU := #_w45, R := "ReiniciarChecarCorr", PV := 3, CV => "ContadorCorr");
   IF #_w45 THEN "ContadorCorrTemp" := "ContadorCorr"; END_IF;
   #_w46 := #_w44 AND ("Var".VectorPrincipalJ1["IntentoCompletoJ1", 1] <> "Var".CodigoOJ1[1]) AND (("Var".VectorPrincipalJ1["IntentoCompletoJ1", 1] = "Var".CodigoOJ1[0]) OR ("Var".VectorPrincipalJ1["IntentoCompletoJ1", 1] = "Var".CodigoOJ1[2]) OR ("Var".VectorPrincipalJ1["IntentoCompletoJ1", 1] = "Var".CodigoOJ1[3]));
   "ContadorSimilares".CTU(CU := #_w46, R := "ReiniciarChecarSimi", PV := 3, CV => "ContadorSimi");
   IF #_w46 THEN "ContadorSimiTemp" := "ContadorSimi"; END_IF;
   #_w47 := "Panel1RojoJ1" AND "Bounce3" AND "Panel1RojoJ1" AND "Intento1J1" AND ("Var".VectorPrincipalJ1["IntentoCompletoJ1", 2] = 0);
   IF #_w47 THEN
       "Var".VectorPrincipalJ1["IntentoCompletoJ1", 2] := 4;
       "Intento2J1" := TRUE;
   END_IF;
   #_w48 := #_w47 AND ("Var".VectorPrincipalJ1["IntentoCompletoJ1", 2] = "Var".CodigoOJ1[2]);
   "ContadorCorrectas".CTU(CU := #_w48, R := "ReiniciarChecarCorr", PV := 3, CV => "ContadorCorr");
   IF #_w48 THEN "ContadorCorrTemp" := "ContadorCorr"; END_IF;
   #_w49 := #_w47 AND ("Var".VectorPrincipalJ1["IntentoCompletoJ1", 2] <> "Var".CodigoOJ1[2]) AND (("Var".VectorPrincipalJ1["IntentoCompletoJ1", 2] = "Var".CodigoOJ1[0]) OR ("Var".VectorPrincipalJ1["IntentoCompletoJ1", 2] = "Var".CodigoOJ1[1]) OR ("Var".VectorPrincipalJ1["IntentoCompletoJ1", 2] = "Var".CodigoOJ1[3]));
   "ContadorSimilares".CTU(CU := #_w49, R := "ReiniciarChecarSimi", PV := 3, CV => "ContadorSimi");
   IF #_w49 THEN "ContadorSimiTemp" := "ContadorSimi"; END_IF;
   #_w50 := "Panel1RojoJ1" AND "Bounce4" AND "Panel1RojoJ1" AND "Intento2J1" AND ("Var".VectorPrincipalJ1["IntentoCompletoJ1", 3] = 0);
   IF #_w50 THEN
       "Var".VectorPrincipalJ1["IntentoCompletoJ1", 3] := 4;
       "Intento3J1" := TRUE;
   END_IF;
   #_w51 := #_w50 AND ("Var".VectorPrincipalJ1["IntentoCompletoJ1", 3] = "Var".CodigoOJ1[3]);
   "ContadorCorrectas".CTU(CU := #_w51, R := "ReiniciarChecarCorr", PV := 3, CV => "ContadorCorr");
   IF #_w51 THEN "ContadorCorrTemp" := "ContadorCorr"; END_IF;
   #_w52 := #_w50 AND ("Var".VectorPrincipalJ1["IntentoCompletoJ1", 3] <> "Var".CodigoOJ1[3]) AND (("Var".VectorPrincipalJ1["IntentoCompletoJ1", 3] = "Var".CodigoOJ1[0]) OR ("Var".VectorPrincipalJ1["IntentoCompletoJ1", 3] = "Var".CodigoOJ1[1]) OR ("Var".VectorPrincipalJ1["IntentoCompletoJ1", 3] = "Var".CodigoOJ1[2]));
   "ContadorSimilares".CTU(CU := #_w52, R := "ReiniciarChecarSimi", PV := 3, CV => "ContadorSimi");
   IF #_w52 THEN "ContadorSimiTemp" := "ContadorSimi"; END_IF;
   #_w53 := "Panel1AzulJ1" AND ("Var".VectorPrincipalJ1["IntentoCompletoJ1", 0] = 0) AND "Bounce1";
   IF #_w53 THEN
       "Var".VectorPrincipalJ1["IntentoCompletoJ1", 0] := 5;
       "Var".VectorCorrectas["IntentoCompletoJ1", 0] := 5;
       "Intento0J1" := TRUE;
   END_IF;
   #_w54 := #_w53 AND ("Var".VectorPrincipalJ1["IntentoCompletoJ1", 0] = "Var".CodigoOJ1[0]);
   "ContadorCorrectas".CTU(CU := #_w54, R := "ReiniciarChecarCorr", PV := 3, CV => "ContadorCorr");
   IF #_w54 THEN "ContadorCorrTemp" := "ContadorCorr"; END_IF;
   #_w55 := #_w53 AND ("Var".VectorPrincipalJ1["IntentoCompletoJ1", 0] <> "Var".CodigoOJ1[0]) AND (("Var".VectorPrincipalJ1["IntentoCompletoJ1", 0] = "Var".CodigoOJ1[1]) OR ("Var".VectorPrincipalJ1["IntentoCompletoJ1", 0] = "Var".CodigoOJ1[2]) OR ("Var".VectorPrincipalJ1["IntentoCompletoJ1", 0] = "Var".CodigoOJ1[3]));
   "ContadorSimilares".CTU(CU := #_w55, R := "ReiniciarChecarSimi", PV := 3, CV => "ContadorSimi");
   IF #_w55 THEN "ContadorSimiTemp" := "ContadorSimi"; END_IF;
   #_w56 := "Panel1AzulJ1" AND "Bounce2" AND "Panel1AzulJ1" AND "Intento0J1" AND ("Var".VectorPrincipalJ1["IntentoCompletoJ1", 1] = 0);
   IF #_w56 THEN
       "Var".VectorPrincipalJ1["IntentoCompletoJ1", 1] := 5;
       "Intento1J1" := TRUE;
   END_IF;
   #_w57 := #_w56 AND ("Var".VectorPrincipalJ1["IntentoCompletoJ1", 1] = "Var".CodigoOJ1[1]);
   "ContadorCorrectas".CTU(CU := #_w57, R := "ReiniciarChecarCorr", PV := 3, CV => "ContadorCorr");
   IF #_w57 THEN "ContadorCorrTemp" := "ContadorCorr"; END_IF;
   #_w58 := #_w56 AND ("Var".VectorPrincipalJ1["IntentoCompletoJ1", 1] <> "Var".CodigoOJ1[1]) AND (("Var".VectorPrincipalJ1["IntentoCompletoJ1", 1] = "Var".CodigoOJ1[0]) OR ("Var".VectorPrincipalJ1["IntentoCompletoJ1", 1] = "Var".CodigoOJ1[2]) OR ("Var".VectorPrincipalJ1["IntentoCompletoJ1", 1] = "Var".CodigoOJ1[3]));
   "ContadorSimilares".CTU(CU := #_w58, R := "ReiniciarChecarSimi", PV := 3, CV => "ContadorSimi");
   IF #_w58 THEN "ContadorSimiTemp" := "ContadorSimi"; END_IF;
   #_w59 := "Panel1AzulJ1" AND "Bounce3" AND "Panel1AzulJ1" AND "Intento1J1" AND ("Var".VectorPrincipalJ1["IntentoCompletoJ1", 2] = 0);
   IF #_w59 THEN
       "Var".VectorPrincipalJ1["IntentoCompletoJ1", 2] := 5;
       "Intento2J1" := TRUE;
   END_IF;
   #_w60 := #_w59 AND ("Var".VectorPrincipalJ1["IntentoCompletoJ1", 2] = "Var".CodigoOJ1[2]);
   "ContadorCorrectas".CTU(CU := #_w60, R := "ReiniciarChecarCorr", PV := 3, CV => "ContadorCorr");
   IF #_w60 THEN "ContadorCorrTemp" := "ContadorCorr"; END_IF;
   #_w61 := #_w59 AND ("Var".VectorPrincipalJ1["IntentoCompletoJ1", 2] <> "Var".CodigoOJ1[2]) AND (("Var".VectorPrincipalJ1["IntentoCompletoJ1", 2] = "Var".CodigoOJ1[0]) OR ("Var".VectorPrincipalJ1["IntentoCompletoJ1", 2] = "Var".CodigoOJ1[1]) OR ("Var".VectorPrincipalJ1["IntentoCompletoJ1", 2] = "Var".CodigoOJ1[3]));
   "ContadorSimilares".CTU(CU := #_w61, R := "ReiniciarChecarSimi", PV := 3, CV => "ContadorSimi");
   IF #_w61 THEN "ContadorSimiTemp" := "ContadorSimi"; END_IF;
   #_w62 := "Panel1AzulJ1" AND "Bounce4" AND "Panel1AzulJ1" AND "Intento2J1" AND ("Var".VectorPrincipalJ1["IntentoCompletoJ1", 3] = 0);
   IF #_w62 THEN
       "Var".VectorPrincipalJ1["IntentoCompletoJ1", 3] := 5;
       "Intento3J1" := TRUE;
   END_IF;
   #_w63 := #_w62 AND ("Var".VectorPrincipalJ1["IntentoCompletoJ1", 3] = "Var".CodigoOJ1[3]);
   "ContadorCorrectas".CTU(CU := #_w63, R := "ReiniciarChecarCorr", PV := 3, CV => "ContadorCorr");
   IF #_w63 THEN "ContadorCorrTemp" := "ContadorCorr"; END_IF;
   #_w64 := #_w62 AND ("Var".VectorPrincipalJ1["IntentoCompletoJ1", 3] <> "Var".CodigoOJ1[3]) AND (("Var".VectorPrincipalJ1["IntentoCompletoJ1", 3] = "Var".CodigoOJ1[0]) OR ("Var".VectorPrincipalJ1["IntentoCompletoJ1", 3] = "Var".CodigoOJ1[2]) OR ("Var".VectorPrincipalJ1["IntentoCompletoJ1", 3] = "Var".CodigoOJ1[2]));
   "ContadorSimilares".CTU(CU := #_w64, R := "ReiniciarChecarSimi", PV := 3, CV => "ContadorSimi");
   IF #_w64 THEN "ContadorSimiTemp" := "ContadorSimi"; END_IF;
   #_w65 := "Panel1VerdeJ1" AND ("Var".VectorPrincipalJ1["IntentoCompletoJ1", 0] = 0) AND "Bounce1";
   IF #_w65 THEN
       "Var".VectorPrincipalJ1["IntentoCompletoJ1", 0] := 6;
       "Var".VectorCorrectas["IntentoCompletoJ1", 0] := 6;
       "Intento0J1" := TRUE;
   END_IF;
   #_w66 := #_w65 AND ("Var".VectorPrincipalJ1["IntentoCompletoJ1", 0] = "Var".CodigoOJ1[0]);
   "ContadorCorrectas".CTU(CU := #_w66, R := "ReiniciarChecarCorr", PV := 3, CV => "ContadorCorr");
   IF #_w66 THEN "ContadorCorrTemp" := "ContadorCorr"; END_IF;
   #_w67 := #_w65 AND ("Var".VectorPrincipalJ1["IntentoCompletoJ1", 0] <> "Var".CodigoOJ1[0]) AND (("Var".VectorPrincipalJ1["IntentoCompletoJ1", 0] = "Var".CodigoOJ1[1]) OR ("Var".VectorPrincipalJ1["IntentoCompletoJ1", 0] = "Var".CodigoOJ1[2]) OR ("Var".VectorPrincipalJ1["IntentoCompletoJ1", 0] = "Var".CodigoOJ1[3]));
   "ContadorSimilares".CTU(CU := #_w67, R := "ReiniciarChecarSimi", PV := 3, CV => "ContadorSimi");
   IF #_w67 THEN "ContadorSimiTemp" := "ContadorSimi"; END_IF;
   #_w68 := "Panel1VerdeJ1" AND "Bounce2" AND "Panel1VerdeJ1" AND "Intento0J1" AND ("Var".VectorPrincipalJ1["IntentoCompletoJ1", 1] = 0);
   IF #_w68 THEN
       "Var".VectorPrincipalJ1["IntentoCompletoJ1", 1] := 6;
       "Intento1J1" := TRUE;
   END_IF;
   #_w69 := #_w68 AND ("Var".VectorPrincipalJ1["IntentoCompletoJ1", 1] = "Var".CodigoOJ1[1]);
   "ContadorCorrectas".CTU(CU := #_w69, R := "ReiniciarChecarCorr", PV := 3, CV => "ContadorCorr");
   IF #_w69 THEN "ContadorCorrTemp" := "ContadorCorr"; END_IF;
   #_w70 := #_w68 AND ("Var".VectorPrincipalJ1["IntentoCompletoJ1", 1] <> "Var".CodigoOJ1[1]) AND (("Var".VectorPrincipalJ1["IntentoCompletoJ1", 1] = "Var".CodigoOJ1[0]) OR ("Var".VectorPrincipalJ1["IntentoCompletoJ1", 1] = "Var".CodigoOJ1[2]) OR ("Var".VectorPrincipalJ1["IntentoCompletoJ1", 1] = "Var".CodigoOJ1[3]));
   "ContadorSimilares".CTU(CU := #_w70, R := "ReiniciarChecarSimi", PV := 3, CV => "ContadorSimi");
   IF #_w70 THEN "ContadorSimiTemp" := "ContadorSimi"; END_IF;
   #_w71 := "Panel1VerdeJ1" AND "Bounce3" AND "Panel1VerdeJ1" AND "Intento1J1" AND ("Var".VectorPrincipalJ1["IntentoCompletoJ1", 2] = 0);
   IF #_w71 THEN
       "Var".VectorPrincipalJ1["IntentoCompletoJ1", 2] := 6;
       "Intento2J1" := TRUE;
   END_IF;
   #_w72 := #_w71 AND ("Var".VectorPrincipalJ1["IntentoCompletoJ1", 2] = "Var".CodigoOJ1[2]);
   "ContadorCorrectas".CTU(CU := #_w72, R := "ReiniciarChecarCorr", PV := 3, CV => "ContadorCorr");
   IF #_w72 THEN "ContadorCorrTemp" := "ContadorCorr"; END_IF;
   #_w73 := #_w71 AND ("Var".VectorPrincipalJ1["IntentoCompletoJ1", 2] <> "Var".CodigoOJ1[2]) AND (("Var".VectorPrincipalJ1["IntentoCompletoJ1", 2] = "Var".CodigoOJ1[0]) OR ("Var".VectorPrincipalJ1["IntentoCompletoJ1", 2] = "Var".CodigoOJ1[1]) OR ("Var".VectorPrincipalJ1["IntentoCompletoJ1", 2] = "Var".CodigoOJ1[3]));
   "ContadorSimilares".CTU(CU := #_w73, R := "ReiniciarChecarSimi", PV := 3, CV => "ContadorSimi");
   IF #_w73 THEN "ContadorSimiTemp" := "ContadorSimi"; END_IF;
   #_w74 := "Panel1VerdeJ1" AND "Bounce4" AND "Panel1VerdeJ1" AND "Intento2J1" AND ("Var".VectorPrincipalJ1["IntentoCompletoJ1", 3] = 0);
   IF #_w74 THEN
       "Var".VectorPrincipalJ1["IntentoCompletoJ1", 3] := 6;
       "Intento3J1" := TRUE;
   END_IF;
   #_w75 := #_w74 AND ("Var".VectorPrincipalJ1["IntentoCompletoJ1", 3] = "Var".CodigoOJ1[3]);
   "ContadorCorrectas".CTU(CU := #_w75, R := "ReiniciarChecarCorr", PV := 3, CV => "ContadorCorr");
   IF #_w75 THEN "ContadorCorrTemp" := "ContadorCorr"; END_IF;
   #_w76 := #_w74 AND ("Var".VectorPrincipalJ1["IntentoCompletoJ1", 3] <> "Var".CodigoOJ1[3]) AND (("Var".VectorPrincipalJ1["IntentoCompletoJ1", 3] = "Var".CodigoOJ1[0]) OR ("Var".VectorPrincipalJ1["IntentoCompletoJ1", 3] = "Var".CodigoOJ1[1]) OR ("Var".VectorPrincipalJ1["IntentoCompletoJ1", 3] = "Var".CodigoOJ1[2]));
   "ContadorSimilares".CTU(CU := #_w76, R := "ReiniciarChecarSimi", PV := 3, CV => "ContadorSimi");
   IF #_w76 THEN "ContadorSimiTemp" := "ContadorSimi"; END_IF;
   #_w77 := "Panel1AmarilloJ1" AND ("Var".VectorPrincipalJ1["IntentoCompletoJ1", 0] = 0) AND "Bounce1";
   IF #_w77 THEN
       "Var".VectorPrincipalJ1["IntentoCompletoJ1", 0] := 7;
       "Var".VectorCorrectas["IntentoCompletoJ1", 0] := 7;
       "Intento0J1" := TRUE;
   END_IF;
   #_w78 := #_w77 AND ("Var".VectorPrincipalJ1["IntentoCompletoJ1", 0] = "Var".CodigoOJ1[0]);
   "ContadorCorrectas".CTU(CU := #_w78, R := "ReiniciarChecarCorr", PV := 3, CV => "ContadorCorr");
   IF #_w78 THEN "ContadorCorrTemp" := "ContadorCorr"; END_IF;
   #_w79 := #_w77 AND ("Var".VectorPrincipalJ1["IntentoCompletoJ1", 0] <> "Var".CodigoOJ1[0]) AND (("Var".VectorPrincipalJ1["IntentoCompletoJ1", 0] = "Var".CodigoOJ1[1]) OR ("Var".VectorPrincipalJ1["IntentoCompletoJ1", 0] = "Var".CodigoOJ1[2]) OR ("Var".VectorPrincipalJ1["IntentoCompletoJ1", 0] = "Var".CodigoOJ1[3]));
   "ContadorSimilares".CTU(CU := #_w79, R := "ReiniciarChecarSimi", PV := 3, CV => "ContadorSimi");
   IF #_w79 THEN "ContadorSimiTemp" := "ContadorSimi"; END_IF;
   #_w80 := "Panel1AmarilloJ1" AND "Bounce2" AND "Panel1AmarilloJ1" AND "Intento0J1" AND ("Var".VectorPrincipalJ1["IntentoCompletoJ1", 1] = 0);
   IF #_w80 THEN
       "Var".VectorPrincipalJ1["IntentoCompletoJ1", 1] := 7;
       "Intento1J1" := TRUE;
   END_IF;
   #_w81 := #_w80 AND ("Var".VectorPrincipalJ1["IntentoCompletoJ1", 1] = "Var".CodigoOJ1[1]);
   "ContadorCorrectas".CTU(CU := #_w81, R := "ReiniciarChecarCorr", PV := 3, CV => "ContadorCorr");
   IF #_w81 THEN "ContadorCorrTemp" := "ContadorCorr"; END_IF;
   #_w82 := #_w80 AND ("Var".VectorPrincipalJ1["IntentoCompletoJ1", 1] <> "Var".CodigoOJ1[1]) AND (("Var".VectorPrincipalJ1["IntentoCompletoJ1", 1] = "Var".CodigoOJ1[0]) OR ("Var".VectorPrincipalJ1["IntentoCompletoJ1", 1] = "Var".CodigoOJ1[2]) OR ("Var".VectorPrincipalJ1["IntentoCompletoJ1", 1] = "Var".CodigoOJ1[3]));
   "ContadorSimilares".CTU(CU := #_w82, R := "ReiniciarChecarSimi", PV := 3, CV => "ContadorSimi");
   IF #_w82 THEN "ContadorSimiTemp" := "ContadorSimi"; END_IF;
   #_w83 := "Panel1AmarilloJ1" AND "Bounce3" AND "Panel1AmarilloJ1" AND "Intento1J1" AND ("Var".VectorPrincipalJ1["IntentoCompletoJ1", 2] = 0);
   IF #_w83 THEN
       "Var".VectorPrincipalJ1["IntentoCompletoJ1", 2] := 7;
       "Intento2J1" := TRUE;
   END_IF;
   #_w84 := #_w83 AND ("Var".VectorPrincipalJ1["IntentoCompletoJ1", 2] = "Var".CodigoOJ1[2]);
   "ContadorCorrectas".CTU(CU := #_w84, R := "ReiniciarChecarCorr", PV := 3, CV => "ContadorCorr");
   IF #_w84 THEN "ContadorCorrTemp" := "ContadorCorr"; END_IF;
   #_w85 := #_w83 AND ("Var".VectorPrincipalJ1["IntentoCompletoJ1", 2] <> "Var".CodigoOJ1[2]) AND (("Var".VectorPrincipalJ1["IntentoCompletoJ1", 2] = "Var".CodigoOJ1[0]) OR ("Var".VectorPrincipalJ1["IntentoCompletoJ1", 2] = "Var".CodigoOJ1[1]) OR ("Var".VectorPrincipalJ1["IntentoCompletoJ1", 2] = "Var".CodigoOJ1[3]));
   "ContadorSimilares".CTU(CU := #_w85, R := "ReiniciarChecarSimi", PV := 3, CV => "ContadorSimi");
   IF #_w85 THEN "ContadorSimiTemp" := "ContadorSimi"; END_IF;
   #_w86 := "Panel1AmarilloJ1" AND "Bounce4" AND "Panel1AmarilloJ1" AND "Intento2J1" AND ("Var".VectorPrincipalJ1["IntentoCompletoJ1", 3] = 0);
   IF #_w86 THEN
       "Var".VectorPrincipalJ1["IntentoCompletoJ1", 3] := 7;
       "Intento3J1" := TRUE;
   END_IF;
   #_w87 := #_w86 AND ("Var".VectorPrincipalJ1["IntentoCompletoJ1", 3] = "Var".CodigoOJ1[3]);
   "ContadorCorrectas".CTU(CU := #_w87, R := "ReiniciarChecarCorr", PV := 3, CV => "ContadorCorr");
   IF #_w87 THEN "ContadorCorrTemp" := "ContadorCorr"; END_IF;
   #_w88 := #_w86 AND ("Var".VectorPrincipalJ1["IntentoCompletoJ1", 3] <> "Var".CodigoOJ1[3]) AND (("Var".VectorPrincipalJ1["IntentoCompletoJ1", 3] = "Var".CodigoOJ1[0]) OR ("Var".VectorPrincipalJ1["IntentoCompletoJ1", 3] = "Var".CodigoOJ1[1]) OR ("Var".VectorPrincipalJ1["IntentoCompletoJ1", 3] = "Var".CodigoOJ1[2]));
   "ContadorSimilares".CTU(CU := #_w88, R := "ReiniciarChecarSimi", PV := 3, CV => "ContadorSimi");
   IF #_w88 THEN "ContadorSimiTemp" := "ContadorSimi"; END_IF;
END_REGION

REGION Network 7: Comprobar Intentos
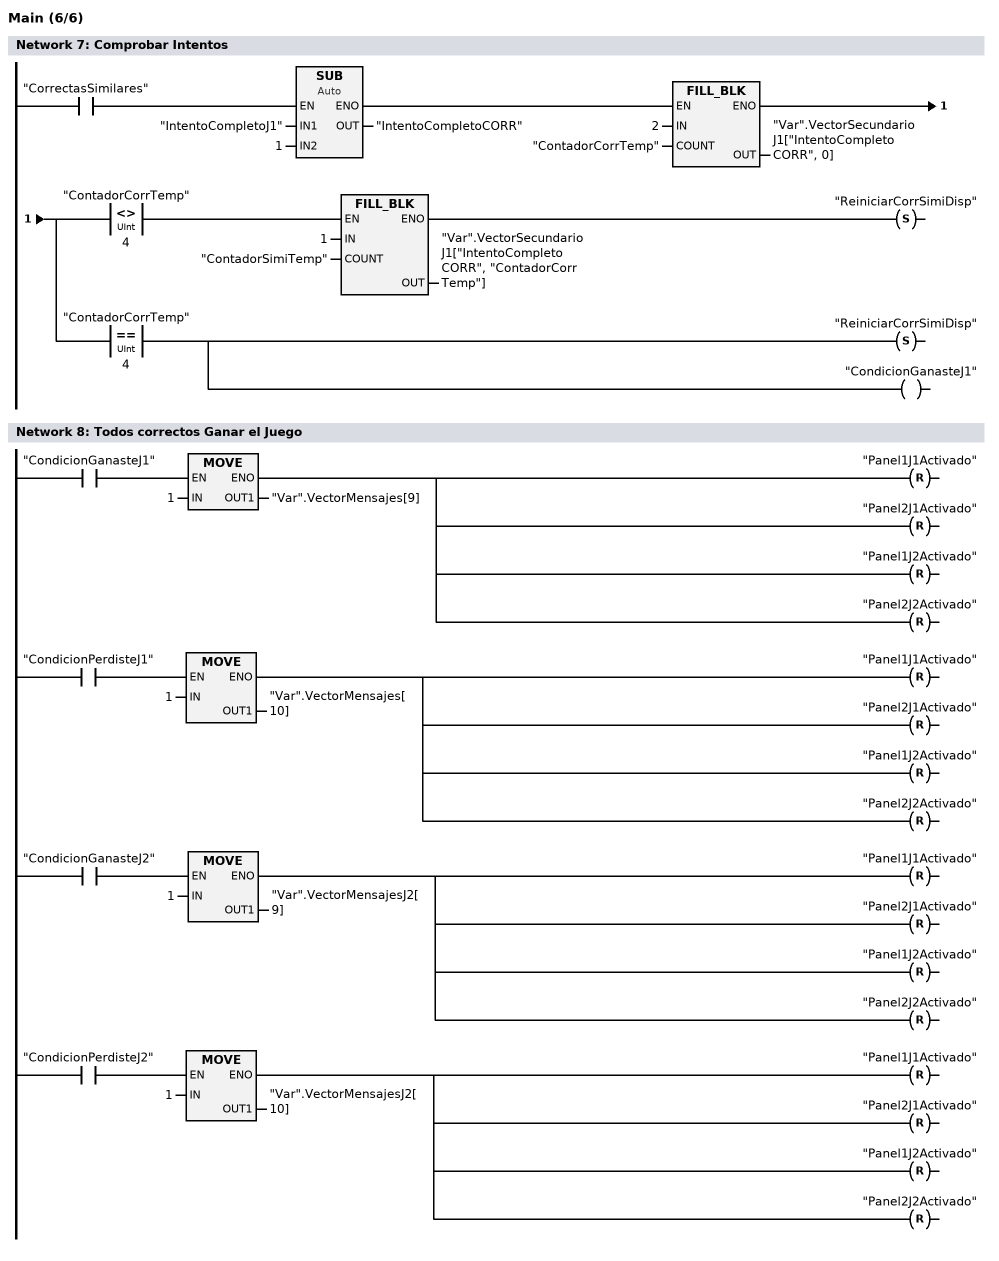
   RUNG wire#powerrail
      Contact( "CorrectasSimilares" )
      Sub(in1 := "IntentoCompletoJ1", in2 := 1, out => "IntentoCompletoCORR")
      FillBlockI(in := 2, count := "ContadorCorrTemp", out => "Var".VectorSecundarioJ1["IntentoCompletoCORR", 0])
      wire#w1
      { S7_Templates := "SrcType := UInt" } NE_Contact(in1 := "ContadorCorrTemp", in2 := 4)
      FillBlockI(in := 1, count := "ContadorSimiTemp", out => "Var".VectorSecundarioJ1["IntentoCompletoCORR", "ContadorCorrTemp"])
      S_Coil( "ReiniciarCorrSimiDisp" )
   END_RUNG
   RUNG wire#w1
      { S7_Templates := "SrcType := UInt" } EQ_Contact(in1 := "ContadorCorrTemp", in2 := 4)
      wire#w2
      S_Coil( "ReiniciarCorrSimiDisp" )
   END_RUNG
   RUNG wire#w2
      Coil( "CondicionGanasteJ1" )
   END_RUNG
   // the same network as SCL:
   IF "CorrectasSimilares" THEN "IntentoCompletoCORR" := "IntentoCompletoJ1" - 1; END_IF;
   #_w1 := "CorrectasSimilares";
   IF #_w1 THEN
       FILL_BLK(IN := 2, COUNT := "ContadorCorrTemp", OUT => "Var".VectorSecundarioJ1["IntentoCompletoCORR", 0]);
   END_IF;
   #_w2 := #_w1 AND ("ContadorCorrTemp" <> 4);
   IF #_w2 THEN
       FILL_BLK(IN := 1,
                COUNT := "ContadorSimiTemp",
                OUT => "Var".VectorSecundarioJ1["IntentoCompletoCORR", "ContadorCorrTemp"]);
       "ReiniciarCorrSimiDisp" := TRUE;
   END_IF;
   #_w3 := #_w1 AND ("ContadorCorrTemp" = 4);
   IF #_w3 THEN "ReiniciarCorrSimiDisp" := TRUE; END_IF;
   "CondicionGanasteJ1" := #_w3;
END_REGION

REGION Network 8: Todos correctos Ganar el Juego
   RUNG wire#powerrail
      Contact( "CondicionGanasteJ1" )
      Move(in := 1, out1 => "Var".VectorMensajes[9])
      wire#w1
      R_Coil( "Panel1J1Activado" )
   END_RUNG
   RUNG wire#w1
      R_Coil( "Panel2J1Activado" )
   END_RUNG
   RUNG wire#w1
      R_Coil( "Panel1J2Activado" )
   END_RUNG
   RUNG wire#w1
      R_Coil( "Panel2J2Activado" )
   END_RUNG
   RUNG wire#powerrail
      Contact( "CondicionPerdisteJ1" )
      Move(in := 1, out1 => "Var".VectorMensajes[10])
      wire#w2
      R_Coil( "Panel1J1Activado" )
   END_RUNG
   RUNG wire#w2
      R_Coil( "Panel2J1Activado" )
   END_RUNG
   RUNG wire#w2
      R_Coil( "Panel1J2Activado" )
   END_RUNG
   RUNG wire#w2
      R_Coil( "Panel2J2Activado" )
   END_RUNG
   RUNG wire#powerrail
      Contact( "CondicionGanasteJ2" )
      Move(in := 1, out1 => "Var".VectorMensajesJ2[9])
      wire#w3
      R_Coil( "Panel1J1Activado" )
   END_RUNG
   RUNG wire#w3
      R_Coil( "Panel2J1Activado" )
   END_RUNG
   RUNG wire#w3
      R_Coil( "Panel1J2Activado" )
   END_RUNG
   RUNG wire#w3
      R_Coil( "Panel2J2Activado" )
   END_RUNG
   RUNG wire#powerrail
      Contact( "CondicionPerdisteJ2" )
      Move(in := 1, out1 => "Var".VectorMensajesJ2[10])
      wire#w4
      R_Coil( "Panel1J1Activado" )
   END_RUNG
   RUNG wire#w4
      R_Coil( "Panel2J1Activado" )
   END_RUNG
   RUNG wire#w4
      R_Coil( "Panel1J2Activado" )
   END_RUNG
   RUNG wire#w4
      R_Coil( "Panel2J2Activado" )
   END_RUNG
   // the same network as SCL:
   IF "CondicionGanasteJ1" THEN
       "Var".VectorMensajes[9] := 1;
       "Panel1J1Activado" := FALSE;
       "Panel2J1Activado" := FALSE;
       "Panel1J2Activado" := FALSE;
       "Panel2J2Activado" := FALSE;
   END_IF;
   IF "CondicionPerdisteJ1" THEN
       "Var".VectorMensajes[10] := 1;
       "Panel1J1Activado" := FALSE;
       "Panel2J1Activado" := FALSE;
       "Panel1J2Activado" := FALSE;
       "Panel2J2Activado" := FALSE;
   END_IF;
   IF "CondicionGanasteJ2" THEN
       "Var".VectorMensajesJ2[9] := 1;
       "Panel1J1Activado" := FALSE;
       "Panel2J1Activado" := FALSE;
       "Panel1J2Activado" := FALSE;
       "Panel2J2Activado" := FALSE;
   END_IF;
   IF "CondicionPerdisteJ2" THEN
       "Var".VectorMensajesJ2[10] := 1;
       "Panel1J1Activado" := FALSE;
       "Panel2J1Activado" := FALSE;
       "Panel1J2Activado" := FALSE;
       "Panel2J2Activado" := FALSE;
   END_IF;
END_REGION
END_ORGANIZATION_BLOCK

(* ===== HMI "HMI_RT_1" =====
system functions are stored by id; their names below are inferred from use
connection "HMI_Connection_1": ETHERNET, S7_1500_OMS

HMI tags "Default tag table"
   "Tag_ScreenNumber" : UInt, internal
   "ReiniciarJuego" : Bool = PLC ReiniciarJuego AT %M6.0, 1 s
   "Panel2CafeJ1" : Bool = PLC Panel2CafeJ1 AT %M10.4, 1 s
   "Panel2RosaJ1" : Bool = PLC Panel2RosaJ1 AT %M10.5, 1 s
   "Panel2MoradoJ1" : Bool = PLC Panel2MoradoJ1 AT %M10.6, 1 s
   "Panel2RojoJ1" : Bool = PLC Panel2RojoJ1 AT %M10.7, 1 s
   "Panel2AzulJ1" : Bool = PLC Panel2AzulJ1 AT %M11.0, 1 s
   "Panel2VerdeJ1" : Bool = PLC Panel2VerdeJ1 AT %M11.1, 1 s
   "Panel2AmarilloJ1" : Bool = PLC Panel2AmarilloJ1 AT %M11.2, 1 s
   "Panel1CafeJ1" : Bool = PLC Panel1CafeJ1 AT %M9.5, 1 s
   "Panel1RosaJ1" : Bool = PLC Panel1RosaJ1 AT %M9.6, 1 s
   "Panel1MoradoJ1" : Bool = PLC Panel1MoradoJ1 AT %M9.7, 1 s
   "Panel1RojoJ1" : Bool = PLC Panel1RojoJ1 AT %M10.0, 1 s
   "Panel1AzulJ1" : Bool = PLC Panel1AzulJ1 AT %M10.1, 1 s
   "Panel1VerdeJ1" : Bool = PLC Panel1VerdeJ1 AT %M10.2, 1 s
   "Panel1AmarilloJ1" : Bool = PLC Panel1AmarilloJ1 AT %M10.3, 1 s
   "Panel1J1Activado" : Bool = PLC Panel1J1Activado AT %M13.1, 1 s
   "Panel2J1Activado" : Bool = PLC Panel2J1Activado AT %M13.2, 1 s
   "Var_VectorMensajes{0}" : Int = PLC "Var".VectorMensajes[0], 1 s
   "Var_VectorMensajes{1}" : Int = PLC "Var".VectorMensajes[1], 1 s
   "Var_VectorMensajes{2}" : Int = PLC "Var".VectorMensajes[2], 1 s
   "Var_VectorMensajes{3}" : Int = PLC "Var".VectorMensajes[3], 1 s
   "Var_VectorMensajes{4}" : Int = PLC "Var".VectorMensajes[4], 1 s
   "Var_VectorMensajes{5}" : Int = PLC "Var".VectorMensajes[5], 1 s
   "Var_VectorMensajes{6}" : Int = PLC "Var".VectorMensajes[6], 1 s
   "Var_VectorMensajes{7}" : Int = PLC "Var".VectorMensajes[7], 1 s
   "Var_VectorMensajes{8}" : Int = PLC "Var".VectorMensajes[8], 1 s
   "Var_VectorMensajes{9}" : Int = PLC "Var".VectorMensajes[9], 1 s
   "Var_VectorMensajes{10}" : Int = PLC "Var".VectorMensajes[10], 1 s
   "Var_CodigoOJ1{0}" : Int = PLC "Var".CodigoOJ1[0], 1 s
   "Var_CodigoOJ1{1}" : Int = PLC "Var".CodigoOJ1[1], 1 s
   "Var_CodigoOJ1{2}" : Int = PLC "Var".CodigoOJ1[2], 1 s
   "Var_CodigoOJ1{3}" : Int = PLC "Var".CodigoOJ1[3], 1 s
   "Var_CodigoSJ1{0}" : Int = PLC "Var".CodigoSJ1[0], 1 s
   "Var_CodigoSJ1{1}" : Int = PLC "Var".CodigoSJ1[1], 1 s
   "Var_CodigoSJ1{2}" : Int = PLC "Var".CodigoSJ1[2], 1 s
   "Var_CodigoSJ1{3}" : Int = PLC "Var".CodigoSJ1[3], 1 s
   "Var_VectorPrincipalJ1{0,0}" : Int = PLC "Var".VectorPrincipalJ1[0,0], 1 s
   "Var_VectorPrincipalJ1{0,1}" : Int = PLC "Var".VectorPrincipalJ1[0,1], 1 s
   "Var_VectorPrincipalJ1{0,2}" : Int = PLC "Var".VectorPrincipalJ1[0,2], 1 s
   "Var_VectorPrincipalJ1{0,3}" : Int = PLC "Var".VectorPrincipalJ1[0,3], 1 s
   "Var_VectorPrincipalJ1{1,0}" : Int = PLC "Var".VectorPrincipalJ1[1,0], 1 s
   "Var_VectorPrincipalJ1{1,1}" : Int = PLC "Var".VectorPrincipalJ1[1,1], 1 s
   "Var_VectorPrincipalJ1{1,2}" : Int = PLC "Var".VectorPrincipalJ1[1,2], 1 s
   "Var_VectorPrincipalJ1{1,3}" : Int = PLC "Var".VectorPrincipalJ1[1,3], 1 s
   "Var_VectorPrincipalJ1{2,0}" : Int = PLC "Var".VectorPrincipalJ1[2,0], 1 s
   "Var_VectorPrincipalJ1{2,1}" : Int = PLC "Var".VectorPrincipalJ1[2,1], 1 s
   "Var_VectorPrincipalJ1{2,2}" : Int = PLC "Var".VectorPrincipalJ1[2,2], 1 s
   "Var_VectorPrincipalJ1{2,3}" : Int = PLC "Var".VectorPrincipalJ1[2,3], 1 s
   "Var_VectorPrincipalJ1{3,0}" : Int = PLC "Var".VectorPrincipalJ1[3,0], 1 s
   "Var_VectorPrincipalJ1{3,1}" : Int = PLC "Var".VectorPrincipalJ1[3,1], 1 s
   "Var_VectorPrincipalJ1{3,2}" : Int = PLC "Var".VectorPrincipalJ1[3,2], 1 s
   "Var_VectorPrincipalJ1{3,3}" : Int = PLC "Var".VectorPrincipalJ1[3,3], 1 s
   "Var_VectorPrincipalJ1{4,0}" : Int = PLC "Var".VectorPrincipalJ1[4,0], 1 s
   "Var_VectorPrincipalJ1{4,1}" : Int = PLC "Var".VectorPrincipalJ1[4,1], 1 s
   "Var_VectorPrincipalJ1{4,2}" : Int = PLC "Var".VectorPrincipalJ1[4,2], 1 s
   "Var_VectorPrincipalJ1{4,3}" : Int = PLC "Var".VectorPrincipalJ1[4,3], 1 s
   "Var_VectorPrincipalJ1{5,0}" : Int = PLC "Var".VectorPrincipalJ1[5,0], 1 s
   "Var_VectorPrincipalJ1{5,1}" : Int = PLC "Var".VectorPrincipalJ1[5,1], 1 s
   "Var_VectorPrincipalJ1{5,2}" : Int = PLC "Var".VectorPrincipalJ1[5,2], 1 s
   "Var_VectorPrincipalJ1{5,3}" : Int = PLC "Var".VectorPrincipalJ1[5,3], 1 s
   "Var_VectorPrincipalJ1{6,0}" : Int = PLC "Var".VectorPrincipalJ1[6,0], 1 s
   "Var_VectorPrincipalJ1{6,1}" : Int = PLC "Var".VectorPrincipalJ1[6,1], 1 s
   "Var_VectorPrincipalJ1{6,2}" : Int = PLC "Var".VectorPrincipalJ1[6,2], 1 s
   "Var_VectorPrincipalJ1{6,3}" : Int = PLC "Var".VectorPrincipalJ1[6,3], 1 s
   "Var_VectorPrincipalJ1{7,0}" : Int = PLC "Var".VectorPrincipalJ1[7,0], 1 s
   "Var_VectorPrincipalJ1{7,1}" : Int = PLC "Var".VectorPrincipalJ1[7,1], 1 s
   "Var_VectorPrincipalJ1{7,2}" : Int = PLC "Var".VectorPrincipalJ1[7,2], 1 s
   "Var_VectorPrincipalJ1{7,3}" : Int = PLC "Var".VectorPrincipalJ1[7,3], 1 s
   "Var_VectorSecundarioJ1{0,0}" : Int = PLC "Var".VectorSecundarioJ1[0,0], 1 s
   "Var_VectorSecundarioJ1{0,1}" : Int = PLC "Var".VectorSecundarioJ1[0,1], 1 s
   "Var_VectorSecundarioJ1{0,2}" : Int = PLC "Var".VectorSecundarioJ1[0,2], 1 s
   "Var_VectorSecundarioJ1{0,3}" : Int = PLC "Var".VectorSecundarioJ1[0,3], 1 s
   "Var_VectorSecundarioJ1{1,0}" : Int = PLC "Var".VectorSecundarioJ1[1,0], 1 s
   "Var_VectorSecundarioJ1{1,1}" : Int = PLC "Var".VectorSecundarioJ1[1,1], 1 s
   "Var_VectorSecundarioJ1{1,2}" : Int = PLC "Var".VectorSecundarioJ1[1,2], 1 s
   "Var_VectorSecundarioJ1{1,3}" : Int = PLC "Var".VectorSecundarioJ1[1,3], 1 s
   "Var_VectorSecundarioJ1{2,0}" : Int = PLC "Var".VectorSecundarioJ1[2,0], 1 s
   "Var_VectorSecundarioJ1{2,1}" : Int = PLC "Var".VectorSecundarioJ1[2,1], 1 s
   "Var_VectorSecundarioJ1{2,2}" : Int = PLC "Var".VectorSecundarioJ1[2,2], 1 s
   "Var_VectorSecundarioJ1{2,3}" : Int = PLC "Var".VectorSecundarioJ1[2,3], 1 s
   "Var_VectorSecundarioJ1{3,0}" : Int = PLC "Var".VectorSecundarioJ1[3,0], 1 s
   "Var_VectorSecundarioJ1{3,1}" : Int = PLC "Var".VectorSecundarioJ1[3,1], 1 s
   "Var_VectorSecundarioJ1{3,2}" : Int = PLC "Var".VectorSecundarioJ1[3,2], 1 s
   "Var_VectorSecundarioJ1{3,3}" : Int = PLC "Var".VectorSecundarioJ1[3,3], 1 s
   "Var_VectorSecundarioJ1{4,0}" : Int = PLC "Var".VectorSecundarioJ1[4,0], 1 s
   "Var_VectorSecundarioJ1{4,1}" : Int = PLC "Var".VectorSecundarioJ1[4,1], 1 s
   "Var_VectorSecundarioJ1{4,2}" : Int = PLC "Var".VectorSecundarioJ1[4,2], 1 s
   "Var_VectorSecundarioJ1{4,3}" : Int = PLC "Var".VectorSecundarioJ1[4,3], 1 s
   "Var_VectorSecundarioJ1{5,0}" : Int = PLC "Var".VectorSecundarioJ1[5,0], 1 s
   "Var_VectorSecundarioJ1{5,1}" : Int = PLC "Var".VectorSecundarioJ1[5,1], 1 s
   "Var_VectorSecundarioJ1{5,2}" : Int = PLC "Var".VectorSecundarioJ1[5,2], 1 s
   "Var_VectorSecundarioJ1{5,3}" : Int = PLC "Var".VectorSecundarioJ1[5,3], 1 s
   "Var_VectorSecundarioJ1{6,0}" : Int = PLC "Var".VectorSecundarioJ1[6,0], 1 s
   "Var_VectorSecundarioJ1{6,1}" : Int = PLC "Var".VectorSecundarioJ1[6,1], 1 s
   "Var_VectorSecundarioJ1{6,2}" : Int = PLC "Var".VectorSecundarioJ1[6,2], 1 s
   "Var_VectorSecundarioJ1{6,3}" : Int = PLC "Var".VectorSecundarioJ1[6,3], 1 s
   "Var_VectorSecundarioJ1{7,0}" : Int = PLC "Var".VectorSecundarioJ1[7,0], 1 s
   "Var_VectorSecundarioJ1{7,1}" : Int = PLC "Var".VectorSecundarioJ1[7,1], 1 s
   "Var_VectorSecundarioJ1{7,2}" : Int = PLC "Var".VectorSecundarioJ1[7,2], 1 s
   "Var_VectorSecundarioJ1{7,3}" : Int = PLC "Var".VectorSecundarioJ1[7,3], 1 s
   "Bounce1" : Bool = PLC Bounce1 AT %M13.6, 1 s
   "Bounce5" : Bool = PLC Bounce5 AT %M14.1, 1 s
   "ReiniciarCorrSimiDisp" : Bool = PLC ReiniciarCorrSimiDisp AT %M34.0, 1 s

screen "Root screen" 800x442, template "Template_1"
   on GenerateScreen: SetTag("Tag_ScreenNumber", 1)
   Button "Button_3" at 67,293 size 28x26; TextOff 'Text'
      on Press: SetBit("Panel1CafeJ1")
      on Release: SetBit("Bounce5"); ResetBit("Panel1CafeJ1")
      Appearance <- "Panel1J1Activado"
   Button "Button_4" at 99,293 size 27x26; TextOff 'Text'
      on Press: SetBit("Panel1RosaJ1")
      on Release: SetBit("Bounce5"); ResetBit("Panel1RosaJ1")
      Appearance <- "Panel1J1Activado"
   Button "Button_5" at 131,293 size 27x24; TextOff 'Text'
      on Press: SetBit("Panel1MoradoJ1")
      on Release: SetBit("Bounce5"); ResetBit("Panel1MoradoJ1")
      Appearance <- "Panel1J1Activado"
   Button "Button_6" at 165,293 size 25x25; TextOff 'Text'
      on Press: SetBit("Panel1RojoJ1")
      on Release: SetBit("Bounce5"); ResetBit("Panel1RojoJ1")
      Appearance <- "Panel1J1Activado"
   Button "Button_7" at 196,293 size 25x24; TextOff 'Text'
      on Press: SetBit("Panel1AzulJ1")
      on Release: SetBit("Bounce5"); ResetBit("Panel1AzulJ1")
      Appearance <- "Panel1J1Activado"
   Button "Button_8" at 227,293 size 25x25; TextOff 'Text'
      on Press: SetBit("Panel1VerdeJ1")
      on Release: SetBit("Bounce5"); ResetBit("Panel1VerdeJ1")
      Appearance <- "Panel1J1Activado"
   Button "Button_9" at 256,294 size 25x23; TextOff 'Text'
      on Press: SetBit("Panel1AmarilloJ1")
      on Release: SetBit("Bounce5"); ResetBit("Panel1AmarilloJ1")
      Appearance <- "Panel1J1Activado"
   TextField "Text field_1" at 37,250 size 16x23; Text '1'
   TextField "Text field_2" at 37,221 size 16x23; Text '2'
   TextField "Text field_3" at 37,194 size 16x23; Text '3'
   TextField "Text field_4" at 37,163 size 16x23; Text '4'
   TextField "Text field_5" at 37,134 size 16x23; Text '5'
   TextField "Text field_6" at 37,103 size 16x23; Text '6'
   TextField "Text field_7" at 37,74 size 16x23; Text '7'
   TextField "Text field_8" at 37,43 size 16x23; Text '8'
   Circle "Circle_1" at 92,254 size 23x23
      Appearance <- "Var_VectorPrincipalJ1{0,0}"
   Circle "Circle_2" at 128,254 size 23x23
      Appearance <- "Var_VectorPrincipalJ1{0,1}"
   Circle "Circle_3" at 164,254 size 23x23
      Appearance <- "Var_VectorPrincipalJ1{0,2}"
   Circle "Circle_4" at 201,254 size 23x23
      Appearance <- "Var_VectorPrincipalJ1{0,3}"
   Circle "Circle_5" at 92,224 size 23x23
      Appearance <- "Var_VectorPrincipalJ1{1,0}"
   Circle "Circle_6" at 128,224 size 23x23
      Appearance <- "Var_VectorPrincipalJ1{1,1}"
   Circle "Circle_7" at 164,224 size 23x23
      Appearance <- "Var_VectorPrincipalJ1{1,2}"
   Circle "Circle_8" at 201,224 size 23x23
      Appearance <- "Var_VectorPrincipalJ1{1,3}"
   Circle "Circle_9" at 92,194 size 23x23
      Appearance <- "Var_VectorPrincipalJ1{2,0}"
   Circle "Circle_10" at 128,194 size 23x23
      Appearance <- "Var_VectorPrincipalJ1{2,1}"
   Circle "Circle_11" at 164,194 size 23x23
      Appearance <- "Var_VectorPrincipalJ1{2,2}"
   Circle "Circle_12" at 201,194 size 23x23
      Appearance <- "Var_VectorPrincipalJ1{2,3}"
   Circle "Circle_13" at 92,164 size 23x23
      Appearance <- "Var_VectorPrincipalJ1{3,0}"
   Circle "Circle_14" at 128,164 size 23x23
      Appearance <- "Var_VectorPrincipalJ1{3,1}"
   Circle "Circle_15" at 164,164 size 23x23
      Appearance <- "Var_VectorPrincipalJ1{3,2}"
   Circle "Circle_16" at 201,164 size 23x23
      Appearance <- "Var_VectorPrincipalJ1{3,3}"
   Circle "Circle_17" at 92,134 size 23x23
      Appearance <- "Var_VectorPrincipalJ1{4,0}"
   Circle "Circle_18" at 128,134 size 23x23
      Appearance <- "Var_VectorPrincipalJ1{4,1}"
   Circle "Circle_19" at 164,134 size 23x23
      Appearance <- "Var_VectorPrincipalJ1{4,2}"
   Circle "Circle_20" at 201,134 size 23x23
      Appearance <- "Var_VectorPrincipalJ1{4,3}"
   Circle "Circle_21" at 92,104 size 23x23
      Appearance <- "Var_VectorPrincipalJ1{5,0}"
   Circle "Circle_22" at 128,104 size 23x23
      Appearance <- "Var_VectorPrincipalJ1{5,1}"
   Circle "Circle_23" at 164,104 size 23x23
      Appearance <- "Var_VectorPrincipalJ1{5,2}"
   Circle "Circle_24" at 201,104 size 23x23
      Appearance <- "Var_VectorPrincipalJ1{5,3}"
   Circle "Circle_25" at 92,74 size 23x23
      Appearance <- "Var_VectorPrincipalJ1{6,0}"
   Circle "Circle_26" at 128,74 size 23x23
      Appearance <- "Var_VectorPrincipalJ1{6,1}"
   Circle "Circle_27" at 164,74 size 23x23
      Appearance <- "Var_VectorPrincipalJ1{6,2}"
   Circle "Circle_28" at 201,74 size 23x23
      Appearance <- "Var_VectorPrincipalJ1{6,3}"
   Circle "Circle_29" at 92,44 size 23x23
      Appearance <- "Var_VectorPrincipalJ1{7,0}"
   Circle "Circle_30" at 128,44 size 23x23
      Appearance <- "Var_VectorPrincipalJ1{7,1}"
   Circle "Circle_31" at 164,44 size 23x23
      Appearance <- "Var_VectorPrincipalJ1{7,2}"
   Circle "Circle_32" at 201,44 size 23x23
      Appearance <- "Var_VectorPrincipalJ1{7,3}"
   Circle "Circle_33" at 255,253 size 14x14
      Appearance <- "Var_VectorSecundarioJ1{0,0}"
   Circle "Circle_34" at 270,253 size 14x14
      Appearance <- "Var_VectorSecundarioJ1{0,1}"
   Circle "Circle_35" at 255,267 size 14x14
      Appearance <- "Var_VectorSecundarioJ1{0,2}"
   Circle "Circle_36" at 270,267 size 14x14
      Appearance <- "Var_VectorSecundarioJ1{0,3}"
   Circle "Circle_37" at 255,223 size 14x14
      Appearance <- "Var_VectorSecundarioJ1{1,0}"
   Circle "Circle_38" at 270,223 size 14x14
      Appearance <- "Var_VectorSecundarioJ1{1,1}"
   Circle "Circle_39" at 255,237 size 14x14
      Appearance <- "Var_VectorSecundarioJ1{1,2}"
   Circle "Circle_40" at 270,237 size 14x14
      Appearance <- "Var_VectorSecundarioJ1{1,3}"
   Circle "Circle_41" at 255,193 size 14x14
      Appearance <- "Var_VectorSecundarioJ1{2,0}"
   Circle "Circle_42" at 270,193 size 14x14
      Appearance <- "Var_VectorSecundarioJ1{2,1}"
   Circle "Circle_43" at 255,207 size 14x14
      Appearance <- "Var_VectorSecundarioJ1{2,2}"
   Circle "Circle_44" at 270,207 size 14x14
      Appearance <- "Var_VectorSecundarioJ1{2,3}"
   Circle "Circle_45" at 255,163 size 14x14
      Appearance <- "Var_VectorSecundarioJ1{3,0}"
   Circle "Circle_46" at 270,163 size 14x14
      Appearance <- "Var_VectorSecundarioJ1{3,1}"
   Circle "Circle_47" at 255,177 size 14x14
      Appearance <- "Var_VectorSecundarioJ1{3,2}"
   Circle "Circle_48" at 270,177 size 14x14
      Appearance <- "Var_VectorSecundarioJ1{3,3}"
   Circle "Circle_49" at 255,133 size 14x14
      Appearance <- "Var_VectorSecundarioJ1{4,0}"
   Circle "Circle_50" at 270,133 size 14x14
      Appearance <- "Var_VectorSecundarioJ1{4,1}"
   Circle "Circle_51" at 255,147 size 14x14
      Appearance <- "Var_VectorSecundarioJ1{4,2}"
   Circle "Circle_52" at 270,147 size 14x14
      Appearance <- "Var_VectorSecundarioJ1{4,3}"
   Circle "Circle_53" at 255,103 size 14x14
      Appearance <- "Var_VectorSecundarioJ1{5,0}"
   Circle "Circle_54" at 270,103 size 14x14
      Appearance <- "Var_VectorSecundarioJ1{5,1}"
   Circle "Circle_55" at 255,117 size 14x14
      Appearance <- "Var_VectorSecundarioJ1{5,2}"
   Circle "Circle_56" at 270,117 size 14x14
      Appearance <- "Var_VectorSecundarioJ1{5,3}"
   Circle "Circle_57" at 255,73 size 14x14
      Appearance <- "Var_VectorSecundarioJ1{6,0}"
   Circle "Circle_58" at 270,73 size 14x14
      Appearance <- "Var_VectorSecundarioJ1{6,1}"
   Circle "Circle_59" at 255,87 size 14x14
      Appearance <- "Var_VectorSecundarioJ1{6,2}"
   Circle "Circle_60" at 270,87 size 14x14
      Appearance <- "Var_VectorSecundarioJ1{6,3}"
   Circle "Circle_61" at 255,43 size 14x14
      Appearance <- "Var_VectorSecundarioJ1{7,0}"
   Circle "Circle_62" at 270,43 size 14x14
      Appearance <- "Var_VectorSecundarioJ1{7,1}"
   Circle "Circle_63" at 255,57 size 14x14
      Appearance <- "Var_VectorSecundarioJ1{7,2}"
   Circle "Circle_64" at 270,57 size 14x14
      Appearance <- "Var_VectorSecundarioJ1{7,3}"
   TextField "Text field_9" at 339,40 size 252x42; Text 'Selecciona el Codigo de tu Oponente:'
   TextField "Text field_10" at 422,20 size 67x23; Text 'INICIO'
   Circle "Circle_65" at 393,108 size 29x29
      Appearance <- "Var_CodigoSJ1{0}"
   Circle "Circle_66" at 431,107 size 29x29
      Appearance <- "Var_CodigoSJ1{1}"
   Circle "Circle_67" at 467,108 size 29x29
      Appearance <- "Var_CodigoSJ1{2}"
   Circle "Circle_68" at 505,107 size 29x29
      Appearance <- "Var_CodigoSJ1{3}"
   Button "Button_10" at 360,160 size 28x26; TextOff 'Text'
      on Press: SetBit("Panel2CafeJ1")
      on Release: SetBit("Bounce1"); ResetBit("Panel2CafeJ1")
      Appearance <- "Panel2J1Activado"
   Button "Button_11" at 392,160 size 27x26; TextOff 'Text'
      on Press: SetBit("Panel2RosaJ1")
      on Release: SetBit("Bounce1"); ResetBit("Panel2RosaJ1")
      Appearance <- "Panel2J1Activado"
   Button "Button_12" at 424,160 size 27x24; TextOff 'Text'
      on Press: SetBit("Panel2MoradoJ1")
      on Release: SetBit("Bounce1"); ResetBit("Panel2MoradoJ1")
      Appearance <- "Panel2J1Activado"
   Button "Button_13" at 458,160 size 25x25; TextOff 'Text'
      on Press: SetBit("Panel2RojoJ1")
      on Release: SetBit("Bounce1"); ResetBit("Panel2RojoJ1")
      Appearance <- "Panel2J1Activado"
   Button "Button_14" at 489,160 size 25x24; TextOff 'Text'
      on Press: SetBit("Panel2AzulJ1")
      on Release: SetBit("Bounce1"); ResetBit("Panel2AzulJ1")
      Appearance <- "Panel2J1Activado"
   Button "Button_16" at 520,160 size 25x25; TextOff 'Text'
      on Press: SetBit("Panel2VerdeJ1")
      on Release: SetBit("Bounce1"); ResetBit("Panel2VerdeJ1")
      Appearance <- "Panel2J1Activado"
   Button "Button_17" at 549,161 size 25x23; TextOff 'Text'
      on Press: SetBit("Panel2AmarilloJ1")
      on Release: SetBit("Bounce1"); ResetBit("Panel2AmarilloJ1")
      Appearance <- "Panel2J1Activado"
   Circle "Circle_69" at 342,274 size 29x29
      Appearance <- "Var_CodigoOJ1{0}"
   Circle "Circle_70" at 379,274 size 29x29
      Appearance <- "Var_CodigoOJ1{1}"
   Circle "Circle_71" at 416,274 size 29x29
      Appearance <- "Var_CodigoOJ1{2}"
   Circle "Circle_72" at 453,274 size 29x29
      Appearance <- "Var_CodigoOJ1{3}"
   TextField "Text field_11" at 341,233 size 142x23; Text 'Codigo Secreto'
   Button "Button_18" at 621,289 size 135x35; TextOff 'Reiniciar Juego'
      on Press: SetBit("ReiniciarJuego")
      on Release: ResetBit("ReiniciarJuego")
   Rectangle "Rectangle_23" at 401,90 size 13x8
      Appearance <- "Var_CodigoSJ1{0}"
   Rectangle "Rectangle_24" at 438,90 size 13x8
      Appearance <- "Var_CodigoSJ1{1}"
   Rectangle "Rectangle_25" at 475,90 size 13x8
      Appearance <- "Var_CodigoSJ1{2}"
   Rectangle "Rectangle_26" at 512,90 size 13x8
      Appearance <- "Var_CodigoSJ1{3}"
   TextField "Text field_12" at 626,28 size 120x17; Text '1. Selecciona un codigo'
      Visibility <- "Var_VectorMensajes{0}"
   TextField "Text field_13" at 627,48 size 117x43; Text '2. Esperando a que el otro jugador seleccione tu codigo'
      Visibility <- "Var_VectorMensajes{1}"
   TextField "Text field_14" at 625,94 size 130x30; Text '3. Ambos codigos seleccionados. Preparate!'
      Visibility <- "Var_VectorMensajes{2}"
   TextField "Text field_15" at 678,126 size 14x20; Text '5'
      Visibility <- "Var_VectorMensajes{3}"
   TextField "Text field_16" at 678,143 size 14x20; Text '4'
      Visibility <- "Var_VectorMensajes{4}"
   TextField "Text field_17" at 679,160 size 14x20; Text '3'
      Visibility <- "Var_VectorMensajes{5}"
   TextField "Text field_18" at 679,178 size 14x20; Text '2'
      Visibility <- "Var_VectorMensajes{6}"
   TextField "Text field_19" at 679,195 size 14x20; Text '1'
      Visibility <- "Var_VectorMensajes{7}"
   TextField "Text field_20" at 632,219 size 119x43; Text '4. Encuentra el codigo secreto antes que tu oponente!'
      Visibility <- "Var_VectorMensajes{8}"
   TextField "Text field_21" at 501,241 size 101x22; Text 'GANASTE!!!'
      Visibility <- "Var_VectorMensajes{9}"
   TextField "Text field_22" at 503,280 size 108x22; Text 'PERDISTE :('
      Visibility <- "Var_VectorMensajes{10}"

Template "Template_1" 800x442
   Button "Exit" at 720,360 size 78x58; TextOff 'Exit'; PictureOff "ExitRuntime_TP700_Comfort_TR"; PictureOn "ExitRuntime_TP700_Comfort_TR"
      on Release: StopRuntime(0)
   Button "Template_Button" at 640,360 size 78x58; TextOff 'Text'
   Button "Template_Button_1" at 560,360 size 78x58; TextOff 'Text'
   Button "Template_Button_2" at 480,360 size 78x58; TextOff 'Text'
   Button "Template_Button_3" at 400,360 size 78x58; TextOff 'Text'
   Button "Template_Button_4" at 321,360 size 78x58; TextOff 'Text'
   Button "Template_Button_5" at 241,360 size 78x58; TextOff 'Text'
   Button "Template_Button_6" at 161,360 size 78x58; TextOff 'Text'
   Button "Alarms" at 81,360 size 78x58; TextOff 'Alarms'; PictureOff "AlarmDisplay_TP700_Comfort_TR"; PictureOn "AlarmDisplay_TP700_Comfort_TR"
      on Release: function_ef3f5d25("Alarm window_Unacknowledged", -1)
   Button "Start screen" at 1,360 size 78x58; TextOff 'Start screen'; PictureOff "NavigateHome_TP700_Comfort_TR"; PictureOn "NavigateHome_TP700_Comfort_TR"
      on Release: ActivateScreen("Root screen", 0)
*)